REGION Network 62: ALL UNCLAMPED UNIT 02
   RUNG wire#powerrail
      Contact( "DB3510_U2_F1_GRIPPER".CYL.FULL_OPEN )
      wire#w1
      Contact( "DB3810_U2_F4_GRIPPER".CYL.FULL_OPEN )
      wire#w2
      Contact( "DB3610_U2_F2_GRIPPER".CYL.FULL_OPEN )
      wire#w3
      Contact( "DB3710_U2_F3_GRIPPER".CYL.FULL_OPEN )
      wire#w4
      Contact( "DB7215_PART_TYPE".PART_TYPE_U02_FIXTURES )
      Coil( "DB2440_GLOBAL_DATA".GLOBAL_DATA.ALL_UNCLAMPED_UNIT_02 )
   END_RUNG
   RUNG wire#powerrail
      Contact( "DB3500_UNIT_02_FIXTURE_1".CLAMPED_WITHOUT_PART_ANALOG )
   END_RUNG wire#w1
   RUNG wire#w1
      Contact( "DB3800_UNIT_02_FIXTURE_4".CLAMPED_WITHOUT_PART_ANALOG )
   END_RUNG wire#w2
   RUNG wire#powerrail
      I_Contact( "DB7240_HARDWARE_SOFTWARE_ENABLE_DISABLE".DISABLE_FIXTURE.SW_UNIT_2_FIX_1_4_ENABLED )
   END_RUNG wire#w2
   RUNG wire#w2
      Contact( "DB3600_UNIT_02_FIXTURE_2".CLAMPED_WITHOUT_PART_ANALOG )
   END_RUNG wire#w3
   RUNG wire#w3
      Contact( "DB3700_UNIT_02_FIXTURE_3".CLAMPED_WITHOUT_PART_ANALOG )
   END_RUNG wire#w4
   RUNG wire#w2
      I_Contact( "DB7240_HARDWARE_SOFTWARE_ENABLE_DISABLE".DISABLE_FIXTURE.SW_UNIT_2_FIX_2_3_ENABLED )
   END_RUNG wire#w4
   // the same network as SCL:
   "DB2440_GLOBAL_DATA".GLOBAL_DATA.ALL_UNCLAMPED_UNIT_02 := ((("DB3510_U2_F1_GRIPPER".CYL.FULL_OPEN OR "DB3500_UNIT_02_FIXTURE_1".CLAMPED_WITHOUT_PART_ANALOG) AND ("DB3810_U2_F4_GRIPPER".CYL.FULL_OPEN OR "DB3800_UNIT_02_FIXTURE_4".CLAMPED_WITHOUT_PART_ANALOG)) OR NOT "DB7240_HARDWARE_SOFTWARE_ENABLE_DISABLE".DISABLE_FIXTURE.SW_UNIT_2_FIX_1_4_ENABLED) AND ((("DB3610_U2_F2_GRIPPER".CYL.FULL_OPEN OR "DB3600_UNIT_02_FIXTURE_2".CLAMPED_WITHOUT_PART_ANALOG) AND ("DB3710_U2_F3_GRIPPER".CYL.FULL_OPEN OR "DB3700_UNIT_02_FIXTURE_3".CLAMPED_WITHOUT_PART_ANALOG)) OR NOT "DB7240_HARDWARE_SOFTWARE_ENABLE_DISABLE".DISABLE_FIXTURE.SW_UNIT_2_FIX_2_3_ENABLED) AND "DB7215_PART_TYPE".PART_TYPE_U02_FIXTURES;
END_REGION

REGION Network 63: CLAMPED OR UNCLAMPED UNIT 02
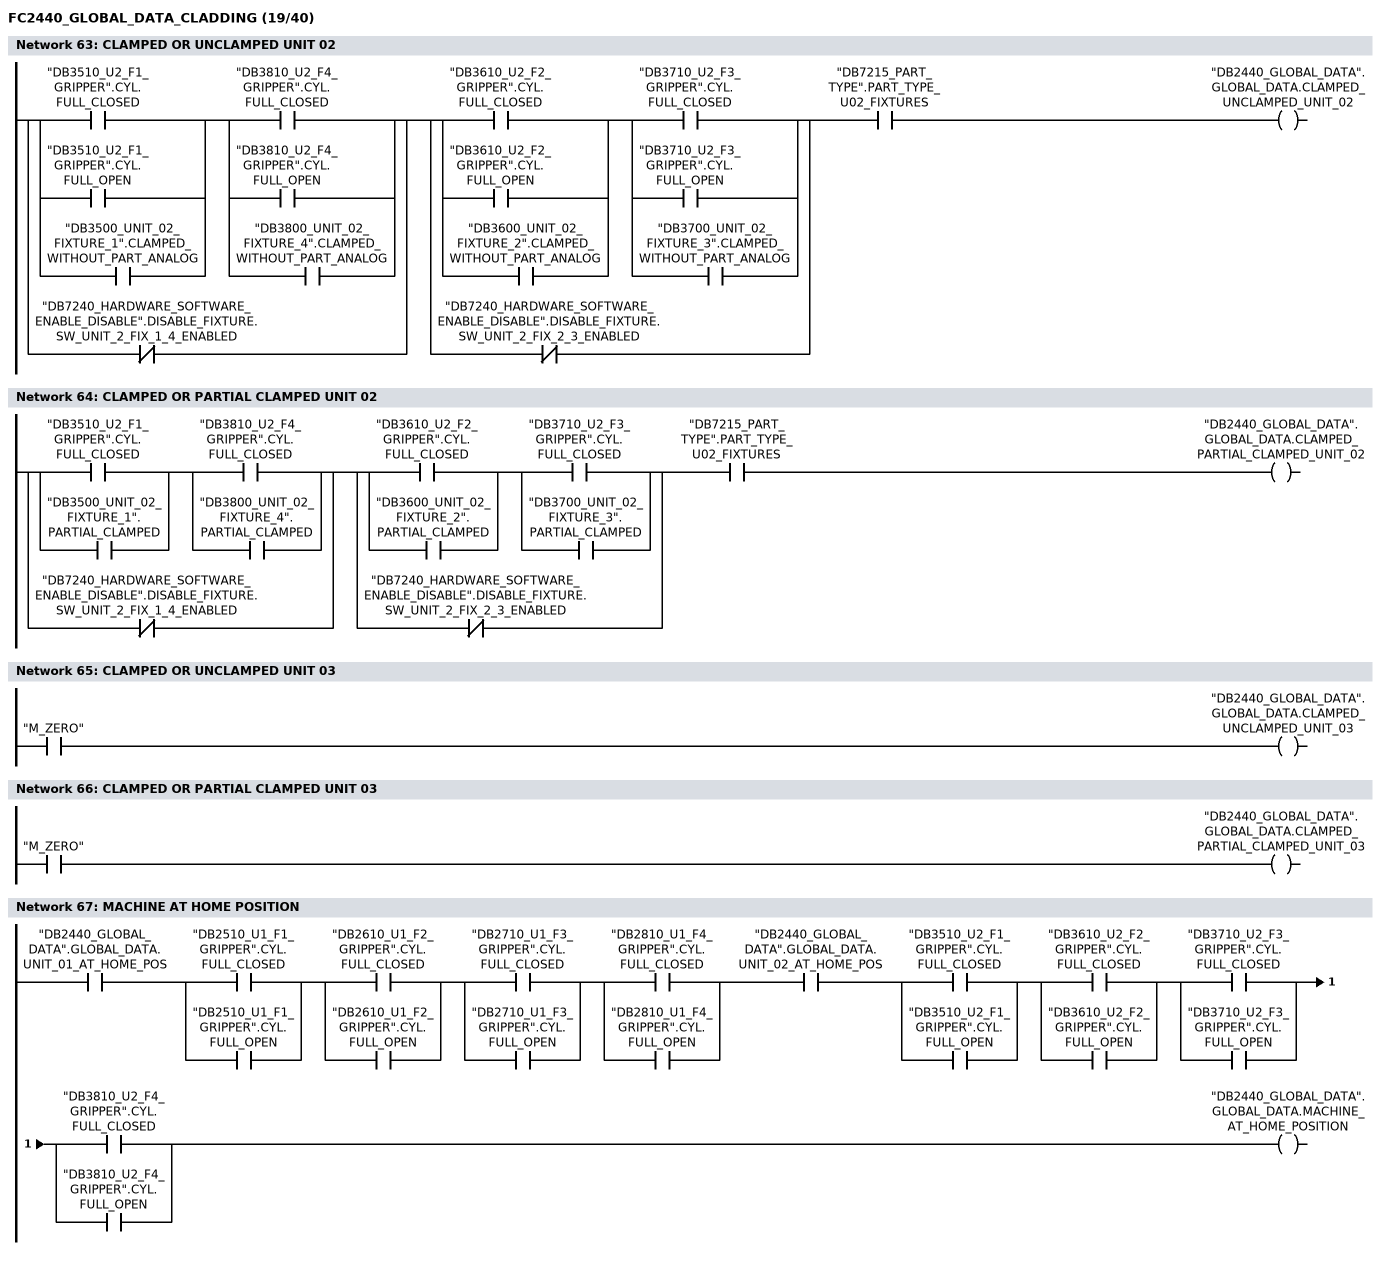
   RUNG wire#powerrail
      Contact( "DB3510_U2_F1_GRIPPER".CYL.FULL_CLOSED )
      wire#w1
      Contact( "DB3810_U2_F4_GRIPPER".CYL.FULL_CLOSED )
      wire#w2
      Contact( "DB3610_U2_F2_GRIPPER".CYL.FULL_CLOSED )
      wire#w3
      Contact( "DB3710_U2_F3_GRIPPER".CYL.FULL_CLOSED )
      wire#w4
      Contact( "DB7215_PART_TYPE".PART_TYPE_U02_FIXTURES )
      Coil( "DB2440_GLOBAL_DATA".GLOBAL_DATA.CLAMPED_UNCLAMPED_UNIT_02 )
   END_RUNG
   RUNG wire#powerrail
      Contact( "DB3510_U2_F1_GRIPPER".CYL.FULL_OPEN )
   END_RUNG wire#w1
   RUNG wire#powerrail
      Contact( "DB3500_UNIT_02_FIXTURE_1".CLAMPED_WITHOUT_PART_ANALOG )
   END_RUNG wire#w1
   RUNG wire#w1
      Contact( "DB3810_U2_F4_GRIPPER".CYL.FULL_OPEN )
   END_RUNG wire#w2
   RUNG wire#w1
      Contact( "DB3800_UNIT_02_FIXTURE_4".CLAMPED_WITHOUT_PART_ANALOG )
   END_RUNG wire#w2
   RUNG wire#powerrail
      I_Contact( "DB7240_HARDWARE_SOFTWARE_ENABLE_DISABLE".DISABLE_FIXTURE.SW_UNIT_2_FIX_1_4_ENABLED )
   END_RUNG wire#w2
   RUNG wire#w2
      Contact( "DB3610_U2_F2_GRIPPER".CYL.FULL_OPEN )
   END_RUNG wire#w3
   RUNG wire#w2
      Contact( "DB3600_UNIT_02_FIXTURE_2".CLAMPED_WITHOUT_PART_ANALOG )
   END_RUNG wire#w3
   RUNG wire#w3
      Contact( "DB3710_U2_F3_GRIPPER".CYL.FULL_OPEN )
   END_RUNG wire#w4
   RUNG wire#w3
      Contact( "DB3700_UNIT_02_FIXTURE_3".CLAMPED_WITHOUT_PART_ANALOG )
   END_RUNG wire#w4
   RUNG wire#w2
      I_Contact( "DB7240_HARDWARE_SOFTWARE_ENABLE_DISABLE".DISABLE_FIXTURE.SW_UNIT_2_FIX_2_3_ENABLED )
   END_RUNG wire#w4
   // the same network as SCL:
   "DB2440_GLOBAL_DATA".GLOBAL_DATA.CLAMPED_UNCLAMPED_UNIT_02 := ((("DB3510_U2_F1_GRIPPER".CYL.FULL_CLOSED OR "DB3510_U2_F1_GRIPPER".CYL.FULL_OPEN OR "DB3500_UNIT_02_FIXTURE_1".CLAMPED_WITHOUT_PART_ANALOG) AND ("DB3810_U2_F4_GRIPPER".CYL.FULL_CLOSED OR "DB3810_U2_F4_GRIPPER".CYL.FULL_OPEN OR "DB3800_UNIT_02_FIXTURE_4".CLAMPED_WITHOUT_PART_ANALOG)) OR NOT "DB7240_HARDWARE_SOFTWARE_ENABLE_DISABLE".DISABLE_FIXTURE.SW_UNIT_2_FIX_1_4_ENABLED) AND ((("DB3610_U2_F2_GRIPPER".CYL.FULL_CLOSED OR "DB3610_U2_F2_GRIPPER".CYL.FULL_OPEN OR "DB3600_UNIT_02_FIXTURE_2".CLAMPED_WITHOUT_PART_ANALOG) AND ("DB3710_U2_F3_GRIPPER".CYL.FULL_CLOSED OR "DB3710_U2_F3_GRIPPER".CYL.FULL_OPEN OR "DB3700_UNIT_02_FIXTURE_3".CLAMPED_WITHOUT_PART_ANALOG)) OR NOT "DB7240_HARDWARE_SOFTWARE_ENABLE_DISABLE".DISABLE_FIXTURE.SW_UNIT_2_FIX_2_3_ENABLED) AND "DB7215_PART_TYPE".PART_TYPE_U02_FIXTURES;
END_REGION

REGION Network 64: CLAMPED OR PARTIAL CLAMPED UNIT 02
   RUNG wire#powerrail
      Contact( "DB3510_U2_F1_GRIPPER".CYL.FULL_CLOSED )
      wire#w1
      Contact( "DB3810_U2_F4_GRIPPER".CYL.FULL_CLOSED )
      wire#w2
      Contact( "DB3610_U2_F2_GRIPPER".CYL.FULL_CLOSED )
      wire#w3
      Contact( "DB3710_U2_F3_GRIPPER".CYL.FULL_CLOSED )
      wire#w4
      Contact( "DB7215_PART_TYPE".PART_TYPE_U02_FIXTURES )
      Coil( "DB2440_GLOBAL_DATA".GLOBAL_DATA.CLAMPED_PARTIAL_CLAMPED_UNIT_02 )
   END_RUNG
   RUNG wire#powerrail
      Contact( "DB3500_UNIT_02_FIXTURE_1".PARTIAL_CLAMPED )
   END_RUNG wire#w1
   RUNG wire#w1
      Contact( "DB3800_UNIT_02_FIXTURE_4".PARTIAL_CLAMPED )
   END_RUNG wire#w2
   RUNG wire#powerrail
      I_Contact( "DB7240_HARDWARE_SOFTWARE_ENABLE_DISABLE".DISABLE_FIXTURE.SW_UNIT_2_FIX_1_4_ENABLED )
   END_RUNG wire#w2
   RUNG wire#w2
      Contact( "DB3600_UNIT_02_FIXTURE_2".PARTIAL_CLAMPED )
   END_RUNG wire#w3
   RUNG wire#w3
      Contact( "DB3700_UNIT_02_FIXTURE_3".PARTIAL_CLAMPED )
   END_RUNG wire#w4
   RUNG wire#w2
      I_Contact( "DB7240_HARDWARE_SOFTWARE_ENABLE_DISABLE".DISABLE_FIXTURE.SW_UNIT_2_FIX_2_3_ENABLED )
   END_RUNG wire#w4
   // the same network as SCL:
   "DB2440_GLOBAL_DATA".GLOBAL_DATA.CLAMPED_PARTIAL_CLAMPED_UNIT_02 := ((("DB3510_U2_F1_GRIPPER".CYL.FULL_CLOSED OR "DB3500_UNIT_02_FIXTURE_1".PARTIAL_CLAMPED) AND ("DB3810_U2_F4_GRIPPER".CYL.FULL_CLOSED OR "DB3800_UNIT_02_FIXTURE_4".PARTIAL_CLAMPED)) OR NOT "DB7240_HARDWARE_SOFTWARE_ENABLE_DISABLE".DISABLE_FIXTURE.SW_UNIT_2_FIX_1_4_ENABLED) AND ((("DB3610_U2_F2_GRIPPER".CYL.FULL_CLOSED OR "DB3600_UNIT_02_FIXTURE_2".PARTIAL_CLAMPED) AND ("DB3710_U2_F3_GRIPPER".CYL.FULL_CLOSED OR "DB3700_UNIT_02_FIXTURE_3".PARTIAL_CLAMPED)) OR NOT "DB7240_HARDWARE_SOFTWARE_ENABLE_DISABLE".DISABLE_FIXTURE.SW_UNIT_2_FIX_2_3_ENABLED) AND "DB7215_PART_TYPE".PART_TYPE_U02_FIXTURES;
END_REGION

REGION Network 65: CLAMPED OR UNCLAMPED UNIT 03
   RUNG wire#powerrail
      Contact( "M_ZERO" )
      Coil( "DB2440_GLOBAL_DATA".GLOBAL_DATA.CLAMPED_UNCLAMPED_UNIT_03 )
   END_RUNG
   // the same network as SCL:
   "DB2440_GLOBAL_DATA".GLOBAL_DATA.CLAMPED_UNCLAMPED_UNIT_03 := "M_ZERO";
END_REGION

REGION Network 66: CLAMPED OR PARTIAL CLAMPED UNIT 03
   RUNG wire#powerrail
      Contact( "M_ZERO" )
      Coil( "DB2440_GLOBAL_DATA".GLOBAL_DATA.CLAMPED_PARTIAL_CLAMPED_UNIT_03 )
   END_RUNG
   // the same network as SCL:
   "DB2440_GLOBAL_DATA".GLOBAL_DATA.CLAMPED_PARTIAL_CLAMPED_UNIT_03 := "M_ZERO";
END_REGION

REGION Network 67: MACHINE AT HOME POSITION
   RUNG wire#powerrail
      Contact( "DB2440_GLOBAL_DATA".GLOBAL_DATA.UNIT_01_AT_HOME_POS )
      wire#w1
      Contact( "DB2510_U1_F1_GRIPPER".CYL.FULL_CLOSED )
      wire#w2
      Contact( "DB2610_U1_F2_GRIPPER".CYL.FULL_CLOSED )
      wire#w3
      Contact( "DB2710_U1_F3_GRIPPER".CYL.FULL_CLOSED )
      wire#w4
      Contact( "DB2810_U1_F4_GRIPPER".CYL.FULL_CLOSED )
      wire#w5
      Contact( "DB2440_GLOBAL_DATA".GLOBAL_DATA.UNIT_02_AT_HOME_POS )
      wire#w6
      Contact( "DB3510_U2_F1_GRIPPER".CYL.FULL_CLOSED )
      wire#w7
      Contact( "DB3610_U2_F2_GRIPPER".CYL.FULL_CLOSED )
      wire#w8
      Contact( "DB3710_U2_F3_GRIPPER".CYL.FULL_CLOSED )
      wire#w9
      Contact( "DB3810_U2_F4_GRIPPER".CYL.FULL_CLOSED )
      wire#w10
      Coil( "DB2440_GLOBAL_DATA".GLOBAL_DATA.MACHINE_AT_HOME_POSITION )
   END_RUNG
   RUNG wire#w1
      Contact( "DB2510_U1_F1_GRIPPER".CYL.FULL_OPEN )
   END_RUNG wire#w2
   RUNG wire#w2
      Contact( "DB2610_U1_F2_GRIPPER".CYL.FULL_OPEN )
   END_RUNG wire#w3
   RUNG wire#w3
      Contact( "DB2710_U1_F3_GRIPPER".CYL.FULL_OPEN )
   END_RUNG wire#w4
   RUNG wire#w4
      Contact( "DB2810_U1_F4_GRIPPER".CYL.FULL_OPEN )
   END_RUNG wire#w5
   RUNG wire#w6
      Contact( "DB3510_U2_F1_GRIPPER".CYL.FULL_OPEN )
   END_RUNG wire#w7
   RUNG wire#w7
      Contact( "DB3610_U2_F2_GRIPPER".CYL.FULL_OPEN )
   END_RUNG wire#w8
   RUNG wire#w8
      Contact( "DB3710_U2_F3_GRIPPER".CYL.FULL_OPEN )
   END_RUNG wire#w9
   RUNG wire#w9
      Contact( "DB3810_U2_F4_GRIPPER".CYL.FULL_OPEN )
   END_RUNG wire#w10
   // the same network as SCL:
   "DB2440_GLOBAL_DATA".GLOBAL_DATA.MACHINE_AT_HOME_POSITION := "DB2440_GLOBAL_DATA".GLOBAL_DATA.UNIT_01_AT_HOME_POS AND ("DB2510_U1_F1_GRIPPER".CYL.FULL_CLOSED OR "DB2510_U1_F1_GRIPPER".CYL.FULL_OPEN) AND ("DB2610_U1_F2_GRIPPER".CYL.FULL_CLOSED OR "DB2610_U1_F2_GRIPPER".CYL.FULL_OPEN) AND ("DB2710_U1_F3_GRIPPER".CYL.FULL_CLOSED OR "DB2710_U1_F3_GRIPPER".CYL.FULL_OPEN) AND ("DB2810_U1_F4_GRIPPER".CYL.FULL_CLOSED OR "DB2810_U1_F4_GRIPPER".CYL.FULL_OPEN) AND "DB2440_GLOBAL_DATA".GLOBAL_DATA.UNIT_02_AT_HOME_POS AND ("DB3510_U2_F1_GRIPPER".CYL.FULL_CLOSED OR "DB3510_U2_F1_GRIPPER".CYL.FULL_OPEN) AND ("DB3610_U2_F2_GRIPPER".CYL.FULL_CLOSED OR "DB3610_U2_F2_GRIPPER".CYL.FULL_OPEN) AND ("DB3710_U2_F3_GRIPPER".CYL.FULL_CLOSED OR "DB3710_U2_F3_GRIPPER".CYL.FULL_OPEN) AND ("DB3810_U2_F4_GRIPPER".CYL.FULL_CLOSED OR "DB3810_U2_F4_GRIPPER".CYL.FULL_OPEN);
END_REGION

REGION Network 68: UNIT 01 STATION 0 ANY CYCLE ACTIVE
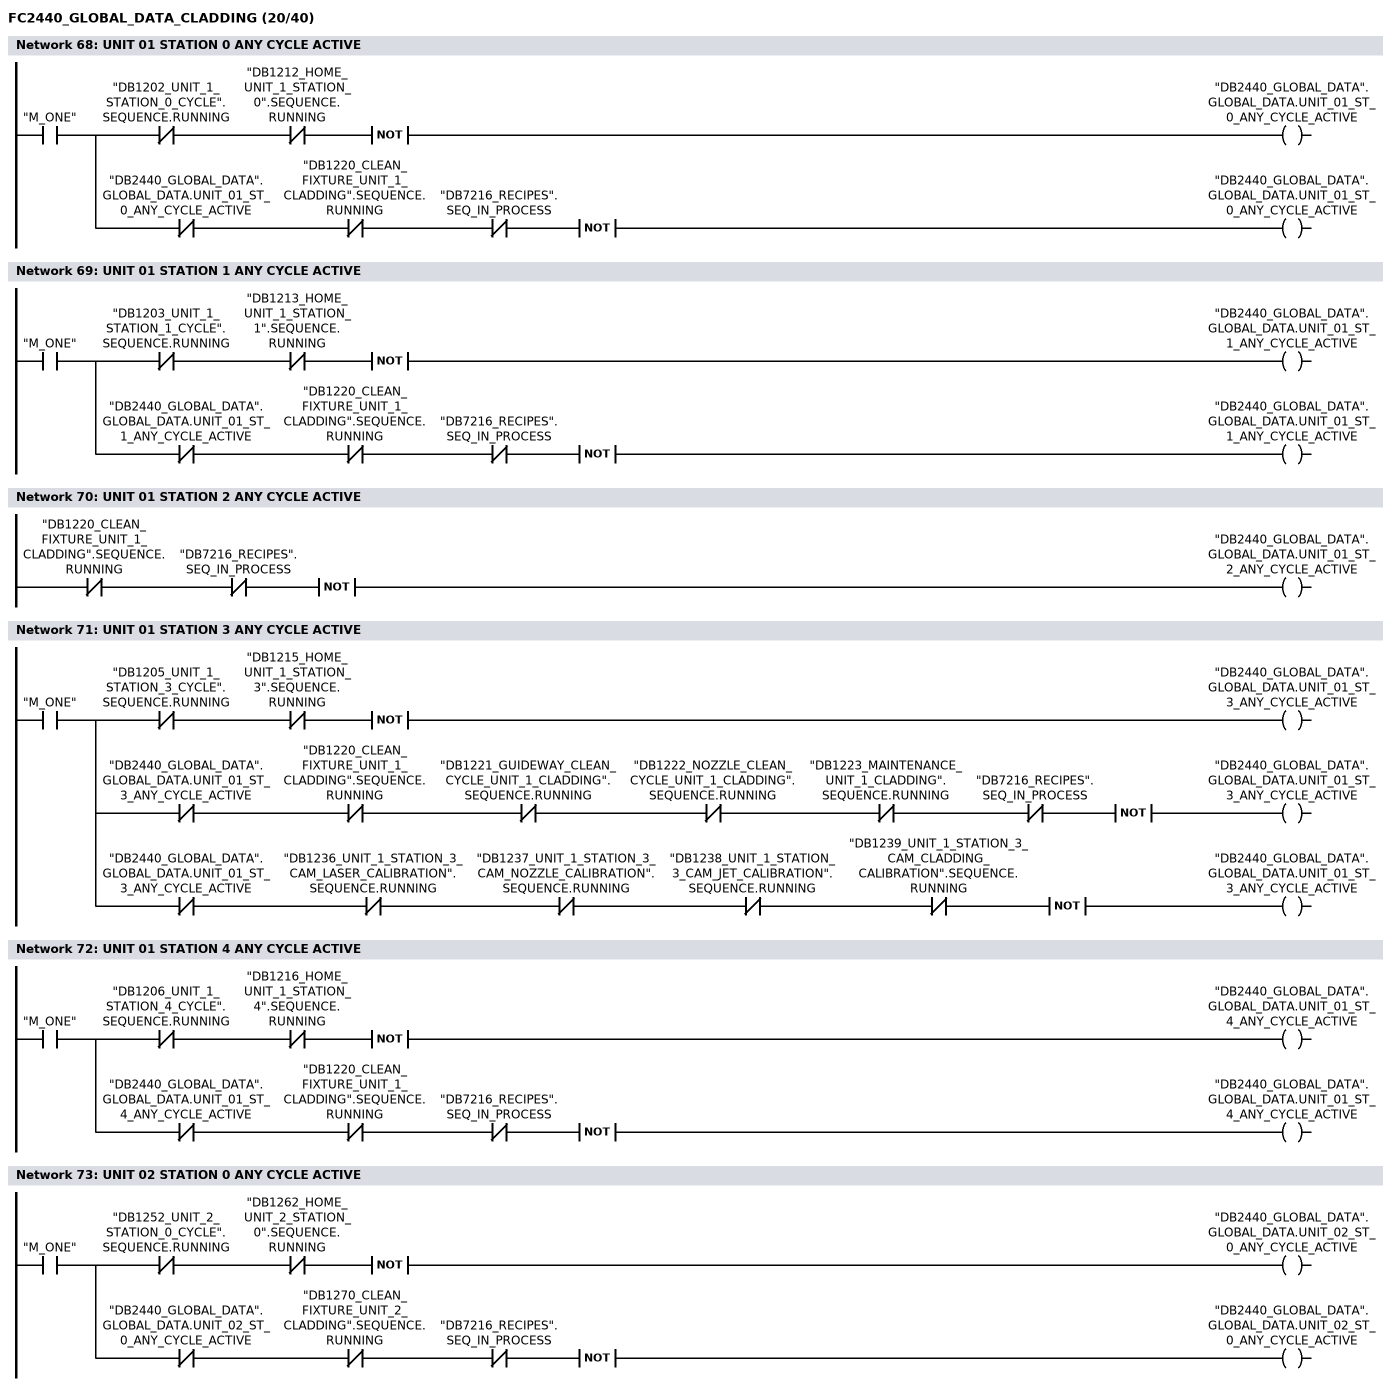
   RUNG wire#powerrail
      Contact( "M_ONE" )
      wire#w1
      I_Contact( "DB1202_UNIT_1_STATION_0_CYCLE".SEQUENCE.RUNNING )
      I_Contact( "DB1212_HOME_UNIT_1_STATION_0".SEQUENCE.RUNNING )
      Not()
      Coil( "DB2440_GLOBAL_DATA".GLOBAL_DATA.UNIT_01_ST_0_ANY_CYCLE_ACTIVE )
   END_RUNG
   RUNG wire#w1
      I_Contact( "DB2440_GLOBAL_DATA".GLOBAL_DATA.UNIT_01_ST_0_ANY_CYCLE_ACTIVE )
      I_Contact( "DB1220_CLEAN_FIXTURE_UNIT_1_CLADDING".SEQUENCE.RUNNING )
      I_Contact( "DB7216_RECIPES".SEQ_IN_PROCESS )
      Not()
      Coil( "DB2440_GLOBAL_DATA".GLOBAL_DATA.UNIT_01_ST_0_ANY_CYCLE_ACTIVE )
   END_RUNG
   // the same network as SCL:
   "DB2440_GLOBAL_DATA".GLOBAL_DATA.UNIT_01_ST_0_ANY_CYCLE_ACTIVE := NOT ("M_ONE" AND NOT "DB1202_UNIT_1_STATION_0_CYCLE".SEQUENCE.RUNNING AND NOT "DB1212_HOME_UNIT_1_STATION_0".SEQUENCE.RUNNING);
   "DB2440_GLOBAL_DATA".GLOBAL_DATA.UNIT_01_ST_0_ANY_CYCLE_ACTIVE := NOT ("M_ONE" AND NOT "DB2440_GLOBAL_DATA".GLOBAL_DATA.UNIT_01_ST_0_ANY_CYCLE_ACTIVE AND NOT "DB1220_CLEAN_FIXTURE_UNIT_1_CLADDING".SEQUENCE.RUNNING AND NOT "DB7216_RECIPES".SEQ_IN_PROCESS);
END_REGION

REGION Network 69: UNIT 01 STATION 1 ANY CYCLE ACTIVE
   RUNG wire#powerrail
      Contact( "M_ONE" )
      wire#w1
      I_Contact( "DB1203_UNIT_1_STATION_1_CYCLE".SEQUENCE.RUNNING )
      I_Contact( "DB1213_HOME_UNIT_1_STATION_1".SEQUENCE.RUNNING )
      Not()
      Coil( "DB2440_GLOBAL_DATA".GLOBAL_DATA.UNIT_01_ST_1_ANY_CYCLE_ACTIVE )
   END_RUNG
   RUNG wire#w1
      I_Contact( "DB2440_GLOBAL_DATA".GLOBAL_DATA.UNIT_01_ST_1_ANY_CYCLE_ACTIVE )
      I_Contact( "DB1220_CLEAN_FIXTURE_UNIT_1_CLADDING".SEQUENCE.RUNNING )
      I_Contact( "DB7216_RECIPES".SEQ_IN_PROCESS )
      Not()
      Coil( "DB2440_GLOBAL_DATA".GLOBAL_DATA.UNIT_01_ST_1_ANY_CYCLE_ACTIVE )
   END_RUNG
   // the same network as SCL:
   "DB2440_GLOBAL_DATA".GLOBAL_DATA.UNIT_01_ST_1_ANY_CYCLE_ACTIVE := NOT ("M_ONE" AND NOT "DB1203_UNIT_1_STATION_1_CYCLE".SEQUENCE.RUNNING AND NOT "DB1213_HOME_UNIT_1_STATION_1".SEQUENCE.RUNNING);
   "DB2440_GLOBAL_DATA".GLOBAL_DATA.UNIT_01_ST_1_ANY_CYCLE_ACTIVE := NOT ("M_ONE" AND NOT "DB2440_GLOBAL_DATA".GLOBAL_DATA.UNIT_01_ST_1_ANY_CYCLE_ACTIVE AND NOT "DB1220_CLEAN_FIXTURE_UNIT_1_CLADDING".SEQUENCE.RUNNING AND NOT "DB7216_RECIPES".SEQ_IN_PROCESS);
END_REGION

REGION Network 70: UNIT 01 STATION 2 ANY CYCLE ACTIVE
   RUNG wire#powerrail
      I_Contact( "DB1220_CLEAN_FIXTURE_UNIT_1_CLADDING".SEQUENCE.RUNNING )
      I_Contact( "DB7216_RECIPES".SEQ_IN_PROCESS )
      Not()
      Coil( "DB2440_GLOBAL_DATA".GLOBAL_DATA.UNIT_01_ST_2_ANY_CYCLE_ACTIVE )
   END_RUNG
   // the same network as SCL:
   "DB2440_GLOBAL_DATA".GLOBAL_DATA.UNIT_01_ST_2_ANY_CYCLE_ACTIVE := NOT (NOT "DB1220_CLEAN_FIXTURE_UNIT_1_CLADDING".SEQUENCE.RUNNING AND NOT "DB7216_RECIPES".SEQ_IN_PROCESS);
END_REGION

REGION Network 71: UNIT 01 STATION 3 ANY CYCLE ACTIVE
   RUNG wire#powerrail
      Contact( "M_ONE" )
      wire#w1
      I_Contact( "DB1205_UNIT_1_STATION_3_CYCLE".SEQUENCE.RUNNING )
      I_Contact( "DB1215_HOME_UNIT_1_STATION_3".SEQUENCE.RUNNING )
      Not()
      Coil( "DB2440_GLOBAL_DATA".GLOBAL_DATA.UNIT_01_ST_3_ANY_CYCLE_ACTIVE )
   END_RUNG
   RUNG wire#w1
      I_Contact( "DB2440_GLOBAL_DATA".GLOBAL_DATA.UNIT_01_ST_3_ANY_CYCLE_ACTIVE )
      I_Contact( "DB1220_CLEAN_FIXTURE_UNIT_1_CLADDING".SEQUENCE.RUNNING )
      I_Contact( "DB1221_GUIDEWAY_CLEAN_CYCLE_UNIT_1_CLADDING".SEQUENCE.RUNNING )
      I_Contact( "DB1222_NOZZLE_CLEAN_CYCLE_UNIT_1_CLADDING".SEQUENCE.RUNNING )
      I_Contact( "DB1223_MAINTENANCE_UNIT_1_CLADDING".SEQUENCE.RUNNING )
      I_Contact( "DB7216_RECIPES".SEQ_IN_PROCESS )
      Not()
      Coil( "DB2440_GLOBAL_DATA".GLOBAL_DATA.UNIT_01_ST_3_ANY_CYCLE_ACTIVE )
   END_RUNG
   RUNG wire#w1
      I_Contact( "DB2440_GLOBAL_DATA".GLOBAL_DATA.UNIT_01_ST_3_ANY_CYCLE_ACTIVE )
      I_Contact( "DB1236_UNIT_1_STATION_3_CAM_LASER_CALIBRATION".SEQUENCE.RUNNING )
      I_Contact( "DB1237_UNIT_1_STATION_3_CAM_NOZZLE_CALIBRATION".SEQUENCE.RUNNING )
      I_Contact( "DB1238_UNIT_1_STATION_3_CAM_JET_CALIBRATION".SEQUENCE.RUNNING )
      I_Contact( "DB1239_UNIT_1_STATION_3_CAM_CLADDING_CALIBRATION".SEQUENCE.RUNNING )
      Not()
      Coil( "DB2440_GLOBAL_DATA".GLOBAL_DATA.UNIT_01_ST_3_ANY_CYCLE_ACTIVE )
   END_RUNG
   // the same network as SCL:
   "DB2440_GLOBAL_DATA".GLOBAL_DATA.UNIT_01_ST_3_ANY_CYCLE_ACTIVE := NOT ("M_ONE" AND NOT "DB1205_UNIT_1_STATION_3_CYCLE".SEQUENCE.RUNNING AND NOT "DB1215_HOME_UNIT_1_STATION_3".SEQUENCE.RUNNING);
   "DB2440_GLOBAL_DATA".GLOBAL_DATA.UNIT_01_ST_3_ANY_CYCLE_ACTIVE := NOT ("M_ONE" AND NOT "DB2440_GLOBAL_DATA".GLOBAL_DATA.UNIT_01_ST_3_ANY_CYCLE_ACTIVE AND NOT "DB1220_CLEAN_FIXTURE_UNIT_1_CLADDING".SEQUENCE.RUNNING AND NOT "DB1221_GUIDEWAY_CLEAN_CYCLE_UNIT_1_CLADDING".SEQUENCE.RUNNING AND NOT "DB1222_NOZZLE_CLEAN_CYCLE_UNIT_1_CLADDING".SEQUENCE.RUNNING AND NOT "DB1223_MAINTENANCE_UNIT_1_CLADDING".SEQUENCE.RUNNING AND NOT "DB7216_RECIPES".SEQ_IN_PROCESS);
   "DB2440_GLOBAL_DATA".GLOBAL_DATA.UNIT_01_ST_3_ANY_CYCLE_ACTIVE := NOT ("M_ONE" AND NOT "DB2440_GLOBAL_DATA".GLOBAL_DATA.UNIT_01_ST_3_ANY_CYCLE_ACTIVE AND NOT "DB1236_UNIT_1_STATION_3_CAM_LASER_CALIBRATION".SEQUENCE.RUNNING AND NOT "DB1237_UNIT_1_STATION_3_CAM_NOZZLE_CALIBRATION".SEQUENCE.RUNNING AND NOT "DB1238_UNIT_1_STATION_3_CAM_JET_CALIBRATION".SEQUENCE.RUNNING AND NOT "DB1239_UNIT_1_STATION_3_CAM_CLADDING_CALIBRATION".SEQUENCE.RUNNING);
END_REGION

REGION Network 72: UNIT 01 STATION 4 ANY CYCLE ACTIVE
   RUNG wire#powerrail
      Contact( "M_ONE" )
      wire#w1
      I_Contact( "DB1206_UNIT_1_STATION_4_CYCLE".SEQUENCE.RUNNING )
      I_Contact( "DB1216_HOME_UNIT_1_STATION_4".SEQUENCE.RUNNING )
      Not()
      Coil( "DB2440_GLOBAL_DATA".GLOBAL_DATA.UNIT_01_ST_4_ANY_CYCLE_ACTIVE )
   END_RUNG
   RUNG wire#w1
      I_Contact( "DB2440_GLOBAL_DATA".GLOBAL_DATA.UNIT_01_ST_4_ANY_CYCLE_ACTIVE )
      I_Contact( "DB1220_CLEAN_FIXTURE_UNIT_1_CLADDING".SEQUENCE.RUNNING )
      I_Contact( "DB7216_RECIPES".SEQ_IN_PROCESS )
      Not()
      Coil( "DB2440_GLOBAL_DATA".GLOBAL_DATA.UNIT_01_ST_4_ANY_CYCLE_ACTIVE )
   END_RUNG
   // the same network as SCL:
   "DB2440_GLOBAL_DATA".GLOBAL_DATA.UNIT_01_ST_4_ANY_CYCLE_ACTIVE := NOT ("M_ONE" AND NOT "DB1206_UNIT_1_STATION_4_CYCLE".SEQUENCE.RUNNING AND NOT "DB1216_HOME_UNIT_1_STATION_4".SEQUENCE.RUNNING);
   "DB2440_GLOBAL_DATA".GLOBAL_DATA.UNIT_01_ST_4_ANY_CYCLE_ACTIVE := NOT ("M_ONE" AND NOT "DB2440_GLOBAL_DATA".GLOBAL_DATA.UNIT_01_ST_4_ANY_CYCLE_ACTIVE AND NOT "DB1220_CLEAN_FIXTURE_UNIT_1_CLADDING".SEQUENCE.RUNNING AND NOT "DB7216_RECIPES".SEQ_IN_PROCESS);
END_REGION

REGION Network 73: UNIT 02 STATION 0 ANY CYCLE ACTIVE
   RUNG wire#powerrail
      Contact( "M_ONE" )
      wire#w1
      I_Contact( "DB1252_UNIT_2_STATION_0_CYCLE".SEQUENCE.RUNNING )
      I_Contact( "DB1262_HOME_UNIT_2_STATION_0".SEQUENCE.RUNNING )
      Not()
      Coil( "DB2440_GLOBAL_DATA".GLOBAL_DATA.UNIT_02_ST_0_ANY_CYCLE_ACTIVE )
   END_RUNG
   RUNG wire#w1
      I_Contact( "DB2440_GLOBAL_DATA".GLOBAL_DATA.UNIT_02_ST_0_ANY_CYCLE_ACTIVE )
      I_Contact( "DB1270_CLEAN_FIXTURE_UNIT_2_CLADDING".SEQUENCE.RUNNING )
      I_Contact( "DB7216_RECIPES".SEQ_IN_PROCESS )
      Not()
      Coil( "DB2440_GLOBAL_DATA".GLOBAL_DATA.UNIT_02_ST_0_ANY_CYCLE_ACTIVE )
   END_RUNG
   // the same network as SCL:
   "DB2440_GLOBAL_DATA".GLOBAL_DATA.UNIT_02_ST_0_ANY_CYCLE_ACTIVE := NOT ("M_ONE" AND NOT "DB1252_UNIT_2_STATION_0_CYCLE".SEQUENCE.RUNNING AND NOT "DB1262_HOME_UNIT_2_STATION_0".SEQUENCE.RUNNING);
   "DB2440_GLOBAL_DATA".GLOBAL_DATA.UNIT_02_ST_0_ANY_CYCLE_ACTIVE := NOT ("M_ONE" AND NOT "DB2440_GLOBAL_DATA".GLOBAL_DATA.UNIT_02_ST_0_ANY_CYCLE_ACTIVE AND NOT "DB1270_CLEAN_FIXTURE_UNIT_2_CLADDING".SEQUENCE.RUNNING AND NOT "DB7216_RECIPES".SEQ_IN_PROCESS);
END_REGION

REGION Network 74: UNIT 02 STATION 1 ANY CYCLE ACTIVE
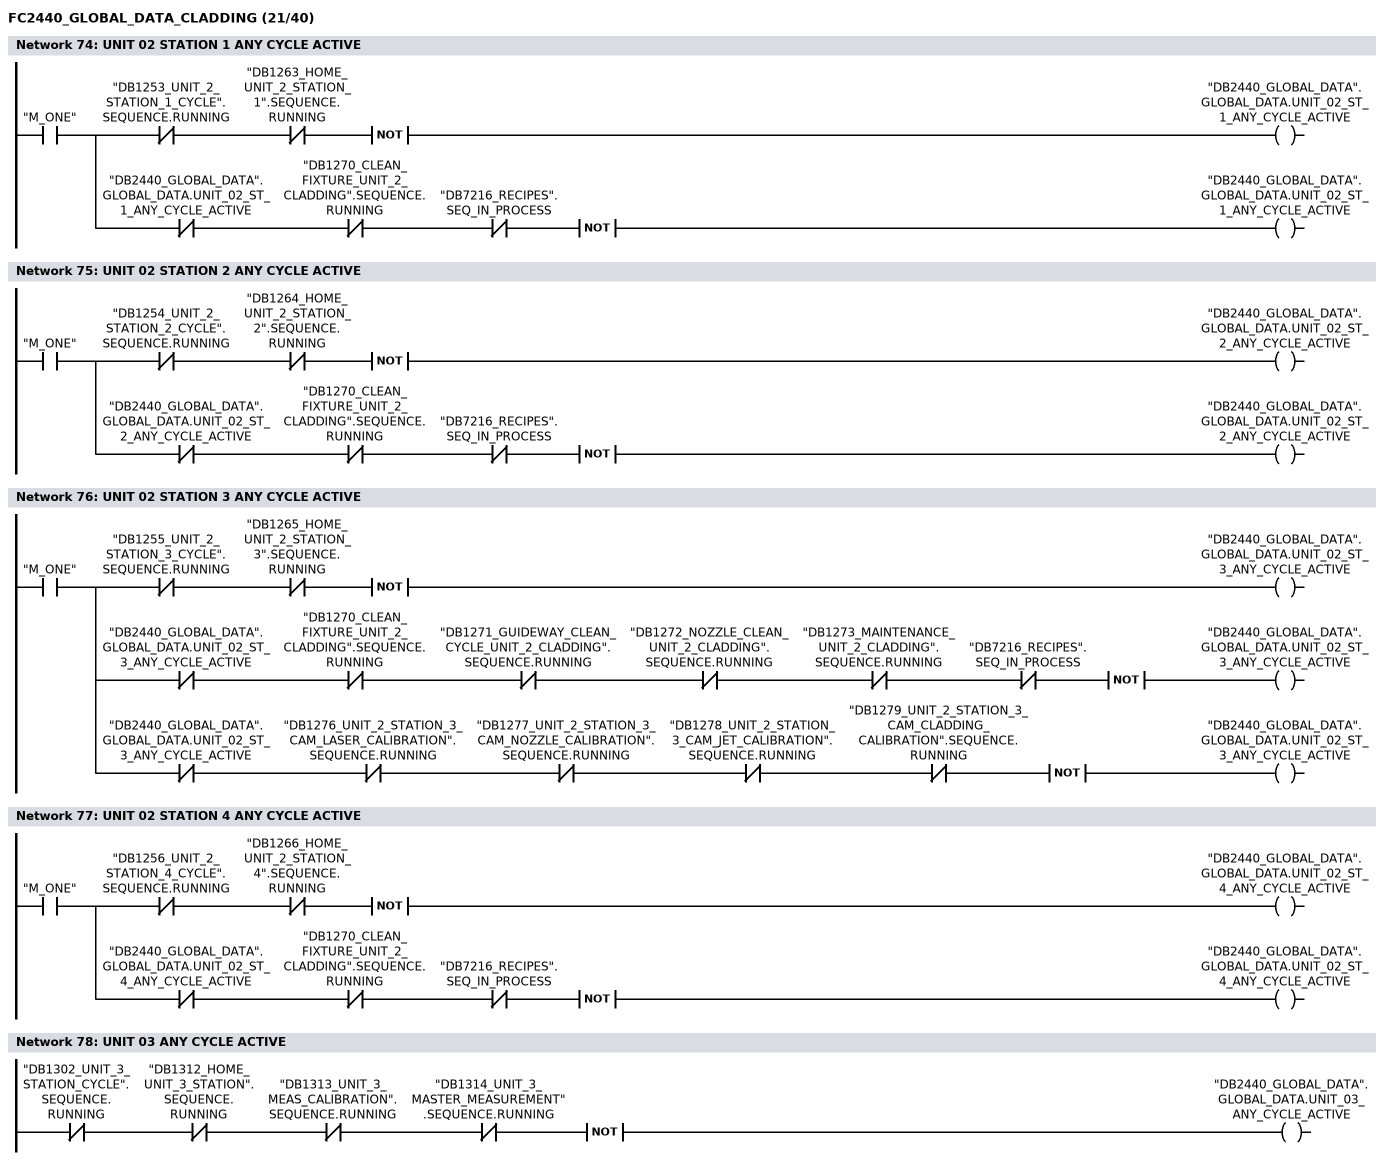
   RUNG wire#powerrail
      Contact( "M_ONE" )
      wire#w1
      I_Contact( "DB1253_UNIT_2_STATION_1_CYCLE".SEQUENCE.RUNNING )
      I_Contact( "DB1263_HOME_UNIT_2_STATION_1".SEQUENCE.RUNNING )
      Not()
      Coil( "DB2440_GLOBAL_DATA".GLOBAL_DATA.UNIT_02_ST_1_ANY_CYCLE_ACTIVE )
   END_RUNG
   RUNG wire#w1
      I_Contact( "DB2440_GLOBAL_DATA".GLOBAL_DATA.UNIT_02_ST_1_ANY_CYCLE_ACTIVE )
      I_Contact( "DB1270_CLEAN_FIXTURE_UNIT_2_CLADDING".SEQUENCE.RUNNING )
      I_Contact( "DB7216_RECIPES".SEQ_IN_PROCESS )
      Not()
      Coil( "DB2440_GLOBAL_DATA".GLOBAL_DATA.UNIT_02_ST_1_ANY_CYCLE_ACTIVE )
   END_RUNG
   // the same network as SCL:
   "DB2440_GLOBAL_DATA".GLOBAL_DATA.UNIT_02_ST_1_ANY_CYCLE_ACTIVE := NOT ("M_ONE" AND NOT "DB1253_UNIT_2_STATION_1_CYCLE".SEQUENCE.RUNNING AND NOT "DB1263_HOME_UNIT_2_STATION_1".SEQUENCE.RUNNING);
   "DB2440_GLOBAL_DATA".GLOBAL_DATA.UNIT_02_ST_1_ANY_CYCLE_ACTIVE := NOT ("M_ONE" AND NOT "DB2440_GLOBAL_DATA".GLOBAL_DATA.UNIT_02_ST_1_ANY_CYCLE_ACTIVE AND NOT "DB1270_CLEAN_FIXTURE_UNIT_2_CLADDING".SEQUENCE.RUNNING AND NOT "DB7216_RECIPES".SEQ_IN_PROCESS);
END_REGION

REGION Network 75: UNIT 02 STATION 2 ANY CYCLE ACTIVE
   RUNG wire#powerrail
      Contact( "M_ONE" )
      wire#w1
      I_Contact( "DB1254_UNIT_2_STATION_2_CYCLE".SEQUENCE.RUNNING )
      I_Contact( "DB1264_HOME_UNIT_2_STATION_2".SEQUENCE.RUNNING )
      Not()
      Coil( "DB2440_GLOBAL_DATA".GLOBAL_DATA.UNIT_02_ST_2_ANY_CYCLE_ACTIVE )
   END_RUNG
   RUNG wire#w1
      I_Contact( "DB2440_GLOBAL_DATA".GLOBAL_DATA.UNIT_02_ST_2_ANY_CYCLE_ACTIVE )
      I_Contact( "DB1270_CLEAN_FIXTURE_UNIT_2_CLADDING".SEQUENCE.RUNNING )
      I_Contact( "DB7216_RECIPES".SEQ_IN_PROCESS )
      Not()
      Coil( "DB2440_GLOBAL_DATA".GLOBAL_DATA.UNIT_02_ST_2_ANY_CYCLE_ACTIVE )
   END_RUNG
   // the same network as SCL:
   "DB2440_GLOBAL_DATA".GLOBAL_DATA.UNIT_02_ST_2_ANY_CYCLE_ACTIVE := NOT ("M_ONE" AND NOT "DB1254_UNIT_2_STATION_2_CYCLE".SEQUENCE.RUNNING AND NOT "DB1264_HOME_UNIT_2_STATION_2".SEQUENCE.RUNNING);
   "DB2440_GLOBAL_DATA".GLOBAL_DATA.UNIT_02_ST_2_ANY_CYCLE_ACTIVE := NOT ("M_ONE" AND NOT "DB2440_GLOBAL_DATA".GLOBAL_DATA.UNIT_02_ST_2_ANY_CYCLE_ACTIVE AND NOT "DB1270_CLEAN_FIXTURE_UNIT_2_CLADDING".SEQUENCE.RUNNING AND NOT "DB7216_RECIPES".SEQ_IN_PROCESS);
END_REGION

REGION Network 76: UNIT 02 STATION 3 ANY CYCLE ACTIVE
   RUNG wire#powerrail
      Contact( "M_ONE" )
      wire#w1
      I_Contact( "DB1255_UNIT_2_STATION_3_CYCLE".SEQUENCE.RUNNING )
      I_Contact( "DB1265_HOME_UNIT_2_STATION_3".SEQUENCE.RUNNING )
      Not()
      Coil( "DB2440_GLOBAL_DATA".GLOBAL_DATA.UNIT_02_ST_3_ANY_CYCLE_ACTIVE )
   END_RUNG
   RUNG wire#w1
      I_Contact( "DB2440_GLOBAL_DATA".GLOBAL_DATA.UNIT_02_ST_3_ANY_CYCLE_ACTIVE )
      I_Contact( "DB1270_CLEAN_FIXTURE_UNIT_2_CLADDING".SEQUENCE.RUNNING )
      I_Contact( "DB1271_GUIDEWAY_CLEAN_CYCLE_UNIT_2_CLADDING".SEQUENCE.RUNNING )
      I_Contact( "DB1272_NOZZLE_CLEAN_UNIT_2_CLADDING".SEQUENCE.RUNNING )
      I_Contact( "DB1273_MAINTENANCE_UNIT_2_CLADDING".SEQUENCE.RUNNING )
      I_Contact( "DB7216_RECIPES".SEQ_IN_PROCESS )
      Not()
      Coil( "DB2440_GLOBAL_DATA".GLOBAL_DATA.UNIT_02_ST_3_ANY_CYCLE_ACTIVE )
   END_RUNG
   RUNG wire#w1
      I_Contact( "DB2440_GLOBAL_DATA".GLOBAL_DATA.UNIT_02_ST_3_ANY_CYCLE_ACTIVE )
      I_Contact( "DB1276_UNIT_2_STATION_3_CAM_LASER_CALIBRATION".SEQUENCE.RUNNING )
      I_Contact( "DB1277_UNIT_2_STATION_3_CAM_NOZZLE_CALIBRATION".SEQUENCE.RUNNING )
      I_Contact( "DB1278_UNIT_2_STATION_3_CAM_JET_CALIBRATION".SEQUENCE.RUNNING )
      I_Contact( "DB1279_UNIT_2_STATION_3_CAM_CLADDING_CALIBRATION".SEQUENCE.RUNNING )
      Not()
      Coil( "DB2440_GLOBAL_DATA".GLOBAL_DATA.UNIT_02_ST_3_ANY_CYCLE_ACTIVE )
   END_RUNG
   // the same network as SCL:
   "DB2440_GLOBAL_DATA".GLOBAL_DATA.UNIT_02_ST_3_ANY_CYCLE_ACTIVE := NOT ("M_ONE" AND NOT "DB1255_UNIT_2_STATION_3_CYCLE".SEQUENCE.RUNNING AND NOT "DB1265_HOME_UNIT_2_STATION_3".SEQUENCE.RUNNING);
   "DB2440_GLOBAL_DATA".GLOBAL_DATA.UNIT_02_ST_3_ANY_CYCLE_ACTIVE := NOT ("M_ONE" AND NOT "DB2440_GLOBAL_DATA".GLOBAL_DATA.UNIT_02_ST_3_ANY_CYCLE_ACTIVE AND NOT "DB1270_CLEAN_FIXTURE_UNIT_2_CLADDING".SEQUENCE.RUNNING AND NOT "DB1271_GUIDEWAY_CLEAN_CYCLE_UNIT_2_CLADDING".SEQUENCE.RUNNING AND NOT "DB1272_NOZZLE_CLEAN_UNIT_2_CLADDING".SEQUENCE.RUNNING AND NOT "DB1273_MAINTENANCE_UNIT_2_CLADDING".SEQUENCE.RUNNING AND NOT "DB7216_RECIPES".SEQ_IN_PROCESS);
   "DB2440_GLOBAL_DATA".GLOBAL_DATA.UNIT_02_ST_3_ANY_CYCLE_ACTIVE := NOT ("M_ONE" AND NOT "DB2440_GLOBAL_DATA".GLOBAL_DATA.UNIT_02_ST_3_ANY_CYCLE_ACTIVE AND NOT "DB1276_UNIT_2_STATION_3_CAM_LASER_CALIBRATION".SEQUENCE.RUNNING AND NOT "DB1277_UNIT_2_STATION_3_CAM_NOZZLE_CALIBRATION".SEQUENCE.RUNNING AND NOT "DB1278_UNIT_2_STATION_3_CAM_JET_CALIBRATION".SEQUENCE.RUNNING AND NOT "DB1279_UNIT_2_STATION_3_CAM_CLADDING_CALIBRATION".SEQUENCE.RUNNING);
END_REGION

REGION Network 77: UNIT 02 STATION 4 ANY CYCLE ACTIVE
   RUNG wire#powerrail
      Contact( "M_ONE" )
      wire#w1
      I_Contact( "DB1256_UNIT_2_STATION_4_CYCLE".SEQUENCE.RUNNING )
      I_Contact( "DB1266_HOME_UNIT_2_STATION_4".SEQUENCE.RUNNING )
      Not()
      Coil( "DB2440_GLOBAL_DATA".GLOBAL_DATA.UNIT_02_ST_4_ANY_CYCLE_ACTIVE )
   END_RUNG
   RUNG wire#w1
      I_Contact( "DB2440_GLOBAL_DATA".GLOBAL_DATA.UNIT_02_ST_4_ANY_CYCLE_ACTIVE )
      I_Contact( "DB1270_CLEAN_FIXTURE_UNIT_2_CLADDING".SEQUENCE.RUNNING )
      I_Contact( "DB7216_RECIPES".SEQ_IN_PROCESS )
      Not()
      Coil( "DB2440_GLOBAL_DATA".GLOBAL_DATA.UNIT_02_ST_4_ANY_CYCLE_ACTIVE )
   END_RUNG
   // the same network as SCL:
   "DB2440_GLOBAL_DATA".GLOBAL_DATA.UNIT_02_ST_4_ANY_CYCLE_ACTIVE := NOT ("M_ONE" AND NOT "DB1256_UNIT_2_STATION_4_CYCLE".SEQUENCE.RUNNING AND NOT "DB1266_HOME_UNIT_2_STATION_4".SEQUENCE.RUNNING);
   "DB2440_GLOBAL_DATA".GLOBAL_DATA.UNIT_02_ST_4_ANY_CYCLE_ACTIVE := NOT ("M_ONE" AND NOT "DB2440_GLOBAL_DATA".GLOBAL_DATA.UNIT_02_ST_4_ANY_CYCLE_ACTIVE AND NOT "DB1270_CLEAN_FIXTURE_UNIT_2_CLADDING".SEQUENCE.RUNNING AND NOT "DB7216_RECIPES".SEQ_IN_PROCESS);
END_REGION

REGION Network 78: UNIT 03 ANY CYCLE ACTIVE
   RUNG wire#powerrail
      I_Contact( "DB1302_UNIT_3_STATION_CYCLE".SEQUENCE.RUNNING )
      I_Contact( "DB1312_HOME_UNIT_3_STATION".SEQUENCE.RUNNING )
      I_Contact( "DB1313_UNIT_3_MEAS_CALIBRATION".SEQUENCE.RUNNING )
      I_Contact( "DB1314_UNIT_3_MASTER_MEASUREMENT".SEQUENCE.RUNNING )
      Not()
      Coil( "DB2440_GLOBAL_DATA".GLOBAL_DATA.UNIT_03_ANY_CYCLE_ACTIVE )
   END_RUNG
   // the same network as SCL:
   "DB2440_GLOBAL_DATA".GLOBAL_DATA.UNIT_03_ANY_CYCLE_ACTIVE := NOT (NOT "DB1302_UNIT_3_STATION_CYCLE".SEQUENCE.RUNNING AND NOT "DB1312_HOME_UNIT_3_STATION".SEQUENCE.RUNNING AND NOT "DB1313_UNIT_3_MEAS_CALIBRATION".SEQUENCE.RUNNING AND NOT "DB1314_UNIT_3_MASTER_MEASUREMENT".SEQUENCE.RUNNING);
END_REGION

REGION Network 79: ANY UNIT 01 CYCLE RUNNING
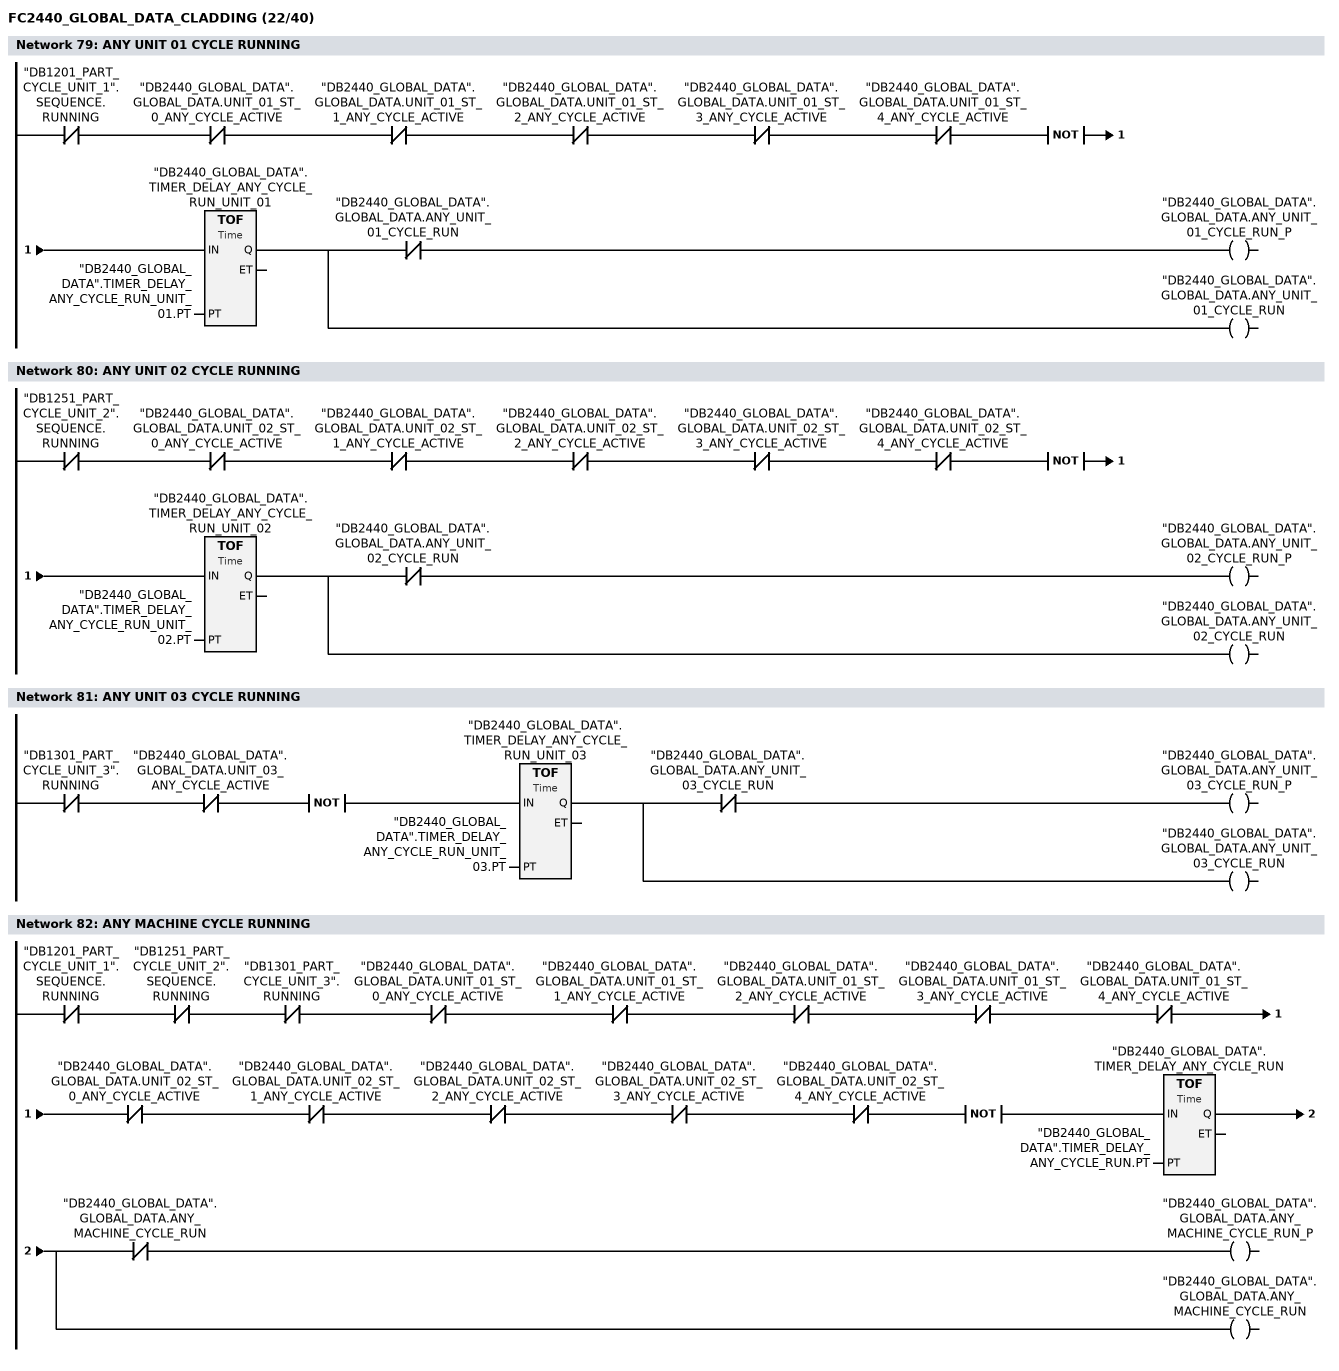
   RUNG wire#powerrail
      I_Contact( "DB1201_PART_CYCLE_UNIT_1".SEQUENCE.RUNNING )
      I_Contact( "DB2440_GLOBAL_DATA".GLOBAL_DATA.UNIT_01_ST_0_ANY_CYCLE_ACTIVE )
      I_Contact( "DB2440_GLOBAL_DATA".GLOBAL_DATA.UNIT_01_ST_1_ANY_CYCLE_ACTIVE )
      I_Contact( "DB2440_GLOBAL_DATA".GLOBAL_DATA.UNIT_01_ST_2_ANY_CYCLE_ACTIVE )
      I_Contact( "DB2440_GLOBAL_DATA".GLOBAL_DATA.UNIT_01_ST_3_ANY_CYCLE_ACTIVE )
      I_Contact( "DB2440_GLOBAL_DATA".GLOBAL_DATA.UNIT_01_ST_4_ANY_CYCLE_ACTIVE )
      Not()
      { S7_Templates := "time_type := Time" } "DB2440_GLOBAL_DATA".TIMER_DELAY_ANY_CYCLE_RUN_UNIT_01.TOF(pt := "DB2440_GLOBAL_DATA".TIMER_DELAY_ANY_CYCLE_RUN_UNIT_01.PT, et =>)
      wire#w1
      I_Contact( "DB2440_GLOBAL_DATA".GLOBAL_DATA.ANY_UNIT_01_CYCLE_RUN )
      Coil( "DB2440_GLOBAL_DATA".GLOBAL_DATA.ANY_UNIT_01_CYCLE_RUN_P )
   END_RUNG
   RUNG wire#w1
      Coil( "DB2440_GLOBAL_DATA".GLOBAL_DATA.ANY_UNIT_01_CYCLE_RUN )
   END_RUNG
   // the same network as SCL:
   "DB2440_GLOBAL_DATA".TIMER_DELAY_ANY_CYCLE_RUN_UNIT_01.TOF(IN := NOT (NOT "DB1201_PART_CYCLE_UNIT_1".SEQUENCE.RUNNING AND NOT "DB2440_GLOBAL_DATA".GLOBAL_DATA.UNIT_01_ST_0_ANY_CYCLE_ACTIVE AND NOT "DB2440_GLOBAL_DATA".GLOBAL_DATA.UNIT_01_ST_1_ANY_CYCLE_ACTIVE AND NOT "DB2440_GLOBAL_DATA".GLOBAL_DATA.UNIT_01_ST_2_ANY_CYCLE_ACTIVE AND NOT "DB2440_GLOBAL_DATA".GLOBAL_DATA.UNIT_01_ST_3_ANY_CYCLE_ACTIVE AND NOT "DB2440_GLOBAL_DATA".GLOBAL_DATA.UNIT_01_ST_4_ANY_CYCLE_ACTIVE),
                           PT := "DB2440_GLOBAL_DATA".TIMER_DELAY_ANY_CYCLE_RUN_UNIT_01.PT);
   "DB2440_GLOBAL_DATA".GLOBAL_DATA.ANY_UNIT_01_CYCLE_RUN_P := "DB2440_GLOBAL_DATA".TIMER_DELAY_ANY_CYCLE_RUN_UNIT_01.Q AND NOT "DB2440_GLOBAL_DATA".GLOBAL_DATA.ANY_UNIT_01_CYCLE_RUN;
   "DB2440_GLOBAL_DATA".GLOBAL_DATA.ANY_UNIT_01_CYCLE_RUN := "DB2440_GLOBAL_DATA".TIMER_DELAY_ANY_CYCLE_RUN_UNIT_01.Q;
END_REGION

REGION Network 80: ANY UNIT 02 CYCLE RUNNING
   RUNG wire#powerrail
      I_Contact( "DB1251_PART_CYCLE_UNIT_2".SEQUENCE.RUNNING )
      I_Contact( "DB2440_GLOBAL_DATA".GLOBAL_DATA.UNIT_02_ST_0_ANY_CYCLE_ACTIVE )
      I_Contact( "DB2440_GLOBAL_DATA".GLOBAL_DATA.UNIT_02_ST_1_ANY_CYCLE_ACTIVE )
      I_Contact( "DB2440_GLOBAL_DATA".GLOBAL_DATA.UNIT_02_ST_2_ANY_CYCLE_ACTIVE )
      I_Contact( "DB2440_GLOBAL_DATA".GLOBAL_DATA.UNIT_02_ST_3_ANY_CYCLE_ACTIVE )
      I_Contact( "DB2440_GLOBAL_DATA".GLOBAL_DATA.UNIT_02_ST_4_ANY_CYCLE_ACTIVE )
      Not()
      { S7_Templates := "time_type := Time" } "DB2440_GLOBAL_DATA".TIMER_DELAY_ANY_CYCLE_RUN_UNIT_02.TOF(pt := "DB2440_GLOBAL_DATA".TIMER_DELAY_ANY_CYCLE_RUN_UNIT_02.PT, et =>)
      wire#w1
      I_Contact( "DB2440_GLOBAL_DATA".GLOBAL_DATA.ANY_UNIT_02_CYCLE_RUN )
      Coil( "DB2440_GLOBAL_DATA".GLOBAL_DATA.ANY_UNIT_02_CYCLE_RUN_P )
   END_RUNG
   RUNG wire#w1
      Coil( "DB2440_GLOBAL_DATA".GLOBAL_DATA.ANY_UNIT_02_CYCLE_RUN )
   END_RUNG
   // the same network as SCL:
   "DB2440_GLOBAL_DATA".TIMER_DELAY_ANY_CYCLE_RUN_UNIT_02.TOF(IN := NOT (NOT "DB1251_PART_CYCLE_UNIT_2".SEQUENCE.RUNNING AND NOT "DB2440_GLOBAL_DATA".GLOBAL_DATA.UNIT_02_ST_0_ANY_CYCLE_ACTIVE AND NOT "DB2440_GLOBAL_DATA".GLOBAL_DATA.UNIT_02_ST_1_ANY_CYCLE_ACTIVE AND NOT "DB2440_GLOBAL_DATA".GLOBAL_DATA.UNIT_02_ST_2_ANY_CYCLE_ACTIVE AND NOT "DB2440_GLOBAL_DATA".GLOBAL_DATA.UNIT_02_ST_3_ANY_CYCLE_ACTIVE AND NOT "DB2440_GLOBAL_DATA".GLOBAL_DATA.UNIT_02_ST_4_ANY_CYCLE_ACTIVE),
                           PT := "DB2440_GLOBAL_DATA".TIMER_DELAY_ANY_CYCLE_RUN_UNIT_02.PT);
   "DB2440_GLOBAL_DATA".GLOBAL_DATA.ANY_UNIT_02_CYCLE_RUN_P := "DB2440_GLOBAL_DATA".TIMER_DELAY_ANY_CYCLE_RUN_UNIT_02.Q AND NOT "DB2440_GLOBAL_DATA".GLOBAL_DATA.ANY_UNIT_02_CYCLE_RUN;
   "DB2440_GLOBAL_DATA".GLOBAL_DATA.ANY_UNIT_02_CYCLE_RUN := "DB2440_GLOBAL_DATA".TIMER_DELAY_ANY_CYCLE_RUN_UNIT_02.Q;
END_REGION

REGION Network 81: ANY UNIT 03 CYCLE RUNNING
   RUNG wire#powerrail
      I_Contact( "DB1301_PART_CYCLE_UNIT_3".RUNNING )
      I_Contact( "DB2440_GLOBAL_DATA".GLOBAL_DATA.UNIT_03_ANY_CYCLE_ACTIVE )
      Not()
      { S7_Templates := "time_type := Time" } "DB2440_GLOBAL_DATA".TIMER_DELAY_ANY_CYCLE_RUN_UNIT_03.TOF(pt := "DB2440_GLOBAL_DATA".TIMER_DELAY_ANY_CYCLE_RUN_UNIT_03.PT, et =>)
      wire#w1
      I_Contact( "DB2440_GLOBAL_DATA".GLOBAL_DATA.ANY_UNIT_03_CYCLE_RUN )
      Coil( "DB2440_GLOBAL_DATA".GLOBAL_DATA.ANY_UNIT_03_CYCLE_RUN_P )
   END_RUNG
   RUNG wire#w1
      Coil( "DB2440_GLOBAL_DATA".GLOBAL_DATA.ANY_UNIT_03_CYCLE_RUN )
   END_RUNG
   // the same network as SCL:
   "DB2440_GLOBAL_DATA".TIMER_DELAY_ANY_CYCLE_RUN_UNIT_03.TOF(IN := NOT (NOT "DB1301_PART_CYCLE_UNIT_3".RUNNING AND NOT "DB2440_GLOBAL_DATA".GLOBAL_DATA.UNIT_03_ANY_CYCLE_ACTIVE),
                           PT := "DB2440_GLOBAL_DATA".TIMER_DELAY_ANY_CYCLE_RUN_UNIT_03.PT);
   "DB2440_GLOBAL_DATA".GLOBAL_DATA.ANY_UNIT_03_CYCLE_RUN_P := "DB2440_GLOBAL_DATA".TIMER_DELAY_ANY_CYCLE_RUN_UNIT_03.Q AND NOT "DB2440_GLOBAL_DATA".GLOBAL_DATA.ANY_UNIT_03_CYCLE_RUN;
   "DB2440_GLOBAL_DATA".GLOBAL_DATA.ANY_UNIT_03_CYCLE_RUN := "DB2440_GLOBAL_DATA".TIMER_DELAY_ANY_CYCLE_RUN_UNIT_03.Q;
END_REGION

REGION Network 82: ANY MACHINE CYCLE RUNNING
   RUNG wire#powerrail
      I_Contact( "DB1201_PART_CYCLE_UNIT_1".SEQUENCE.RUNNING )
      I_Contact( "DB1251_PART_CYCLE_UNIT_2".SEQUENCE.RUNNING )
      I_Contact( "DB1301_PART_CYCLE_UNIT_3".RUNNING )
      I_Contact( "DB2440_GLOBAL_DATA".GLOBAL_DATA.UNIT_01_ST_0_ANY_CYCLE_ACTIVE )
      I_Contact( "DB2440_GLOBAL_DATA".GLOBAL_DATA.UNIT_01_ST_1_ANY_CYCLE_ACTIVE )
      I_Contact( "DB2440_GLOBAL_DATA".GLOBAL_DATA.UNIT_01_ST_2_ANY_CYCLE_ACTIVE )
      I_Contact( "DB2440_GLOBAL_DATA".GLOBAL_DATA.UNIT_01_ST_3_ANY_CYCLE_ACTIVE )
      I_Contact( "DB2440_GLOBAL_DATA".GLOBAL_DATA.UNIT_01_ST_4_ANY_CYCLE_ACTIVE )
      I_Contact( "DB2440_GLOBAL_DATA".GLOBAL_DATA.UNIT_02_ST_0_ANY_CYCLE_ACTIVE )
      I_Contact( "DB2440_GLOBAL_DATA".GLOBAL_DATA.UNIT_02_ST_1_ANY_CYCLE_ACTIVE )
      I_Contact( "DB2440_GLOBAL_DATA".GLOBAL_DATA.UNIT_02_ST_2_ANY_CYCLE_ACTIVE )
      I_Contact( "DB2440_GLOBAL_DATA".GLOBAL_DATA.UNIT_02_ST_3_ANY_CYCLE_ACTIVE )
      I_Contact( "DB2440_GLOBAL_DATA".GLOBAL_DATA.UNIT_02_ST_4_ANY_CYCLE_ACTIVE )
      Not()
      { S7_Templates := "time_type := Time" } "DB2440_GLOBAL_DATA".TIMER_DELAY_ANY_CYCLE_RUN.TOF(pt := "DB2440_GLOBAL_DATA".TIMER_DELAY_ANY_CYCLE_RUN.PT, et =>)
      wire#w1
      I_Contact( "DB2440_GLOBAL_DATA".GLOBAL_DATA.ANY_MACHINE_CYCLE_RUN )
      Coil( "DB2440_GLOBAL_DATA".GLOBAL_DATA.ANY_MACHINE_CYCLE_RUN_P )
   END_RUNG
   RUNG wire#w1
      Coil( "DB2440_GLOBAL_DATA".GLOBAL_DATA.ANY_MACHINE_CYCLE_RUN )
   END_RUNG
   // the same network as SCL:
   "DB2440_GLOBAL_DATA".TIMER_DELAY_ANY_CYCLE_RUN.TOF(IN := NOT (NOT "DB1201_PART_CYCLE_UNIT_1".SEQUENCE.RUNNING AND NOT "DB1251_PART_CYCLE_UNIT_2".SEQUENCE.RUNNING AND NOT "DB1301_PART_CYCLE_UNIT_3".RUNNING AND NOT "DB2440_GLOBAL_DATA".GLOBAL_DATA.UNIT_01_ST_0_ANY_CYCLE_ACTIVE AND NOT "DB2440_GLOBAL_DATA".GLOBAL_DATA.UNIT_01_ST_1_ANY_CYCLE_ACTIVE AND NOT "DB2440_GLOBAL_DATA".GLOBAL_DATA.UNIT_01_ST_2_ANY_CYCLE_ACTIVE AND NOT "DB2440_GLOBAL_DATA".GLOBAL_DATA.UNIT_01_ST_3_ANY_CYCLE_ACTIVE AND NOT "DB2440_GLOBAL_DATA".GLOBAL_DATA.UNIT_01_ST_4_ANY_CYCLE_ACTIVE AND NOT "DB2440_GLOBAL_DATA".GLOBAL_DATA.UNIT_02_ST_0_ANY_CYCLE_ACTIVE AND NOT "DB2440_GLOBAL_DATA".GLOBAL_DATA.UNIT_02_ST_1_ANY_CYCLE_ACTIVE AND NOT "DB2440_GLOBAL_DATA".GLOBAL_DATA.UNIT_02_ST_2_ANY_CYCLE_ACTIVE AND NOT "DB2440_GLOBAL_DATA".GLOBAL_DATA.UNIT_02_ST_3_ANY_CYCLE_ACTIVE AND NOT "DB2440_GLOBAL_DATA".GLOBAL_DATA.UNIT_02_ST_4_ANY_CYCLE_ACTIVE),
                           PT := "DB2440_GLOBAL_DATA".TIMER_DELAY_ANY_CYCLE_RUN.PT);
   "DB2440_GLOBAL_DATA".GLOBAL_DATA.ANY_MACHINE_CYCLE_RUN_P := "DB2440_GLOBAL_DATA".TIMER_DELAY_ANY_CYCLE_RUN.Q AND NOT "DB2440_GLOBAL_DATA".GLOBAL_DATA.ANY_MACHINE_CYCLE_RUN;
   "DB2440_GLOBAL_DATA".GLOBAL_DATA.ANY_MACHINE_CYCLE_RUN := "DB2440_GLOBAL_DATA".TIMER_DELAY_ANY_CYCLE_RUN.Q;
END_REGION

REGION Network 83: NO MACHINE CYCLE RUNNING ALL
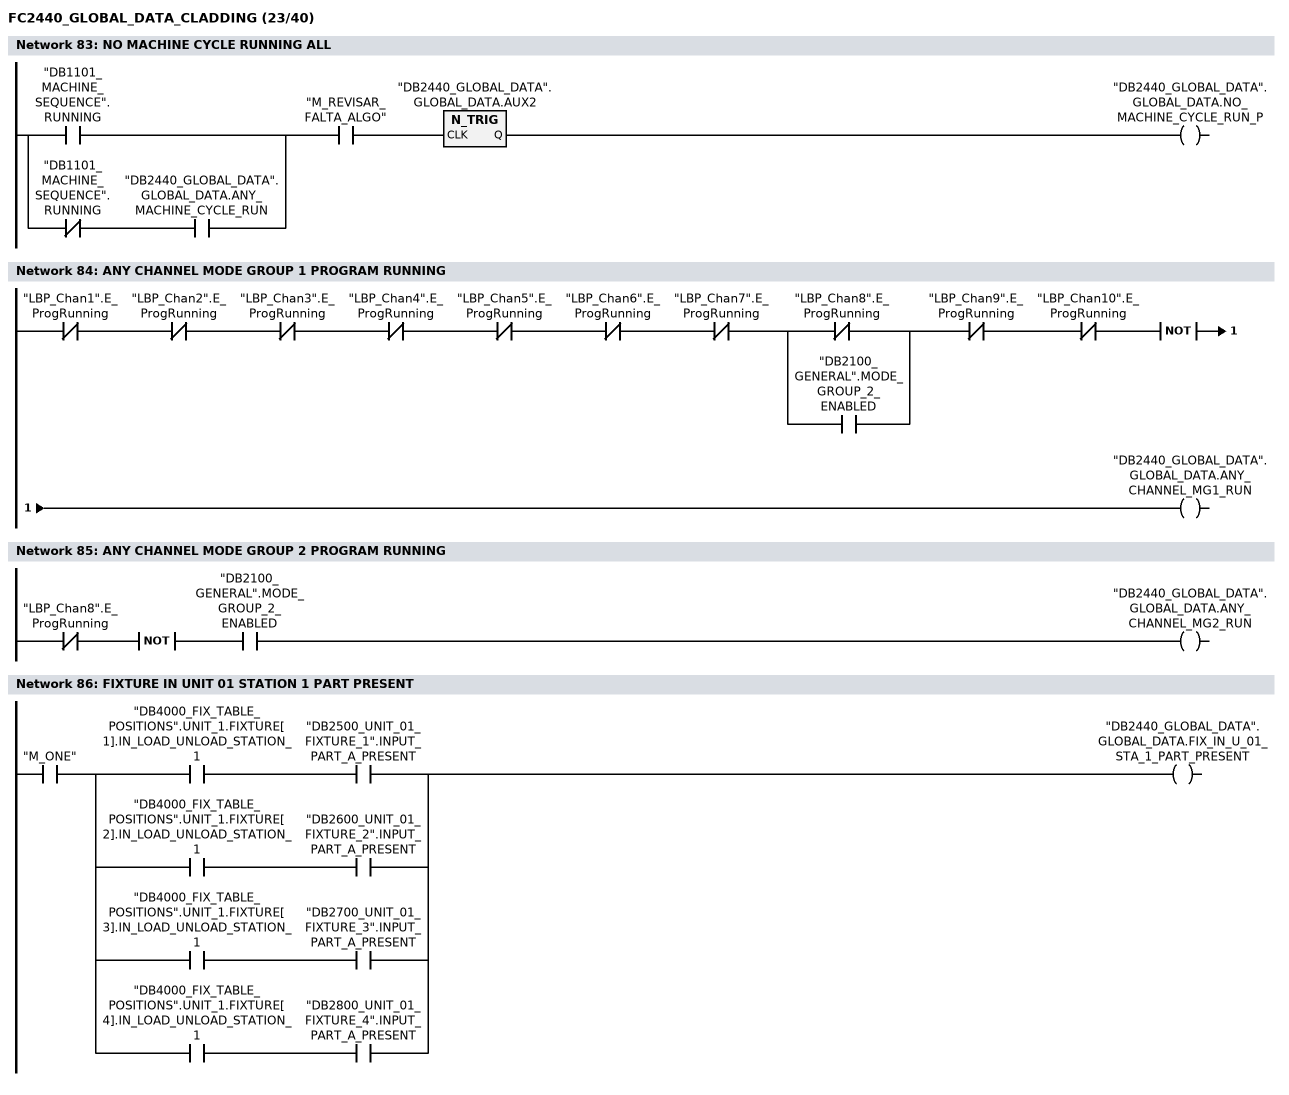
   RUNG wire#powerrail
      Contact( "DB1101_MACHINE_SEQUENCE".RUNNING )
      wire#w1
      Contact( "M_REVISAR_FALTA_ALGO" )
      N_Trig( "DB2440_GLOBAL_DATA".GLOBAL_DATA.AUX2 )
      Coil( "DB2440_GLOBAL_DATA".GLOBAL_DATA.NO_MACHINE_CYCLE_RUN_P )
   END_RUNG
   RUNG wire#powerrail
      I_Contact( "DB1101_MACHINE_SEQUENCE".RUNNING )
      Contact( "DB2440_GLOBAL_DATA".GLOBAL_DATA.ANY_MACHINE_CYCLE_RUN )
   END_RUNG wire#w1
   // the same network as SCL:
   #_w1 := ("DB1101_MACHINE_SEQUENCE".RUNNING OR (NOT "DB1101_MACHINE_SEQUENCE".RUNNING AND "DB2440_GLOBAL_DATA".GLOBAL_DATA.ANY_MACHINE_CYCLE_RUN)) AND "M_REVISAR_FALTA_ALGO";
   #_w2 := NOT #_w1 AND "DB2440_GLOBAL_DATA".GLOBAL_DATA.AUX2;   // falling edge
   "DB2440_GLOBAL_DATA".GLOBAL_DATA.AUX2 := #_w1;
   "DB2440_GLOBAL_DATA".GLOBAL_DATA.NO_MACHINE_CYCLE_RUN_P := #_w2;
END_REGION

REGION Network 84: ANY CHANNEL MODE GROUP 1 PROGRAM RUNNING
   RUNG wire#powerrail
      I_Contact( "LBP_Chan1".E_ProgRunning )
      I_Contact( "LBP_Chan2".E_ProgRunning )
      I_Contact( "LBP_Chan3".E_ProgRunning )
      I_Contact( "LBP_Chan4".E_ProgRunning )
      I_Contact( "LBP_Chan5".E_ProgRunning )
      I_Contact( "LBP_Chan6".E_ProgRunning )
      I_Contact( "LBP_Chan7".E_ProgRunning )
      wire#w1
      I_Contact( "LBP_Chan8".E_ProgRunning )
      wire#w2
      I_Contact( "LBP_Chan9".E_ProgRunning )
      I_Contact( "LBP_Chan10".E_ProgRunning )
      Not()
      Coil( "DB2440_GLOBAL_DATA".GLOBAL_DATA.ANY_CHANNEL_MG1_RUN )
   END_RUNG
   RUNG wire#w1
      Contact( "DB2100_GENERAL".MODE_GROUP_2_ENABLED )
   END_RUNG wire#w2
   // the same network as SCL:
   "DB2440_GLOBAL_DATA".GLOBAL_DATA.ANY_CHANNEL_MG1_RUN := NOT (NOT "LBP_Chan1".E_ProgRunning AND NOT "LBP_Chan2".E_ProgRunning AND NOT "LBP_Chan3".E_ProgRunning AND NOT "LBP_Chan4".E_ProgRunning AND NOT "LBP_Chan5".E_ProgRunning AND NOT "LBP_Chan6".E_ProgRunning AND NOT "LBP_Chan7".E_ProgRunning AND (NOT "LBP_Chan8".E_ProgRunning OR "DB2100_GENERAL".MODE_GROUP_2_ENABLED) AND NOT "LBP_Chan9".E_ProgRunning AND NOT "LBP_Chan10".E_ProgRunning);
END_REGION

REGION Network 85: ANY CHANNEL MODE GROUP 2 PROGRAM RUNNING
   RUNG wire#powerrail
      I_Contact( "LBP_Chan8".E_ProgRunning )
      Not()
      Contact( "DB2100_GENERAL".MODE_GROUP_2_ENABLED )
      Coil( "DB2440_GLOBAL_DATA".GLOBAL_DATA.ANY_CHANNEL_MG2_RUN )
   END_RUNG
   // the same network as SCL:
   "DB2440_GLOBAL_DATA".GLOBAL_DATA.ANY_CHANNEL_MG2_RUN := NOT (NOT "LBP_Chan8".E_ProgRunning) AND "DB2100_GENERAL".MODE_GROUP_2_ENABLED;
END_REGION

REGION Network 86: FIXTURE IN UNIT 01 STATION 1 PART PRESENT
   RUNG wire#powerrail
      Contact( "M_ONE" )
      wire#w1
      Contact( "DB4000_FIX_TABLE_POSITIONS".UNIT_1.FIXTURE[1].IN_LOAD_UNLOAD_STATION_1 )
      Contact( "DB2500_UNIT_01_FIXTURE_1".INPUT_PART_A_PRESENT )
      wire#w2
      Coil( "DB2440_GLOBAL_DATA".GLOBAL_DATA.FIX_IN_U_01_STA_1_PART_PRESENT )
   END_RUNG
   RUNG wire#w1
      Contact( "DB4000_FIX_TABLE_POSITIONS".UNIT_1.FIXTURE[2].IN_LOAD_UNLOAD_STATION_1 )
      Contact( "DB2600_UNIT_01_FIXTURE_2".INPUT_PART_A_PRESENT )
   END_RUNG wire#w2
   RUNG wire#w1
      Contact( "DB4000_FIX_TABLE_POSITIONS".UNIT_1.FIXTURE[3].IN_LOAD_UNLOAD_STATION_1 )
      Contact( "DB2700_UNIT_01_FIXTURE_3".INPUT_PART_A_PRESENT )
   END_RUNG wire#w2
   RUNG wire#w1
      Contact( "DB4000_FIX_TABLE_POSITIONS".UNIT_1.FIXTURE[4].IN_LOAD_UNLOAD_STATION_1 )
      Contact( "DB2800_UNIT_01_FIXTURE_4".INPUT_PART_A_PRESENT )
   END_RUNG wire#w2
   // the same network as SCL:
   "DB2440_GLOBAL_DATA".GLOBAL_DATA.FIX_IN_U_01_STA_1_PART_PRESENT := "M_ONE" AND (("DB4000_FIX_TABLE_POSITIONS".UNIT_1.FIXTURE[1].IN_LOAD_UNLOAD_STATION_1 AND "DB2500_UNIT_01_FIXTURE_1".INPUT_PART_A_PRESENT) OR ("DB4000_FIX_TABLE_POSITIONS".UNIT_1.FIXTURE[2].IN_LOAD_UNLOAD_STATION_1 AND "DB2600_UNIT_01_FIXTURE_2".INPUT_PART_A_PRESENT) OR ("DB4000_FIX_TABLE_POSITIONS".UNIT_1.FIXTURE[3].IN_LOAD_UNLOAD_STATION_1 AND "DB2700_UNIT_01_FIXTURE_3".INPUT_PART_A_PRESENT) OR ("DB4000_FIX_TABLE_POSITIONS".UNIT_1.FIXTURE[4].IN_LOAD_UNLOAD_STATION_1 AND "DB2800_UNIT_01_FIXTURE_4".INPUT_PART_A_PRESENT));
END_REGION

REGION Network 87: FIXTURE IN UNIT 01 STATION 2 PART PRESENT
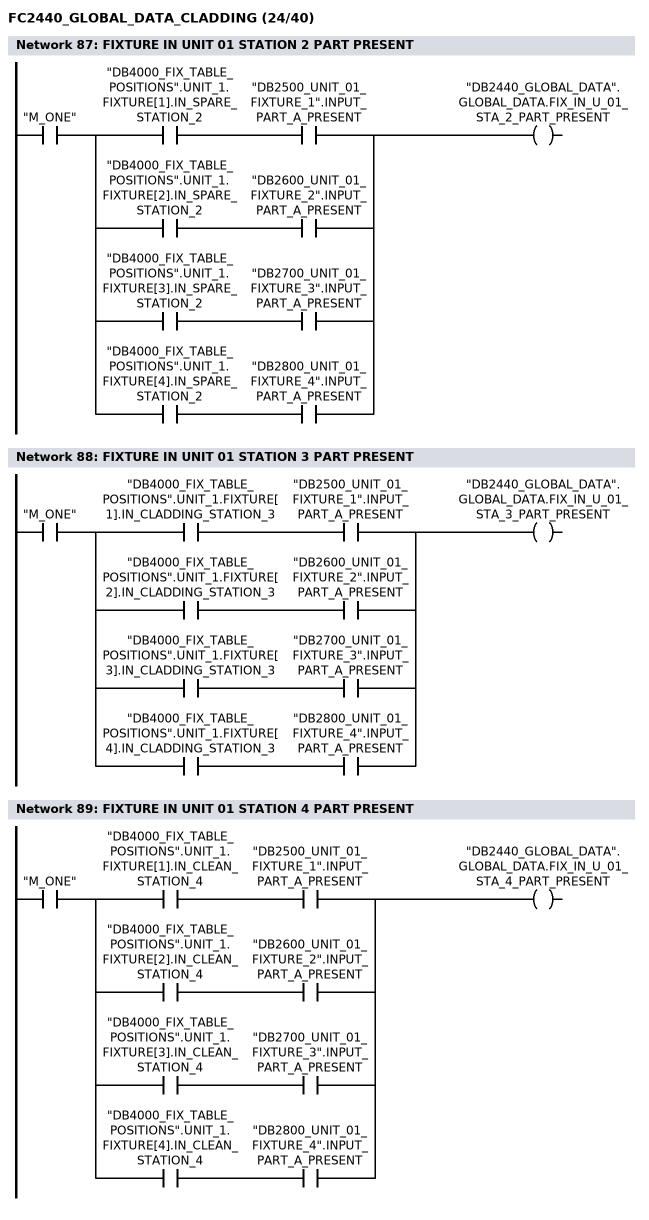
   RUNG wire#powerrail
      Contact( "M_ONE" )
      wire#w1
      Contact( "DB4000_FIX_TABLE_POSITIONS".UNIT_1.FIXTURE[1].IN_SPARE_STATION_2 )
      Contact( "DB2500_UNIT_01_FIXTURE_1".INPUT_PART_A_PRESENT )
      wire#w2
      Coil( "DB2440_GLOBAL_DATA".GLOBAL_DATA.FIX_IN_U_01_STA_2_PART_PRESENT )
   END_RUNG
   RUNG wire#w1
      Contact( "DB4000_FIX_TABLE_POSITIONS".UNIT_1.FIXTURE[2].IN_SPARE_STATION_2 )
      Contact( "DB2600_UNIT_01_FIXTURE_2".INPUT_PART_A_PRESENT )
   END_RUNG wire#w2
   RUNG wire#w1
      Contact( "DB4000_FIX_TABLE_POSITIONS".UNIT_1.FIXTURE[3].IN_SPARE_STATION_2 )
      Contact( "DB2700_UNIT_01_FIXTURE_3".INPUT_PART_A_PRESENT )
   END_RUNG wire#w2
   RUNG wire#w1
      Contact( "DB4000_FIX_TABLE_POSITIONS".UNIT_1.FIXTURE[4].IN_SPARE_STATION_2 )
      Contact( "DB2800_UNIT_01_FIXTURE_4".INPUT_PART_A_PRESENT )
   END_RUNG wire#w2
   // the same network as SCL:
   "DB2440_GLOBAL_DATA".GLOBAL_DATA.FIX_IN_U_01_STA_2_PART_PRESENT := "M_ONE" AND (("DB4000_FIX_TABLE_POSITIONS".UNIT_1.FIXTURE[1].IN_SPARE_STATION_2 AND "DB2500_UNIT_01_FIXTURE_1".INPUT_PART_A_PRESENT) OR ("DB4000_FIX_TABLE_POSITIONS".UNIT_1.FIXTURE[2].IN_SPARE_STATION_2 AND "DB2600_UNIT_01_FIXTURE_2".INPUT_PART_A_PRESENT) OR ("DB4000_FIX_TABLE_POSITIONS".UNIT_1.FIXTURE[3].IN_SPARE_STATION_2 AND "DB2700_UNIT_01_FIXTURE_3".INPUT_PART_A_PRESENT) OR ("DB4000_FIX_TABLE_POSITIONS".UNIT_1.FIXTURE[4].IN_SPARE_STATION_2 AND "DB2800_UNIT_01_FIXTURE_4".INPUT_PART_A_PRESENT));
END_REGION

REGION Network 88: FIXTURE IN UNIT 01 STATION 3 PART PRESENT
   RUNG wire#powerrail
      Contact( "M_ONE" )
      wire#w1
      Contact( "DB4000_FIX_TABLE_POSITIONS".UNIT_1.FIXTURE[1].IN_CLADDING_STATION_3 )
      Contact( "DB2500_UNIT_01_FIXTURE_1".INPUT_PART_A_PRESENT )
      wire#w2
      Coil( "DB2440_GLOBAL_DATA".GLOBAL_DATA.FIX_IN_U_01_STA_3_PART_PRESENT )
   END_RUNG
   RUNG wire#w1
      Contact( "DB4000_FIX_TABLE_POSITIONS".UNIT_1.FIXTURE[2].IN_CLADDING_STATION_3 )
      Contact( "DB2600_UNIT_01_FIXTURE_2".INPUT_PART_A_PRESENT )
   END_RUNG wire#w2
   RUNG wire#w1
      Contact( "DB4000_FIX_TABLE_POSITIONS".UNIT_1.FIXTURE[3].IN_CLADDING_STATION_3 )
      Contact( "DB2700_UNIT_01_FIXTURE_3".INPUT_PART_A_PRESENT )
   END_RUNG wire#w2
   RUNG wire#w1
      Contact( "DB4000_FIX_TABLE_POSITIONS".UNIT_1.FIXTURE[4].IN_CLADDING_STATION_3 )
      Contact( "DB2800_UNIT_01_FIXTURE_4".INPUT_PART_A_PRESENT )
   END_RUNG wire#w2
   // the same network as SCL:
   "DB2440_GLOBAL_DATA".GLOBAL_DATA.FIX_IN_U_01_STA_3_PART_PRESENT := "M_ONE" AND (("DB4000_FIX_TABLE_POSITIONS".UNIT_1.FIXTURE[1].IN_CLADDING_STATION_3 AND "DB2500_UNIT_01_FIXTURE_1".INPUT_PART_A_PRESENT) OR ("DB4000_FIX_TABLE_POSITIONS".UNIT_1.FIXTURE[2].IN_CLADDING_STATION_3 AND "DB2600_UNIT_01_FIXTURE_2".INPUT_PART_A_PRESENT) OR ("DB4000_FIX_TABLE_POSITIONS".UNIT_1.FIXTURE[3].IN_CLADDING_STATION_3 AND "DB2700_UNIT_01_FIXTURE_3".INPUT_PART_A_PRESENT) OR ("DB4000_FIX_TABLE_POSITIONS".UNIT_1.FIXTURE[4].IN_CLADDING_STATION_3 AND "DB2800_UNIT_01_FIXTURE_4".INPUT_PART_A_PRESENT));
END_REGION

REGION Network 89: FIXTURE IN UNIT 01 STATION 4 PART PRESENT
   RUNG wire#powerrail
      Contact( "M_ONE" )
      wire#w1
      Contact( "DB4000_FIX_TABLE_POSITIONS".UNIT_1.FIXTURE[1].IN_CLEAN_STATION_4 )
      Contact( "DB2500_UNIT_01_FIXTURE_1".INPUT_PART_A_PRESENT )
      wire#w2
      Coil( "DB2440_GLOBAL_DATA".GLOBAL_DATA.FIX_IN_U_01_STA_4_PART_PRESENT )
   END_RUNG
   RUNG wire#w1
      Contact( "DB4000_FIX_TABLE_POSITIONS".UNIT_1.FIXTURE[2].IN_CLEAN_STATION_4 )
      Contact( "DB2600_UNIT_01_FIXTURE_2".INPUT_PART_A_PRESENT )
   END_RUNG wire#w2
   RUNG wire#w1
      Contact( "DB4000_FIX_TABLE_POSITIONS".UNIT_1.FIXTURE[3].IN_CLEAN_STATION_4 )
      Contact( "DB2700_UNIT_01_FIXTURE_3".INPUT_PART_A_PRESENT )
   END_RUNG wire#w2
   RUNG wire#w1
      Contact( "DB4000_FIX_TABLE_POSITIONS".UNIT_1.FIXTURE[4].IN_CLEAN_STATION_4 )
      Contact( "DB2800_UNIT_01_FIXTURE_4".INPUT_PART_A_PRESENT )
   END_RUNG wire#w2
   // the same network as SCL:
   "DB2440_GLOBAL_DATA".GLOBAL_DATA.FIX_IN_U_01_STA_4_PART_PRESENT := "M_ONE" AND (("DB4000_FIX_TABLE_POSITIONS".UNIT_1.FIXTURE[1].IN_CLEAN_STATION_4 AND "DB2500_UNIT_01_FIXTURE_1".INPUT_PART_A_PRESENT) OR ("DB4000_FIX_TABLE_POSITIONS".UNIT_1.FIXTURE[2].IN_CLEAN_STATION_4 AND "DB2600_UNIT_01_FIXTURE_2".INPUT_PART_A_PRESENT) OR ("DB4000_FIX_TABLE_POSITIONS".UNIT_1.FIXTURE[3].IN_CLEAN_STATION_4 AND "DB2700_UNIT_01_FIXTURE_3".INPUT_PART_A_PRESENT) OR ("DB4000_FIX_TABLE_POSITIONS".UNIT_1.FIXTURE[4].IN_CLEAN_STATION_4 AND "DB2800_UNIT_01_FIXTURE_4".INPUT_PART_A_PRESENT));
END_REGION

REGION Network 90: FIXTURE IN UNIT 02 STATION 1 PART PRESENT
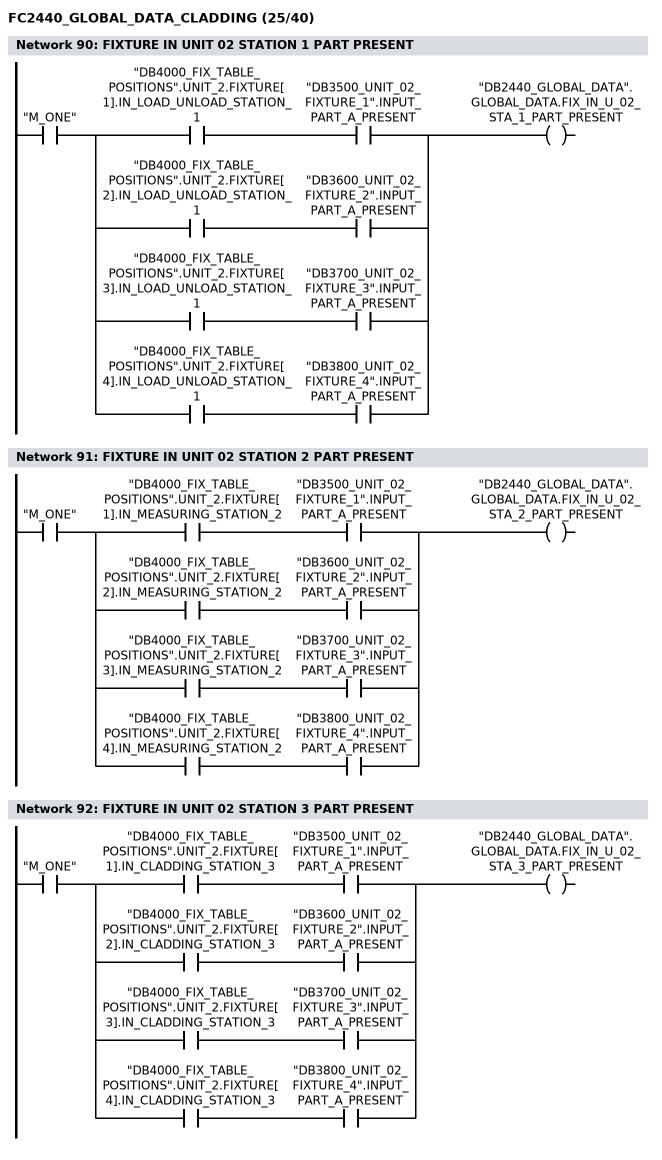
   RUNG wire#powerrail
      Contact( "M_ONE" )
      wire#w1
      Contact( "DB4000_FIX_TABLE_POSITIONS".UNIT_2.FIXTURE[1].IN_LOAD_UNLOAD_STATION_1 )
      Contact( "DB3500_UNIT_02_FIXTURE_1".INPUT_PART_A_PRESENT )
      wire#w2
      Coil( "DB2440_GLOBAL_DATA".GLOBAL_DATA.FIX_IN_U_02_STA_1_PART_PRESENT )
   END_RUNG
   RUNG wire#w1
      Contact( "DB4000_FIX_TABLE_POSITIONS".UNIT_2.FIXTURE[2].IN_LOAD_UNLOAD_STATION_1 )
      Contact( "DB3600_UNIT_02_FIXTURE_2".INPUT_PART_A_PRESENT )
   END_RUNG wire#w2
   RUNG wire#w1
      Contact( "DB4000_FIX_TABLE_POSITIONS".UNIT_2.FIXTURE[3].IN_LOAD_UNLOAD_STATION_1 )
      Contact( "DB3700_UNIT_02_FIXTURE_3".INPUT_PART_A_PRESENT )
   END_RUNG wire#w2
   RUNG wire#w1
      Contact( "DB4000_FIX_TABLE_POSITIONS".UNIT_2.FIXTURE[4].IN_LOAD_UNLOAD_STATION_1 )
      Contact( "DB3800_UNIT_02_FIXTURE_4".INPUT_PART_A_PRESENT )
   END_RUNG wire#w2
   // the same network as SCL:
   "DB2440_GLOBAL_DATA".GLOBAL_DATA.FIX_IN_U_02_STA_1_PART_PRESENT := "M_ONE" AND (("DB4000_FIX_TABLE_POSITIONS".UNIT_2.FIXTURE[1].IN_LOAD_UNLOAD_STATION_1 AND "DB3500_UNIT_02_FIXTURE_1".INPUT_PART_A_PRESENT) OR ("DB4000_FIX_TABLE_POSITIONS".UNIT_2.FIXTURE[2].IN_LOAD_UNLOAD_STATION_1 AND "DB3600_UNIT_02_FIXTURE_2".INPUT_PART_A_PRESENT) OR ("DB4000_FIX_TABLE_POSITIONS".UNIT_2.FIXTURE[3].IN_LOAD_UNLOAD_STATION_1 AND "DB3700_UNIT_02_FIXTURE_3".INPUT_PART_A_PRESENT) OR ("DB4000_FIX_TABLE_POSITIONS".UNIT_2.FIXTURE[4].IN_LOAD_UNLOAD_STATION_1 AND "DB3800_UNIT_02_FIXTURE_4".INPUT_PART_A_PRESENT));
END_REGION

REGION Network 91: FIXTURE IN UNIT 02 STATION 2 PART PRESENT
   RUNG wire#powerrail
      Contact( "M_ONE" )
      wire#w1
      Contact( "DB4000_FIX_TABLE_POSITIONS".UNIT_2.FIXTURE[1].IN_MEASURING_STATION_2 )
      Contact( "DB3500_UNIT_02_FIXTURE_1".INPUT_PART_A_PRESENT )
      wire#w2
      Coil( "DB2440_GLOBAL_DATA".GLOBAL_DATA.FIX_IN_U_02_STA_2_PART_PRESENT )
   END_RUNG
   RUNG wire#w1
      Contact( "DB4000_FIX_TABLE_POSITIONS".UNIT_2.FIXTURE[2].IN_MEASURING_STATION_2 )
      Contact( "DB3600_UNIT_02_FIXTURE_2".INPUT_PART_A_PRESENT )
   END_RUNG wire#w2
   RUNG wire#w1
      Contact( "DB4000_FIX_TABLE_POSITIONS".UNIT_2.FIXTURE[3].IN_MEASURING_STATION_2 )
      Contact( "DB3700_UNIT_02_FIXTURE_3".INPUT_PART_A_PRESENT )
   END_RUNG wire#w2
   RUNG wire#w1
      Contact( "DB4000_FIX_TABLE_POSITIONS".UNIT_2.FIXTURE[4].IN_MEASURING_STATION_2 )
      Contact( "DB3800_UNIT_02_FIXTURE_4".INPUT_PART_A_PRESENT )
   END_RUNG wire#w2
   // the same network as SCL:
   "DB2440_GLOBAL_DATA".GLOBAL_DATA.FIX_IN_U_02_STA_2_PART_PRESENT := "M_ONE" AND (("DB4000_FIX_TABLE_POSITIONS".UNIT_2.FIXTURE[1].IN_MEASURING_STATION_2 AND "DB3500_UNIT_02_FIXTURE_1".INPUT_PART_A_PRESENT) OR ("DB4000_FIX_TABLE_POSITIONS".UNIT_2.FIXTURE[2].IN_MEASURING_STATION_2 AND "DB3600_UNIT_02_FIXTURE_2".INPUT_PART_A_PRESENT) OR ("DB4000_FIX_TABLE_POSITIONS".UNIT_2.FIXTURE[3].IN_MEASURING_STATION_2 AND "DB3700_UNIT_02_FIXTURE_3".INPUT_PART_A_PRESENT) OR ("DB4000_FIX_TABLE_POSITIONS".UNIT_2.FIXTURE[4].IN_MEASURING_STATION_2 AND "DB3800_UNIT_02_FIXTURE_4".INPUT_PART_A_PRESENT));
END_REGION

REGION Network 92: FIXTURE IN UNIT 02 STATION 3 PART PRESENT
   RUNG wire#powerrail
      Contact( "M_ONE" )
      wire#w1
      Contact( "DB4000_FIX_TABLE_POSITIONS".UNIT_2.FIXTURE[1].IN_CLADDING_STATION_3 )
      Contact( "DB3500_UNIT_02_FIXTURE_1".INPUT_PART_A_PRESENT )
      wire#w2
      Coil( "DB2440_GLOBAL_DATA".GLOBAL_DATA.FIX_IN_U_02_STA_3_PART_PRESENT )
   END_RUNG
   RUNG wire#w1
      Contact( "DB4000_FIX_TABLE_POSITIONS".UNIT_2.FIXTURE[2].IN_CLADDING_STATION_3 )
      Contact( "DB3600_UNIT_02_FIXTURE_2".INPUT_PART_A_PRESENT )
   END_RUNG wire#w2
   RUNG wire#w1
      Contact( "DB4000_FIX_TABLE_POSITIONS".UNIT_2.FIXTURE[3].IN_CLADDING_STATION_3 )
      Contact( "DB3700_UNIT_02_FIXTURE_3".INPUT_PART_A_PRESENT )
   END_RUNG wire#w2
   RUNG wire#w1
      Contact( "DB4000_FIX_TABLE_POSITIONS".UNIT_2.FIXTURE[4].IN_CLADDING_STATION_3 )
      Contact( "DB3800_UNIT_02_FIXTURE_4".INPUT_PART_A_PRESENT )
   END_RUNG wire#w2
   // the same network as SCL:
   "DB2440_GLOBAL_DATA".GLOBAL_DATA.FIX_IN_U_02_STA_3_PART_PRESENT := "M_ONE" AND (("DB4000_FIX_TABLE_POSITIONS".UNIT_2.FIXTURE[1].IN_CLADDING_STATION_3 AND "DB3500_UNIT_02_FIXTURE_1".INPUT_PART_A_PRESENT) OR ("DB4000_FIX_TABLE_POSITIONS".UNIT_2.FIXTURE[2].IN_CLADDING_STATION_3 AND "DB3600_UNIT_02_FIXTURE_2".INPUT_PART_A_PRESENT) OR ("DB4000_FIX_TABLE_POSITIONS".UNIT_2.FIXTURE[3].IN_CLADDING_STATION_3 AND "DB3700_UNIT_02_FIXTURE_3".INPUT_PART_A_PRESENT) OR ("DB4000_FIX_TABLE_POSITIONS".UNIT_2.FIXTURE[4].IN_CLADDING_STATION_3 AND "DB3800_UNIT_02_FIXTURE_4".INPUT_PART_A_PRESENT));
END_REGION

REGION Network 93: FIXTURE IN UNIT 02 STATION 4 PART PRESENT
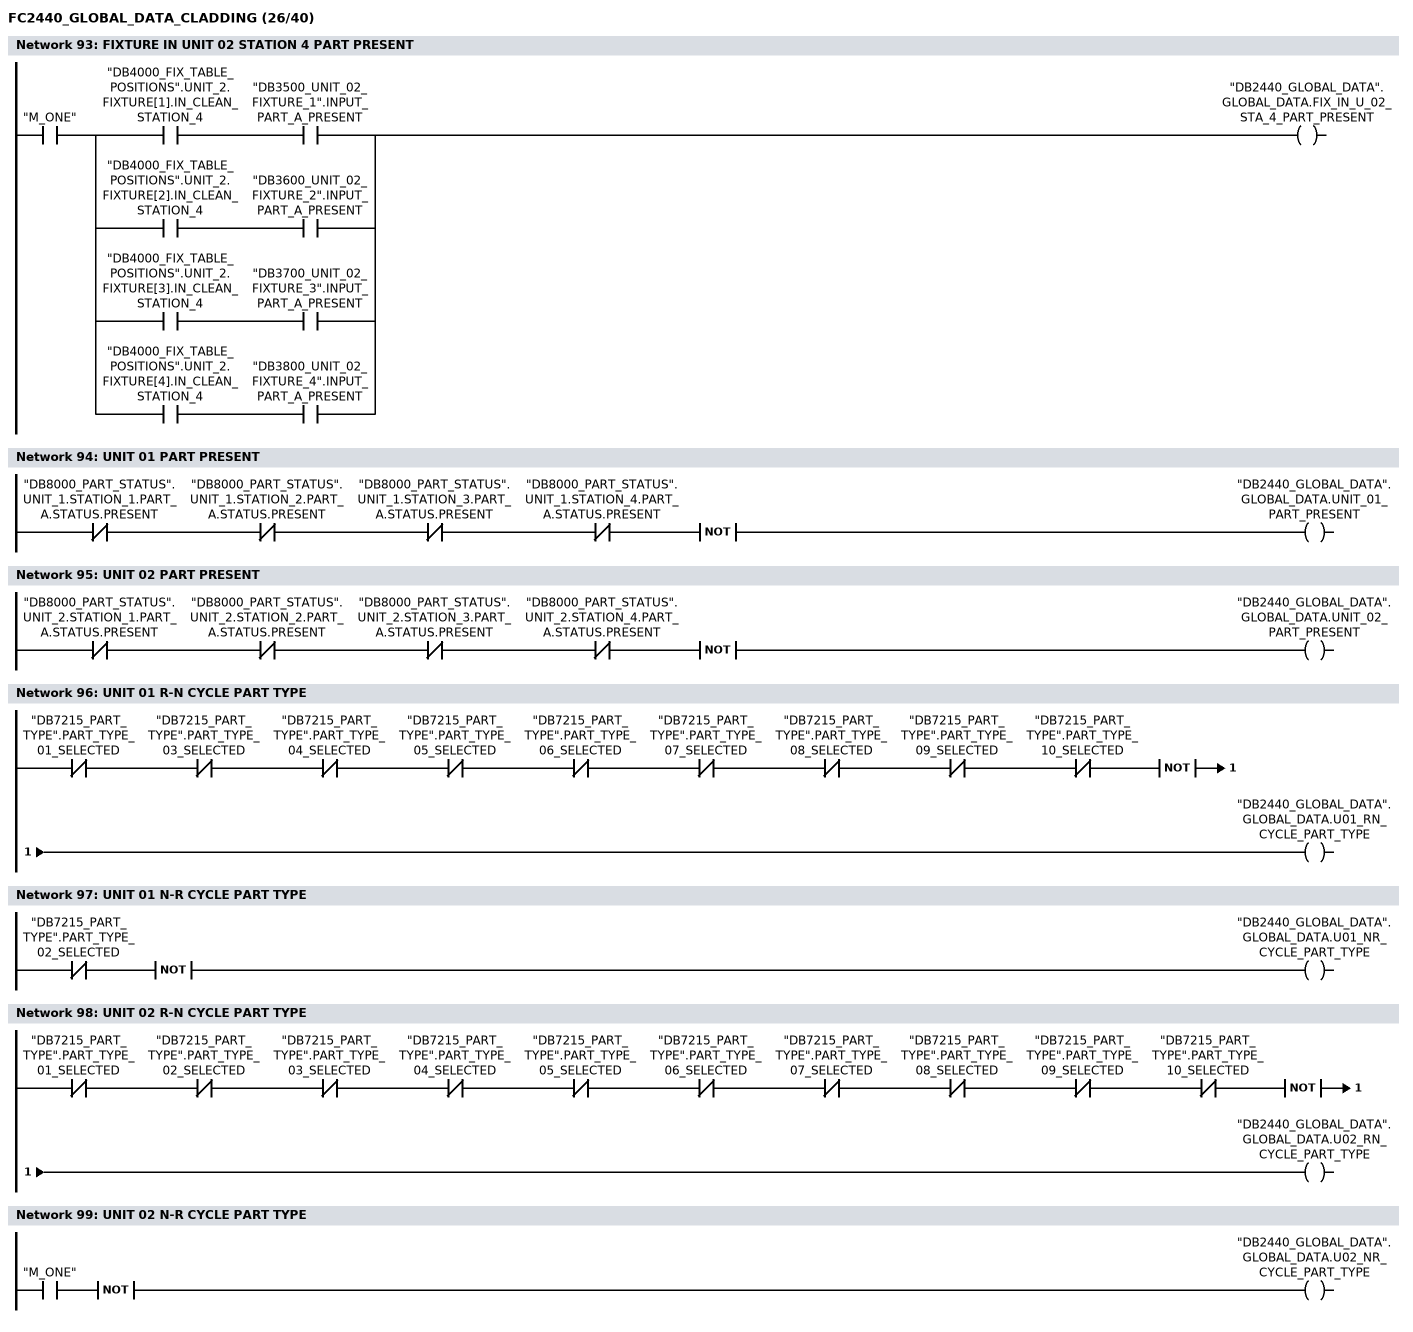
   RUNG wire#powerrail
      Contact( "M_ONE" )
      wire#w1
      Contact( "DB4000_FIX_TABLE_POSITIONS".UNIT_2.FIXTURE[1].IN_CLEAN_STATION_4 )
      Contact( "DB3500_UNIT_02_FIXTURE_1".INPUT_PART_A_PRESENT )
      wire#w2
      Coil( "DB2440_GLOBAL_DATA".GLOBAL_DATA.FIX_IN_U_02_STA_4_PART_PRESENT )
   END_RUNG
   RUNG wire#w1
      Contact( "DB4000_FIX_TABLE_POSITIONS".UNIT_2.FIXTURE[2].IN_CLEAN_STATION_4 )
      Contact( "DB3600_UNIT_02_FIXTURE_2".INPUT_PART_A_PRESENT )
   END_RUNG wire#w2
   RUNG wire#w1
      Contact( "DB4000_FIX_TABLE_POSITIONS".UNIT_2.FIXTURE[3].IN_CLEAN_STATION_4 )
      Contact( "DB3700_UNIT_02_FIXTURE_3".INPUT_PART_A_PRESENT )
   END_RUNG wire#w2
   RUNG wire#w1
      Contact( "DB4000_FIX_TABLE_POSITIONS".UNIT_2.FIXTURE[4].IN_CLEAN_STATION_4 )
      Contact( "DB3800_UNIT_02_FIXTURE_4".INPUT_PART_A_PRESENT )
   END_RUNG wire#w2
   // the same network as SCL:
   "DB2440_GLOBAL_DATA".GLOBAL_DATA.FIX_IN_U_02_STA_4_PART_PRESENT := "M_ONE" AND (("DB4000_FIX_TABLE_POSITIONS".UNIT_2.FIXTURE[1].IN_CLEAN_STATION_4 AND "DB3500_UNIT_02_FIXTURE_1".INPUT_PART_A_PRESENT) OR ("DB4000_FIX_TABLE_POSITIONS".UNIT_2.FIXTURE[2].IN_CLEAN_STATION_4 AND "DB3600_UNIT_02_FIXTURE_2".INPUT_PART_A_PRESENT) OR ("DB4000_FIX_TABLE_POSITIONS".UNIT_2.FIXTURE[3].IN_CLEAN_STATION_4 AND "DB3700_UNIT_02_FIXTURE_3".INPUT_PART_A_PRESENT) OR ("DB4000_FIX_TABLE_POSITIONS".UNIT_2.FIXTURE[4].IN_CLEAN_STATION_4 AND "DB3800_UNIT_02_FIXTURE_4".INPUT_PART_A_PRESENT));
END_REGION

REGION Network 94: UNIT 01 PART PRESENT
   RUNG wire#powerrail
      I_Contact( "DB8000_PART_STATUS".UNIT_1.STATION_1.PART_A.STATUS.PRESENT )
      I_Contact( "DB8000_PART_STATUS".UNIT_1.STATION_2.PART_A.STATUS.PRESENT )
      I_Contact( "DB8000_PART_STATUS".UNIT_1.STATION_3.PART_A.STATUS.PRESENT )
      I_Contact( "DB8000_PART_STATUS".UNIT_1.STATION_4.PART_A.STATUS.PRESENT )
      Not()
      Coil( "DB2440_GLOBAL_DATA".GLOBAL_DATA.UNIT_01_PART_PRESENT )
   END_RUNG
   // the same network as SCL:
   "DB2440_GLOBAL_DATA".GLOBAL_DATA.UNIT_01_PART_PRESENT := NOT (NOT "DB8000_PART_STATUS".UNIT_1.STATION_1.PART_A.STATUS.PRESENT AND NOT "DB8000_PART_STATUS".UNIT_1.STATION_2.PART_A.STATUS.PRESENT AND NOT "DB8000_PART_STATUS".UNIT_1.STATION_3.PART_A.STATUS.PRESENT AND NOT "DB8000_PART_STATUS".UNIT_1.STATION_4.PART_A.STATUS.PRESENT);
END_REGION

REGION Network 95: UNIT 02 PART PRESENT
   RUNG wire#powerrail
      I_Contact( "DB8000_PART_STATUS".UNIT_2.STATION_1.PART_A.STATUS.PRESENT )
      I_Contact( "DB8000_PART_STATUS".UNIT_2.STATION_2.PART_A.STATUS.PRESENT )
      I_Contact( "DB8000_PART_STATUS".UNIT_2.STATION_3.PART_A.STATUS.PRESENT )
      I_Contact( "DB8000_PART_STATUS".UNIT_2.STATION_4.PART_A.STATUS.PRESENT )
      Not()
      Coil( "DB2440_GLOBAL_DATA".GLOBAL_DATA.UNIT_02_PART_PRESENT )
   END_RUNG
   // the same network as SCL:
   "DB2440_GLOBAL_DATA".GLOBAL_DATA.UNIT_02_PART_PRESENT := NOT (NOT "DB8000_PART_STATUS".UNIT_2.STATION_1.PART_A.STATUS.PRESENT AND NOT "DB8000_PART_STATUS".UNIT_2.STATION_2.PART_A.STATUS.PRESENT AND NOT "DB8000_PART_STATUS".UNIT_2.STATION_3.PART_A.STATUS.PRESENT AND NOT "DB8000_PART_STATUS".UNIT_2.STATION_4.PART_A.STATUS.PRESENT);
END_REGION

REGION Network 96: UNIT 01 R-N CYCLE PART TYPE
   RUNG wire#powerrail
      I_Contact( "DB7215_PART_TYPE".PART_TYPE_01_SELECTED )
      I_Contact( "DB7215_PART_TYPE".PART_TYPE_03_SELECTED )
      I_Contact( "DB7215_PART_TYPE".PART_TYPE_04_SELECTED )
      I_Contact( "DB7215_PART_TYPE".PART_TYPE_05_SELECTED )
      I_Contact( "DB7215_PART_TYPE".PART_TYPE_06_SELECTED )
      I_Contact( "DB7215_PART_TYPE".PART_TYPE_07_SELECTED )
      I_Contact( "DB7215_PART_TYPE".PART_TYPE_08_SELECTED )
      I_Contact( "DB7215_PART_TYPE".PART_TYPE_09_SELECTED )
      I_Contact( "DB7215_PART_TYPE".PART_TYPE_10_SELECTED )
      Not()
      Coil( "DB2440_GLOBAL_DATA".GLOBAL_DATA.U01_RN_CYCLE_PART_TYPE )
   END_RUNG
   // the same network as SCL:
   "DB2440_GLOBAL_DATA".GLOBAL_DATA.U01_RN_CYCLE_PART_TYPE := NOT (NOT "DB7215_PART_TYPE".PART_TYPE_01_SELECTED AND NOT "DB7215_PART_TYPE".PART_TYPE_03_SELECTED AND NOT "DB7215_PART_TYPE".PART_TYPE_04_SELECTED AND NOT "DB7215_PART_TYPE".PART_TYPE_05_SELECTED AND NOT "DB7215_PART_TYPE".PART_TYPE_06_SELECTED AND NOT "DB7215_PART_TYPE".PART_TYPE_07_SELECTED AND NOT "DB7215_PART_TYPE".PART_TYPE_08_SELECTED AND NOT "DB7215_PART_TYPE".PART_TYPE_09_SELECTED AND NOT "DB7215_PART_TYPE".PART_TYPE_10_SELECTED);
END_REGION

REGION Network 97: UNIT 01 N-R CYCLE PART TYPE
   RUNG wire#powerrail
      I_Contact( "DB7215_PART_TYPE".PART_TYPE_02_SELECTED )
      Not()
      Coil( "DB2440_GLOBAL_DATA".GLOBAL_DATA.U01_NR_CYCLE_PART_TYPE )
   END_RUNG
   // the same network as SCL:
   "DB2440_GLOBAL_DATA".GLOBAL_DATA.U01_NR_CYCLE_PART_TYPE := NOT (NOT "DB7215_PART_TYPE".PART_TYPE_02_SELECTED);
END_REGION

REGION Network 98: UNIT 02 R-N CYCLE PART TYPE
   RUNG wire#powerrail
      I_Contact( "DB7215_PART_TYPE".PART_TYPE_01_SELECTED )
      I_Contact( "DB7215_PART_TYPE".PART_TYPE_02_SELECTED )
      I_Contact( "DB7215_PART_TYPE".PART_TYPE_03_SELECTED )
      I_Contact( "DB7215_PART_TYPE".PART_TYPE_04_SELECTED )
      I_Contact( "DB7215_PART_TYPE".PART_TYPE_05_SELECTED )
      I_Contact( "DB7215_PART_TYPE".PART_TYPE_06_SELECTED )
      I_Contact( "DB7215_PART_TYPE".PART_TYPE_07_SELECTED )
      I_Contact( "DB7215_PART_TYPE".PART_TYPE_08_SELECTED )
      I_Contact( "DB7215_PART_TYPE".PART_TYPE_09_SELECTED )
      I_Contact( "DB7215_PART_TYPE".PART_TYPE_10_SELECTED )
      Not()
      Coil( "DB2440_GLOBAL_DATA".GLOBAL_DATA.U02_RN_CYCLE_PART_TYPE )
   END_RUNG
   // the same network as SCL:
   "DB2440_GLOBAL_DATA".GLOBAL_DATA.U02_RN_CYCLE_PART_TYPE := NOT (NOT "DB7215_PART_TYPE".PART_TYPE_01_SELECTED AND NOT "DB7215_PART_TYPE".PART_TYPE_02_SELECTED AND NOT "DB7215_PART_TYPE".PART_TYPE_03_SELECTED AND NOT "DB7215_PART_TYPE".PART_TYPE_04_SELECTED AND NOT "DB7215_PART_TYPE".PART_TYPE_05_SELECTED AND NOT "DB7215_PART_TYPE".PART_TYPE_06_SELECTED AND NOT "DB7215_PART_TYPE".PART_TYPE_07_SELECTED AND NOT "DB7215_PART_TYPE".PART_TYPE_08_SELECTED AND NOT "DB7215_PART_TYPE".PART_TYPE_09_SELECTED AND NOT "DB7215_PART_TYPE".PART_TYPE_10_SELECTED);
END_REGION

REGION Network 99: UNIT 02 N-R CYCLE PART TYPE
   RUNG wire#powerrail
      Contact( "M_ONE" )
      Not()
      Coil( "DB2440_GLOBAL_DATA".GLOBAL_DATA.U02_NR_CYCLE_PART_TYPE )
   END_RUNG
   // the same network as SCL:
   "DB2440_GLOBAL_DATA".GLOBAL_DATA.U02_NR_CYCLE_PART_TYPE := NOT "M_ONE";
END_REGION

REGION Network 100: CHANNEL 1 PARAMETER SET SELECTION A
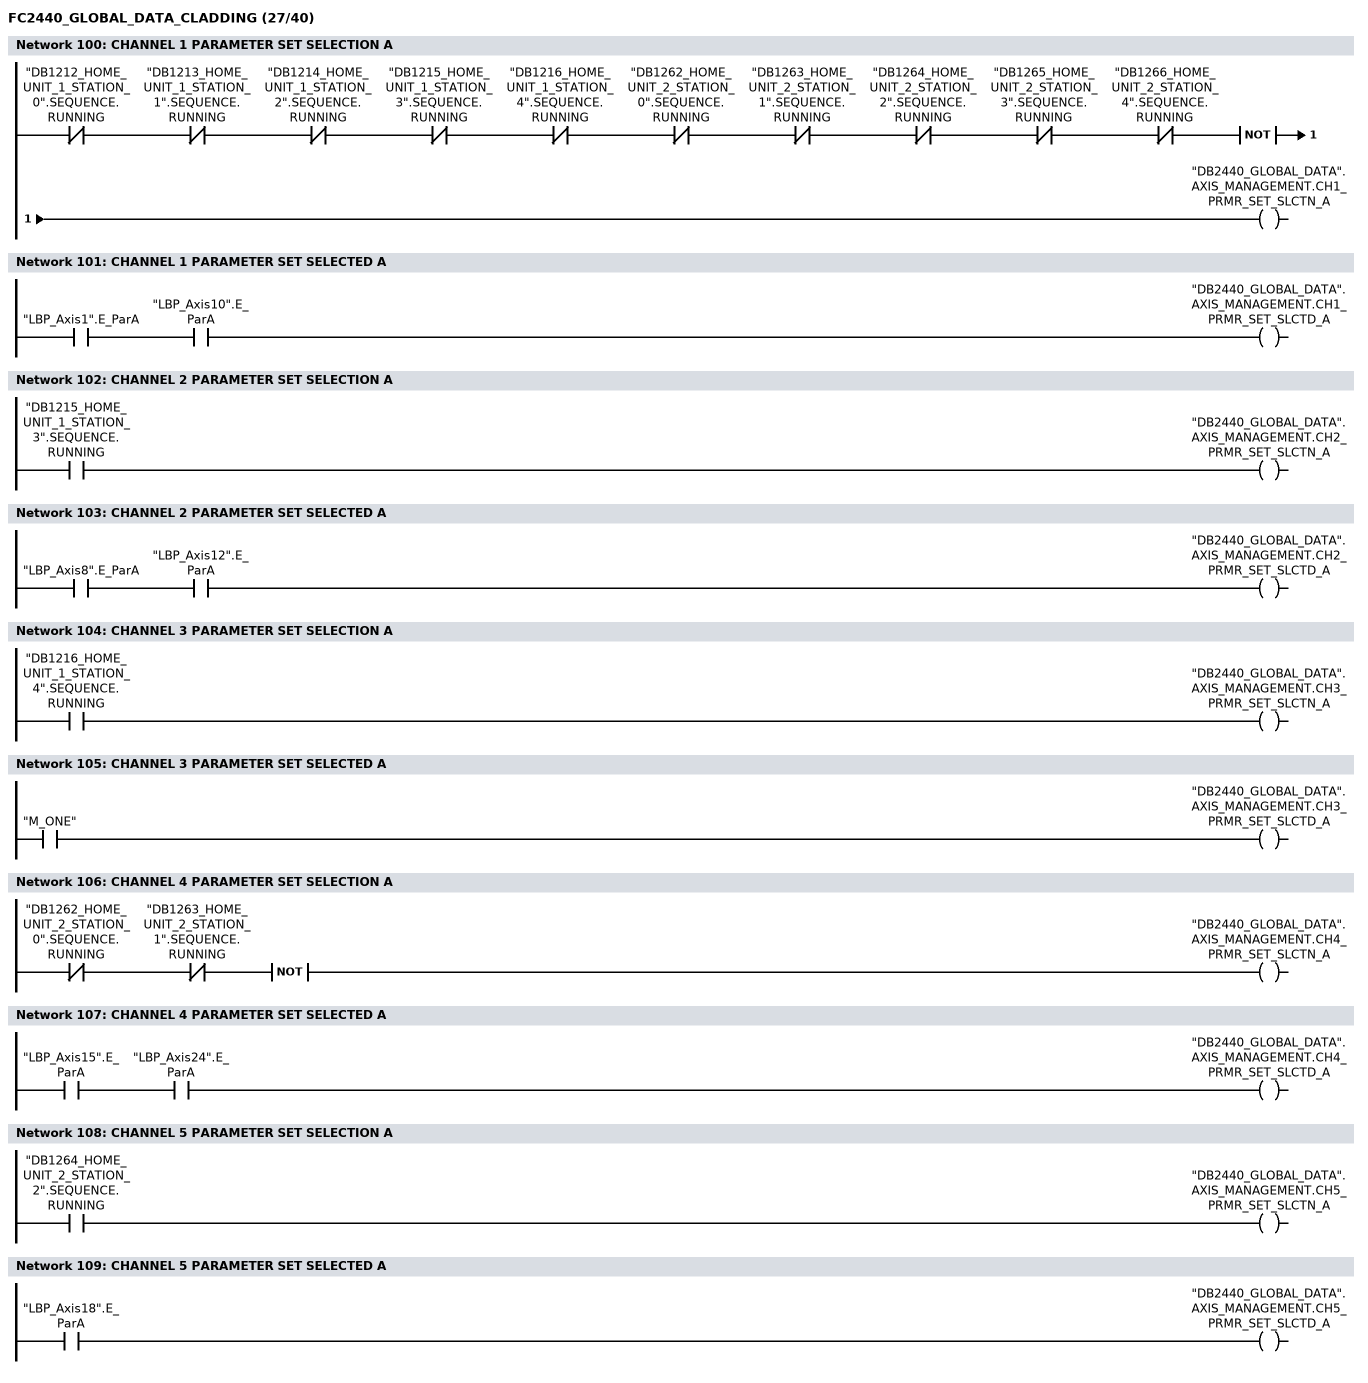
   RUNG wire#powerrail
      I_Contact( "DB1212_HOME_UNIT_1_STATION_0".SEQUENCE.RUNNING )
      I_Contact( "DB1213_HOME_UNIT_1_STATION_1".SEQUENCE.RUNNING )
      I_Contact( "DB1214_HOME_UNIT_1_STATION_2".SEQUENCE.RUNNING )
      I_Contact( "DB1215_HOME_UNIT_1_STATION_3".SEQUENCE.RUNNING )
      I_Contact( "DB1216_HOME_UNIT_1_STATION_4".SEQUENCE.RUNNING )
      I_Contact( "DB1262_HOME_UNIT_2_STATION_0".SEQUENCE.RUNNING )
      I_Contact( "DB1263_HOME_UNIT_2_STATION_1".SEQUENCE.RUNNING )
      I_Contact( "DB1264_HOME_UNIT_2_STATION_2".SEQUENCE.RUNNING )
      I_Contact( "DB1265_HOME_UNIT_2_STATION_3".SEQUENCE.RUNNING )
      I_Contact( "DB1266_HOME_UNIT_2_STATION_4".SEQUENCE.RUNNING )
      Not()
      Coil( "DB2440_GLOBAL_DATA".AXIS_MANAGEMENT.CH1_PRMR_SET_SLCTN_A )
   END_RUNG
   // the same network as SCL:
   "DB2440_GLOBAL_DATA".AXIS_MANAGEMENT.CH1_PRMR_SET_SLCTN_A := NOT (NOT "DB1212_HOME_UNIT_1_STATION_0".SEQUENCE.RUNNING AND NOT "DB1213_HOME_UNIT_1_STATION_1".SEQUENCE.RUNNING AND NOT "DB1214_HOME_UNIT_1_STATION_2".SEQUENCE.RUNNING AND NOT "DB1215_HOME_UNIT_1_STATION_3".SEQUENCE.RUNNING AND NOT "DB1216_HOME_UNIT_1_STATION_4".SEQUENCE.RUNNING AND NOT "DB1262_HOME_UNIT_2_STATION_0".SEQUENCE.RUNNING AND NOT "DB1263_HOME_UNIT_2_STATION_1".SEQUENCE.RUNNING AND NOT "DB1264_HOME_UNIT_2_STATION_2".SEQUENCE.RUNNING AND NOT "DB1265_HOME_UNIT_2_STATION_3".SEQUENCE.RUNNING AND NOT "DB1266_HOME_UNIT_2_STATION_4".SEQUENCE.RUNNING);
END_REGION

REGION Network 101: CHANNEL 1 PARAMETER SET SELECTED A
   RUNG wire#powerrail
      Contact( "LBP_Axis1".E_ParA )
      Contact( "LBP_Axis10".E_ParA )
      Coil( "DB2440_GLOBAL_DATA".AXIS_MANAGEMENT.CH1_PRMR_SET_SLCTD_A )
   END_RUNG
   // the same network as SCL:
   "DB2440_GLOBAL_DATA".AXIS_MANAGEMENT.CH1_PRMR_SET_SLCTD_A := "LBP_Axis1".E_ParA AND "LBP_Axis10".E_ParA;
END_REGION

REGION Network 102: CHANNEL 2 PARAMETER SET SELECTION A
   RUNG wire#powerrail
      Contact( "DB1215_HOME_UNIT_1_STATION_3".SEQUENCE.RUNNING )
      Coil( "DB2440_GLOBAL_DATA".AXIS_MANAGEMENT.CH2_PRMR_SET_SLCTN_A )
   END_RUNG
   // the same network as SCL:
   "DB2440_GLOBAL_DATA".AXIS_MANAGEMENT.CH2_PRMR_SET_SLCTN_A := "DB1215_HOME_UNIT_1_STATION_3".SEQUENCE.RUNNING;
END_REGION

REGION Network 103: CHANNEL 2 PARAMETER SET SELECTED A
   RUNG wire#powerrail
      Contact( "LBP_Axis8".E_ParA )
      Contact( "LBP_Axis12".E_ParA )
      Coil( "DB2440_GLOBAL_DATA".AXIS_MANAGEMENT.CH2_PRMR_SET_SLCTD_A )
   END_RUNG
   // the same network as SCL:
   "DB2440_GLOBAL_DATA".AXIS_MANAGEMENT.CH2_PRMR_SET_SLCTD_A := "LBP_Axis8".E_ParA AND "LBP_Axis12".E_ParA;
END_REGION

REGION Network 104: CHANNEL 3 PARAMETER SET SELECTION A
   RUNG wire#powerrail
      Contact( "DB1216_HOME_UNIT_1_STATION_4".SEQUENCE.RUNNING )
      Coil( "DB2440_GLOBAL_DATA".AXIS_MANAGEMENT.CH3_PRMR_SET_SLCTN_A )
   END_RUNG
   // the same network as SCL:
   "DB2440_GLOBAL_DATA".AXIS_MANAGEMENT.CH3_PRMR_SET_SLCTN_A := "DB1216_HOME_UNIT_1_STATION_4".SEQUENCE.RUNNING;
END_REGION

REGION Network 105: CHANNEL 3 PARAMETER SET SELECTED A
   RUNG wire#powerrail
      Contact( "M_ONE" )
      Coil( "DB2440_GLOBAL_DATA".AXIS_MANAGEMENT.CH3_PRMR_SET_SLCTD_A )
   END_RUNG
   // the same network as SCL:
   "DB2440_GLOBAL_DATA".AXIS_MANAGEMENT.CH3_PRMR_SET_SLCTD_A := "M_ONE";
END_REGION

REGION Network 106: CHANNEL 4 PARAMETER SET SELECTION A
   RUNG wire#powerrail
      I_Contact( "DB1262_HOME_UNIT_2_STATION_0".SEQUENCE.RUNNING )
      I_Contact( "DB1263_HOME_UNIT_2_STATION_1".SEQUENCE.RUNNING )
      Not()
      Coil( "DB2440_GLOBAL_DATA".AXIS_MANAGEMENT.CH4_PRMR_SET_SLCTN_A )
   END_RUNG
   // the same network as SCL:
   "DB2440_GLOBAL_DATA".AXIS_MANAGEMENT.CH4_PRMR_SET_SLCTN_A := NOT (NOT "DB1262_HOME_UNIT_2_STATION_0".SEQUENCE.RUNNING AND NOT "DB1263_HOME_UNIT_2_STATION_1".SEQUENCE.RUNNING);
END_REGION

REGION Network 107: CHANNEL 4 PARAMETER SET SELECTED A
   RUNG wire#powerrail
      Contact( "LBP_Axis15".E_ParA )
      Contact( "LBP_Axis24".E_ParA )
      Coil( "DB2440_GLOBAL_DATA".AXIS_MANAGEMENT.CH4_PRMR_SET_SLCTD_A )
   END_RUNG
   // the same network as SCL:
   "DB2440_GLOBAL_DATA".AXIS_MANAGEMENT.CH4_PRMR_SET_SLCTD_A := "LBP_Axis15".E_ParA AND "LBP_Axis24".E_ParA;
END_REGION

REGION Network 108: CHANNEL 5 PARAMETER SET SELECTION A
   RUNG wire#powerrail
      Contact( "DB1264_HOME_UNIT_2_STATION_2".SEQUENCE.RUNNING )
      Coil( "DB2440_GLOBAL_DATA".AXIS_MANAGEMENT.CH5_PRMR_SET_SLCTN_A )
   END_RUNG
   // the same network as SCL:
   "DB2440_GLOBAL_DATA".AXIS_MANAGEMENT.CH5_PRMR_SET_SLCTN_A := "DB1264_HOME_UNIT_2_STATION_2".SEQUENCE.RUNNING;
END_REGION

REGION Network 109: CHANNEL 5 PARAMETER SET SELECTED A
   RUNG wire#powerrail
      Contact( "LBP_Axis18".E_ParA )
      Coil( "DB2440_GLOBAL_DATA".AXIS_MANAGEMENT.CH5_PRMR_SET_SLCTD_A )
   END_RUNG
   // the same network as SCL:
   "DB2440_GLOBAL_DATA".AXIS_MANAGEMENT.CH5_PRMR_SET_SLCTD_A := "LBP_Axis18".E_ParA;
END_REGION

REGION Network 110: CHANNEL 6 PARAMETER SET SELECTION A
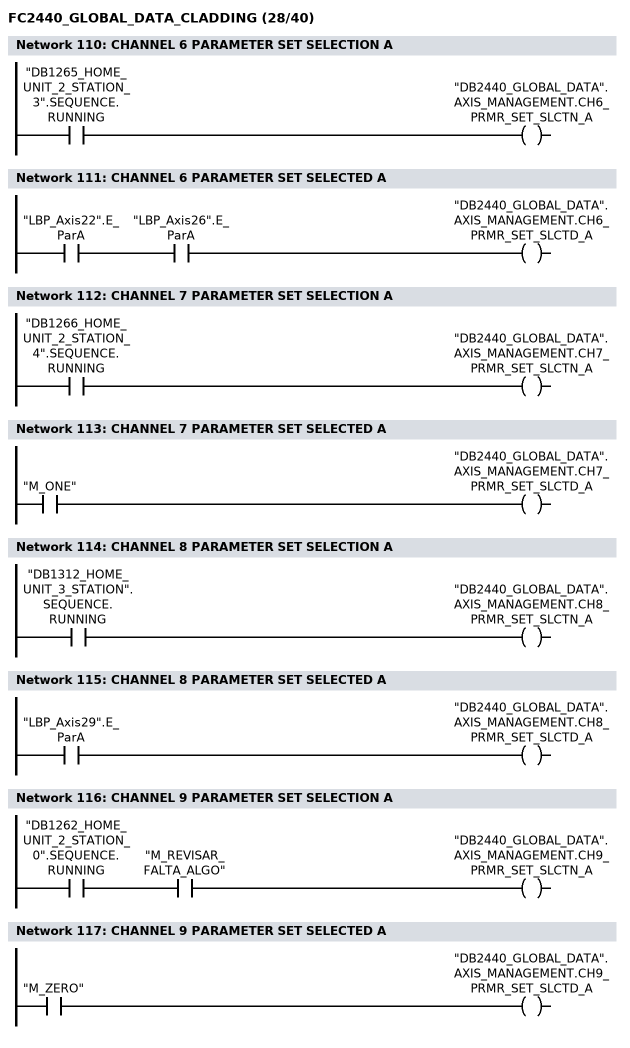
   RUNG wire#powerrail
      Contact( "DB1265_HOME_UNIT_2_STATION_3".SEQUENCE.RUNNING )
      Coil( "DB2440_GLOBAL_DATA".AXIS_MANAGEMENT.CH6_PRMR_SET_SLCTN_A )
   END_RUNG
   // the same network as SCL:
   "DB2440_GLOBAL_DATA".AXIS_MANAGEMENT.CH6_PRMR_SET_SLCTN_A := "DB1265_HOME_UNIT_2_STATION_3".SEQUENCE.RUNNING;
END_REGION

REGION Network 111: CHANNEL 6 PARAMETER SET SELECTED A
   RUNG wire#powerrail
      Contact( "LBP_Axis22".E_ParA )
      Contact( "LBP_Axis26".E_ParA )
      Coil( "DB2440_GLOBAL_DATA".AXIS_MANAGEMENT.CH6_PRMR_SET_SLCTD_A )
   END_RUNG
   // the same network as SCL:
   "DB2440_GLOBAL_DATA".AXIS_MANAGEMENT.CH6_PRMR_SET_SLCTD_A := "LBP_Axis22".E_ParA AND "LBP_Axis26".E_ParA;
END_REGION

REGION Network 112: CHANNEL 7 PARAMETER SET SELECTION A
   RUNG wire#powerrail
      Contact( "DB1266_HOME_UNIT_2_STATION_4".SEQUENCE.RUNNING )
      Coil( "DB2440_GLOBAL_DATA".AXIS_MANAGEMENT.CH7_PRMR_SET_SLCTN_A )
   END_RUNG
   // the same network as SCL:
   "DB2440_GLOBAL_DATA".AXIS_MANAGEMENT.CH7_PRMR_SET_SLCTN_A := "DB1266_HOME_UNIT_2_STATION_4".SEQUENCE.RUNNING;
END_REGION

REGION Network 113: CHANNEL 7 PARAMETER SET SELECTED A
   RUNG wire#powerrail
      Contact( "M_ONE" )
      Coil( "DB2440_GLOBAL_DATA".AXIS_MANAGEMENT.CH7_PRMR_SET_SLCTD_A )
   END_RUNG
   // the same network as SCL:
   "DB2440_GLOBAL_DATA".AXIS_MANAGEMENT.CH7_PRMR_SET_SLCTD_A := "M_ONE";
END_REGION

REGION Network 114: CHANNEL 8 PARAMETER SET SELECTION A
   RUNG wire#powerrail
      Contact( "DB1312_HOME_UNIT_3_STATION".SEQUENCE.RUNNING )
      Coil( "DB2440_GLOBAL_DATA".AXIS_MANAGEMENT.CH8_PRMR_SET_SLCTN_A )
   END_RUNG
   // the same network as SCL:
   "DB2440_GLOBAL_DATA".AXIS_MANAGEMENT.CH8_PRMR_SET_SLCTN_A := "DB1312_HOME_UNIT_3_STATION".SEQUENCE.RUNNING;
END_REGION

REGION Network 115: CHANNEL 8 PARAMETER SET SELECTED A
   RUNG wire#powerrail
      Contact( "LBP_Axis29".E_ParA )
      Coil( "DB2440_GLOBAL_DATA".AXIS_MANAGEMENT.CH8_PRMR_SET_SLCTD_A )
   END_RUNG
   // the same network as SCL:
   "DB2440_GLOBAL_DATA".AXIS_MANAGEMENT.CH8_PRMR_SET_SLCTD_A := "LBP_Axis29".E_ParA;
END_REGION

REGION Network 116: CHANNEL 9 PARAMETER SET SELECTION A
   RUNG wire#powerrail
      Contact( "DB1262_HOME_UNIT_2_STATION_0".SEQUENCE.RUNNING )
      Contact( "M_REVISAR_FALTA_ALGO" )
      Coil( "DB2440_GLOBAL_DATA".AXIS_MANAGEMENT.CH9_PRMR_SET_SLCTN_A )
   END_RUNG
   // the same network as SCL:
   "DB2440_GLOBAL_DATA".AXIS_MANAGEMENT.CH9_PRMR_SET_SLCTN_A := "DB1262_HOME_UNIT_2_STATION_0".SEQUENCE.RUNNING AND "M_REVISAR_FALTA_ALGO";
END_REGION

REGION Network 117: CHANNEL 9 PARAMETER SET SELECTED A
   RUNG wire#powerrail
      Contact( "M_ZERO" )
      Coil( "DB2440_GLOBAL_DATA".AXIS_MANAGEMENT.CH9_PRMR_SET_SLCTD_A )
   END_RUNG
   // the same network as SCL:
   "DB2440_GLOBAL_DATA".AXIS_MANAGEMENT.CH9_PRMR_SET_SLCTD_A := "M_ZERO";
END_REGION

REGION Network 118: ALL FULL DEPTH UNIT 01
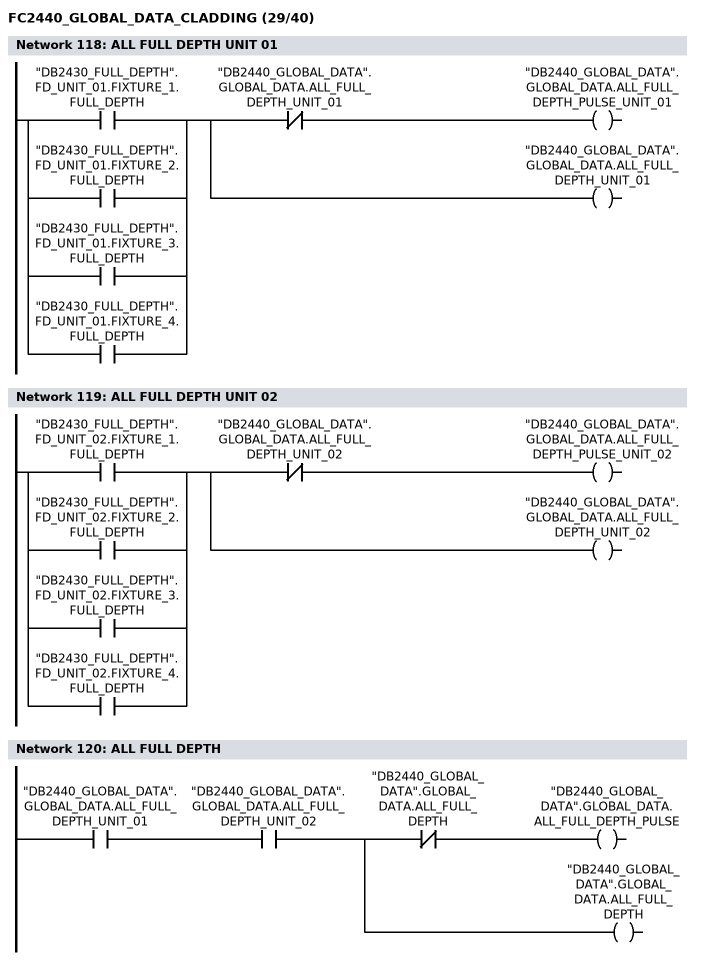
   RUNG wire#powerrail
      Contact( "DB2430_FULL_DEPTH".FD_UNIT_01.FIXTURE_1.FULL_DEPTH )
      wire#w1
      I_Contact( "DB2440_GLOBAL_DATA".GLOBAL_DATA.ALL_FULL_DEPTH_UNIT_01 )
      Coil( "DB2440_GLOBAL_DATA".GLOBAL_DATA.ALL_FULL_DEPTH_PULSE_UNIT_01 )
   END_RUNG
   RUNG wire#powerrail
      Contact( "DB2430_FULL_DEPTH".FD_UNIT_01.FIXTURE_2.FULL_DEPTH )
   END_RUNG wire#w1
   RUNG wire#powerrail
      Contact( "DB2430_FULL_DEPTH".FD_UNIT_01.FIXTURE_3.FULL_DEPTH )
   END_RUNG wire#w1
   RUNG wire#powerrail
      Contact( "DB2430_FULL_DEPTH".FD_UNIT_01.FIXTURE_4.FULL_DEPTH )
   END_RUNG wire#w1
   RUNG wire#w1
      Coil( "DB2440_GLOBAL_DATA".GLOBAL_DATA.ALL_FULL_DEPTH_UNIT_01 )
   END_RUNG
   // the same network as SCL:
   #_w1 := "DB2430_FULL_DEPTH".FD_UNIT_01.FIXTURE_1.FULL_DEPTH OR "DB2430_FULL_DEPTH".FD_UNIT_01.FIXTURE_2.FULL_DEPTH OR "DB2430_FULL_DEPTH".FD_UNIT_01.FIXTURE_3.FULL_DEPTH OR "DB2430_FULL_DEPTH".FD_UNIT_01.FIXTURE_4.FULL_DEPTH;
   "DB2440_GLOBAL_DATA".GLOBAL_DATA.ALL_FULL_DEPTH_PULSE_UNIT_01 := #_w1 AND NOT "DB2440_GLOBAL_DATA".GLOBAL_DATA.ALL_FULL_DEPTH_UNIT_01;
   "DB2440_GLOBAL_DATA".GLOBAL_DATA.ALL_FULL_DEPTH_UNIT_01 := #_w1;
END_REGION

REGION Network 119: ALL FULL DEPTH UNIT 02
   RUNG wire#powerrail
      Contact( "DB2430_FULL_DEPTH".FD_UNIT_02.FIXTURE_1.FULL_DEPTH )
      wire#w1
      I_Contact( "DB2440_GLOBAL_DATA".GLOBAL_DATA.ALL_FULL_DEPTH_UNIT_02 )
      Coil( "DB2440_GLOBAL_DATA".GLOBAL_DATA.ALL_FULL_DEPTH_PULSE_UNIT_02 )
   END_RUNG
   RUNG wire#powerrail
      Contact( "DB2430_FULL_DEPTH".FD_UNIT_02.FIXTURE_2.FULL_DEPTH )
   END_RUNG wire#w1
   RUNG wire#powerrail
      Contact( "DB2430_FULL_DEPTH".FD_UNIT_02.FIXTURE_3.FULL_DEPTH )
   END_RUNG wire#w1
   RUNG wire#powerrail
      Contact( "DB2430_FULL_DEPTH".FD_UNIT_02.FIXTURE_4.FULL_DEPTH )
   END_RUNG wire#w1
   RUNG wire#w1
      Coil( "DB2440_GLOBAL_DATA".GLOBAL_DATA.ALL_FULL_DEPTH_UNIT_02 )
   END_RUNG
   // the same network as SCL:
   #_w1 := "DB2430_FULL_DEPTH".FD_UNIT_02.FIXTURE_1.FULL_DEPTH OR "DB2430_FULL_DEPTH".FD_UNIT_02.FIXTURE_2.FULL_DEPTH OR "DB2430_FULL_DEPTH".FD_UNIT_02.FIXTURE_3.FULL_DEPTH OR "DB2430_FULL_DEPTH".FD_UNIT_02.FIXTURE_4.FULL_DEPTH;
   "DB2440_GLOBAL_DATA".GLOBAL_DATA.ALL_FULL_DEPTH_PULSE_UNIT_02 := #_w1 AND NOT "DB2440_GLOBAL_DATA".GLOBAL_DATA.ALL_FULL_DEPTH_UNIT_02;
   "DB2440_GLOBAL_DATA".GLOBAL_DATA.ALL_FULL_DEPTH_UNIT_02 := #_w1;
END_REGION

REGION Network 120: ALL FULL DEPTH
   RUNG wire#powerrail
      Contact( "DB2440_GLOBAL_DATA".GLOBAL_DATA.ALL_FULL_DEPTH_UNIT_01 )
      Contact( "DB2440_GLOBAL_DATA".GLOBAL_DATA.ALL_FULL_DEPTH_UNIT_02 )
      wire#w1
      I_Contact( "DB2440_GLOBAL_DATA".GLOBAL_DATA.ALL_FULL_DEPTH )
      Coil( "DB2440_GLOBAL_DATA".GLOBAL_DATA.ALL_FULL_DEPTH_PULSE )
   END_RUNG
   RUNG wire#w1
      Coil( "DB2440_GLOBAL_DATA".GLOBAL_DATA.ALL_FULL_DEPTH )
   END_RUNG
   // the same network as SCL:
   #_w1 := "DB2440_GLOBAL_DATA".GLOBAL_DATA.ALL_FULL_DEPTH_UNIT_01 AND "DB2440_GLOBAL_DATA".GLOBAL_DATA.ALL_FULL_DEPTH_UNIT_02;
   "DB2440_GLOBAL_DATA".GLOBAL_DATA.ALL_FULL_DEPTH_PULSE := #_w1 AND NOT "DB2440_GLOBAL_DATA".GLOBAL_DATA.ALL_FULL_DEPTH;
   "DB2440_GLOBAL_DATA".GLOBAL_DATA.ALL_FULL_DEPTH := #_w1;
END_REGION

REGION Network 121: RESET FULL DEPTH PULSE UNIT 01 FIXTURE 1
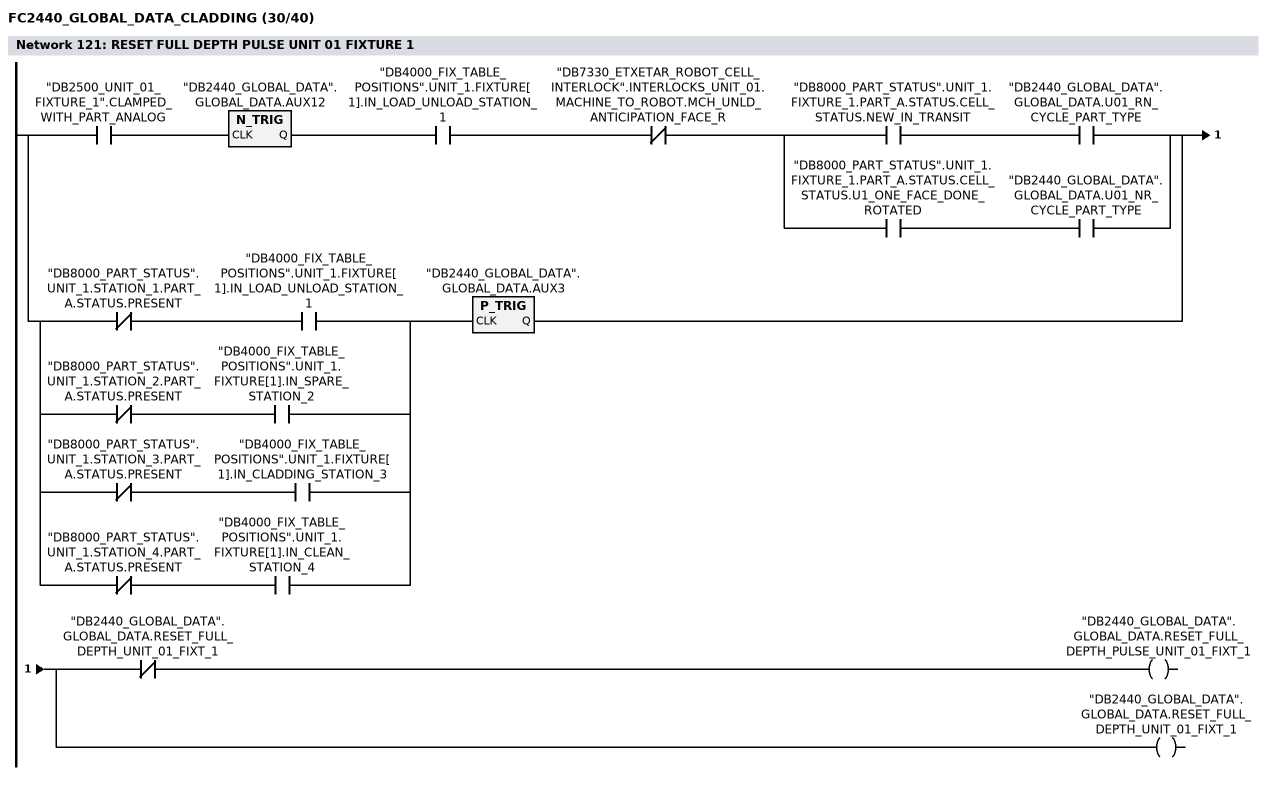
   RUNG wire#powerrail
      Contact( "DB2500_UNIT_01_FIXTURE_1".CLAMPED_WITH_PART_ANALOG )
      N_Trig( "DB2440_GLOBAL_DATA".GLOBAL_DATA.AUX12 )
      Contact( "DB4000_FIX_TABLE_POSITIONS".UNIT_1.FIXTURE[1].IN_LOAD_UNLOAD_STATION_1 )
      I_Contact( "DB7330_ETXETAR_ROBOT_CELL_INTERLOCK".INTERLOCKS_UNIT_01.MACHINE_TO_ROBOT.MCH_UNLD_ANTICIPATION_FACE_R )
      wire#w1
      Contact( "DB8000_PART_STATUS".UNIT_1.FIXTURE_1.PART_A.STATUS.CELL_STATUS.NEW_IN_TRANSIT )
      Contact( "DB2440_GLOBAL_DATA".GLOBAL_DATA.U01_RN_CYCLE_PART_TYPE )
      wire#w2
      I_Contact( "DB2440_GLOBAL_DATA".GLOBAL_DATA.RESET_FULL_DEPTH_UNIT_01_FIXT_1 )
      Coil( "DB2440_GLOBAL_DATA".GLOBAL_DATA.RESET_FULL_DEPTH_PULSE_UNIT_01_FIXT_1 )
   END_RUNG
   RUNG wire#w1
      Contact( "DB8000_PART_STATUS".UNIT_1.FIXTURE_1.PART_A.STATUS.CELL_STATUS.U1_ONE_FACE_DONE_ROTATED )
      Contact( "DB2440_GLOBAL_DATA".GLOBAL_DATA.U01_NR_CYCLE_PART_TYPE )
   END_RUNG wire#w2
   RUNG wire#powerrail
      I_Contact( "DB8000_PART_STATUS".UNIT_1.STATION_1.PART_A.STATUS.PRESENT )
      Contact( "DB4000_FIX_TABLE_POSITIONS".UNIT_1.FIXTURE[1].IN_LOAD_UNLOAD_STATION_1 )
      wire#w3
      P_Trig( "DB2440_GLOBAL_DATA".GLOBAL_DATA.AUX3 )
   END_RUNG wire#w2
   RUNG wire#powerrail
      I_Contact( "DB8000_PART_STATUS".UNIT_1.STATION_2.PART_A.STATUS.PRESENT )
      Contact( "DB4000_FIX_TABLE_POSITIONS".UNIT_1.FIXTURE[1].IN_SPARE_STATION_2 )
   END_RUNG wire#w3
   RUNG wire#powerrail
      I_Contact( "DB8000_PART_STATUS".UNIT_1.STATION_3.PART_A.STATUS.PRESENT )
      Contact( "DB4000_FIX_TABLE_POSITIONS".UNIT_1.FIXTURE[1].IN_CLADDING_STATION_3 )
   END_RUNG wire#w3
   RUNG wire#powerrail
      I_Contact( "DB8000_PART_STATUS".UNIT_1.STATION_4.PART_A.STATUS.PRESENT )
      Contact( "DB4000_FIX_TABLE_POSITIONS".UNIT_1.FIXTURE[1].IN_CLEAN_STATION_4 )
   END_RUNG wire#w3
   RUNG wire#w2
      Coil( "DB2440_GLOBAL_DATA".GLOBAL_DATA.RESET_FULL_DEPTH_UNIT_01_FIXT_1 )
   END_RUNG
   // the same network as SCL:
   #_w1 := NOT "DB2500_UNIT_01_FIXTURE_1".CLAMPED_WITH_PART_ANALOG AND "DB2440_GLOBAL_DATA".GLOBAL_DATA.AUX12;   // falling edge
   "DB2440_GLOBAL_DATA".GLOBAL_DATA.AUX12 := "DB2500_UNIT_01_FIXTURE_1".CLAMPED_WITH_PART_ANALOG;
   #_w2 := (NOT "DB8000_PART_STATUS".UNIT_1.STATION_1.PART_A.STATUS.PRESENT AND "DB4000_FIX_TABLE_POSITIONS".UNIT_1.FIXTURE[1].IN_LOAD_UNLOAD_STATION_1) OR (NOT "DB8000_PART_STATUS".UNIT_1.STATION_2.PART_A.STATUS.PRESENT AND "DB4000_FIX_TABLE_POSITIONS".UNIT_1.FIXTURE[1].IN_SPARE_STATION_2) OR (NOT "DB8000_PART_STATUS".UNIT_1.STATION_3.PART_A.STATUS.PRESENT AND "DB4000_FIX_TABLE_POSITIONS".UNIT_1.FIXTURE[1].IN_CLADDING_STATION_3) OR (NOT "DB8000_PART_STATUS".UNIT_1.STATION_4.PART_A.STATUS.PRESENT AND "DB4000_FIX_TABLE_POSITIONS".UNIT_1.FIXTURE[1].IN_CLEAN_STATION_4);
   #_w3 := #_w2 AND NOT "DB2440_GLOBAL_DATA".GLOBAL_DATA.AUX3;   // rising edge
   "DB2440_GLOBAL_DATA".GLOBAL_DATA.AUX3 := #_w2;
   #_w4 := (#_w1 AND "DB4000_FIX_TABLE_POSITIONS".UNIT_1.FIXTURE[1].IN_LOAD_UNLOAD_STATION_1 AND NOT "DB7330_ETXETAR_ROBOT_CELL_INTERLOCK".INTERLOCKS_UNIT_01.MACHINE_TO_ROBOT.MCH_UNLD_ANTICIPATION_FACE_R AND (("DB8000_PART_STATUS".UNIT_1.FIXTURE_1.PART_A.STATUS.CELL_STATUS.NEW_IN_TRANSIT AND "DB2440_GLOBAL_DATA".GLOBAL_DATA.U01_RN_CYCLE_PART_TYPE) OR ("DB8000_PART_STATUS".UNIT_1.FIXTURE_1.PART_A.STATUS.CELL_STATUS.U1_ONE_FACE_DONE_ROTATED AND "DB2440_GLOBAL_DATA".GLOBAL_DATA.U01_NR_CYCLE_PART_TYPE))) OR #_w3;
   "DB2440_GLOBAL_DATA".GLOBAL_DATA.RESET_FULL_DEPTH_PULSE_UNIT_01_FIXT_1 := #_w4 AND NOT "DB2440_GLOBAL_DATA".GLOBAL_DATA.RESET_FULL_DEPTH_UNIT_01_FIXT_1;
   "DB2440_GLOBAL_DATA".GLOBAL_DATA.RESET_FULL_DEPTH_UNIT_01_FIXT_1 := #_w4;
END_REGION

REGION Network 122: RESET FULL DEPTH PULSE UNIT 01 FIXTURE 2
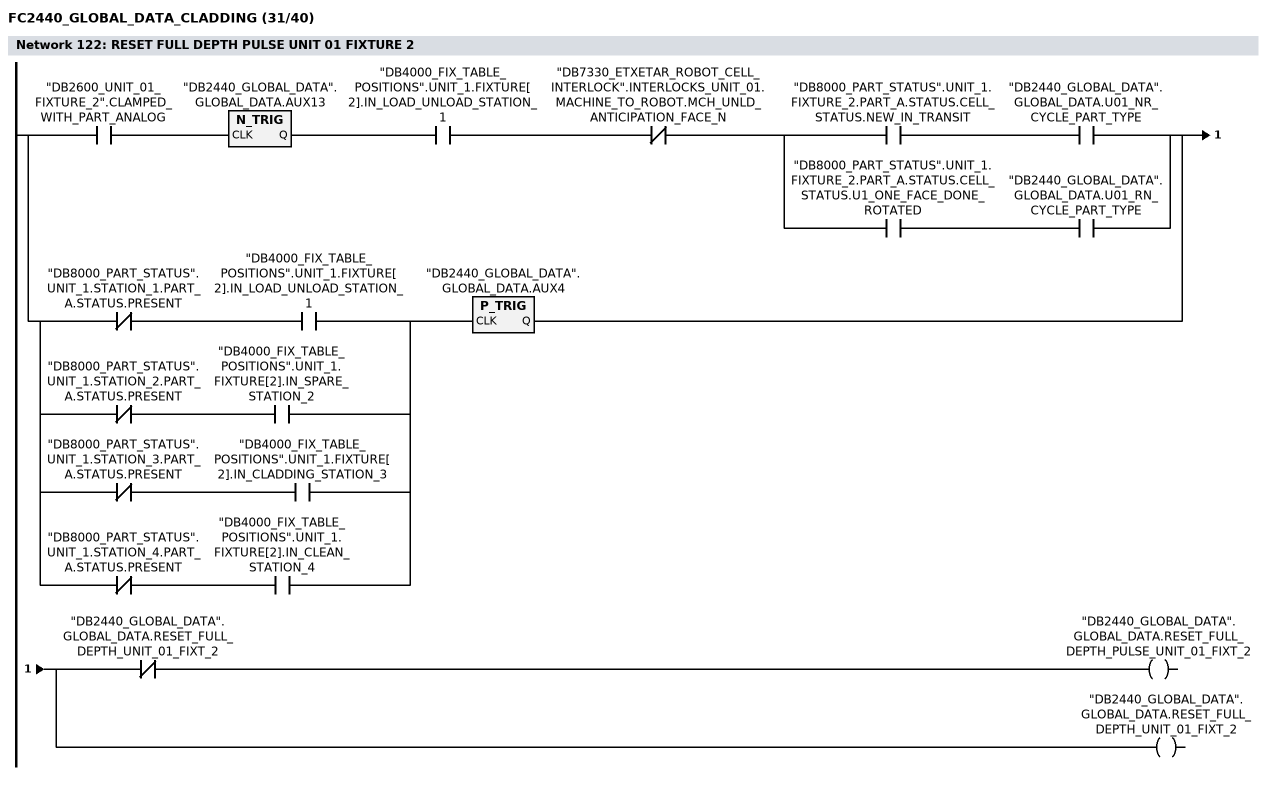
   RUNG wire#powerrail
      Contact( "DB2600_UNIT_01_FIXTURE_2".CLAMPED_WITH_PART_ANALOG )
      N_Trig( "DB2440_GLOBAL_DATA".GLOBAL_DATA.AUX13 )
      Contact( "DB4000_FIX_TABLE_POSITIONS".UNIT_1.FIXTURE[2].IN_LOAD_UNLOAD_STATION_1 )
      I_Contact( "DB7330_ETXETAR_ROBOT_CELL_INTERLOCK".INTERLOCKS_UNIT_01.MACHINE_TO_ROBOT.MCH_UNLD_ANTICIPATION_FACE_N )
      wire#w1
      Contact( "DB8000_PART_STATUS".UNIT_1.FIXTURE_2.PART_A.STATUS.CELL_STATUS.NEW_IN_TRANSIT )
      Contact( "DB2440_GLOBAL_DATA".GLOBAL_DATA.U01_NR_CYCLE_PART_TYPE )
      wire#w2
      I_Contact( "DB2440_GLOBAL_DATA".GLOBAL_DATA.RESET_FULL_DEPTH_UNIT_01_FIXT_2 )
      Coil( "DB2440_GLOBAL_DATA".GLOBAL_DATA.RESET_FULL_DEPTH_PULSE_UNIT_01_FIXT_2 )
   END_RUNG
   RUNG wire#w1
      Contact( "DB8000_PART_STATUS".UNIT_1.FIXTURE_2.PART_A.STATUS.CELL_STATUS.U1_ONE_FACE_DONE_ROTATED )
      Contact( "DB2440_GLOBAL_DATA".GLOBAL_DATA.U01_RN_CYCLE_PART_TYPE )
   END_RUNG wire#w2
   RUNG wire#powerrail
      I_Contact( "DB8000_PART_STATUS".UNIT_1.STATION_1.PART_A.STATUS.PRESENT )
      Contact( "DB4000_FIX_TABLE_POSITIONS".UNIT_1.FIXTURE[2].IN_LOAD_UNLOAD_STATION_1 )
      wire#w3
      P_Trig( "DB2440_GLOBAL_DATA".GLOBAL_DATA.AUX4 )
   END_RUNG wire#w2
   RUNG wire#powerrail
      I_Contact( "DB8000_PART_STATUS".UNIT_1.STATION_2.PART_A.STATUS.PRESENT )
      Contact( "DB4000_FIX_TABLE_POSITIONS".UNIT_1.FIXTURE[2].IN_SPARE_STATION_2 )
   END_RUNG wire#w3
   RUNG wire#powerrail
      I_Contact( "DB8000_PART_STATUS".UNIT_1.STATION_3.PART_A.STATUS.PRESENT )
      Contact( "DB4000_FIX_TABLE_POSITIONS".UNIT_1.FIXTURE[2].IN_CLADDING_STATION_3 )
   END_RUNG wire#w3
   RUNG wire#powerrail
      I_Contact( "DB8000_PART_STATUS".UNIT_1.STATION_4.PART_A.STATUS.PRESENT )
      Contact( "DB4000_FIX_TABLE_POSITIONS".UNIT_1.FIXTURE[2].IN_CLEAN_STATION_4 )
   END_RUNG wire#w3
   RUNG wire#w2
      Coil( "DB2440_GLOBAL_DATA".GLOBAL_DATA.RESET_FULL_DEPTH_UNIT_01_FIXT_2 )
   END_RUNG
   // the same network as SCL:
   #_w1 := NOT "DB2600_UNIT_01_FIXTURE_2".CLAMPED_WITH_PART_ANALOG AND "DB2440_GLOBAL_DATA".GLOBAL_DATA.AUX13;   // falling edge
   "DB2440_GLOBAL_DATA".GLOBAL_DATA.AUX13 := "DB2600_UNIT_01_FIXTURE_2".CLAMPED_WITH_PART_ANALOG;
   #_w2 := (NOT "DB8000_PART_STATUS".UNIT_1.STATION_1.PART_A.STATUS.PRESENT AND "DB4000_FIX_TABLE_POSITIONS".UNIT_1.FIXTURE[2].IN_LOAD_UNLOAD_STATION_1) OR (NOT "DB8000_PART_STATUS".UNIT_1.STATION_2.PART_A.STATUS.PRESENT AND "DB4000_FIX_TABLE_POSITIONS".UNIT_1.FIXTURE[2].IN_SPARE_STATION_2) OR (NOT "DB8000_PART_STATUS".UNIT_1.STATION_3.PART_A.STATUS.PRESENT AND "DB4000_FIX_TABLE_POSITIONS".UNIT_1.FIXTURE[2].IN_CLADDING_STATION_3) OR (NOT "DB8000_PART_STATUS".UNIT_1.STATION_4.PART_A.STATUS.PRESENT AND "DB4000_FIX_TABLE_POSITIONS".UNIT_1.FIXTURE[2].IN_CLEAN_STATION_4);
   #_w3 := #_w2 AND NOT "DB2440_GLOBAL_DATA".GLOBAL_DATA.AUX4;   // rising edge
   "DB2440_GLOBAL_DATA".GLOBAL_DATA.AUX4 := #_w2;
   #_w4 := (#_w1 AND "DB4000_FIX_TABLE_POSITIONS".UNIT_1.FIXTURE[2].IN_LOAD_UNLOAD_STATION_1 AND NOT "DB7330_ETXETAR_ROBOT_CELL_INTERLOCK".INTERLOCKS_UNIT_01.MACHINE_TO_ROBOT.MCH_UNLD_ANTICIPATION_FACE_N AND (("DB8000_PART_STATUS".UNIT_1.FIXTURE_2.PART_A.STATUS.CELL_STATUS.NEW_IN_TRANSIT AND "DB2440_GLOBAL_DATA".GLOBAL_DATA.U01_NR_CYCLE_PART_TYPE) OR ("DB8000_PART_STATUS".UNIT_1.FIXTURE_2.PART_A.STATUS.CELL_STATUS.U1_ONE_FACE_DONE_ROTATED AND "DB2440_GLOBAL_DATA".GLOBAL_DATA.U01_RN_CYCLE_PART_TYPE))) OR #_w3;
   "DB2440_GLOBAL_DATA".GLOBAL_DATA.RESET_FULL_DEPTH_PULSE_UNIT_01_FIXT_2 := #_w4 AND NOT "DB2440_GLOBAL_DATA".GLOBAL_DATA.RESET_FULL_DEPTH_UNIT_01_FIXT_2;
   "DB2440_GLOBAL_DATA".GLOBAL_DATA.RESET_FULL_DEPTH_UNIT_01_FIXT_2 := #_w4;
END_REGION

REGION Network 123: RESET FULL DEPTH PULSE UNIT 01 FIXTURE 3
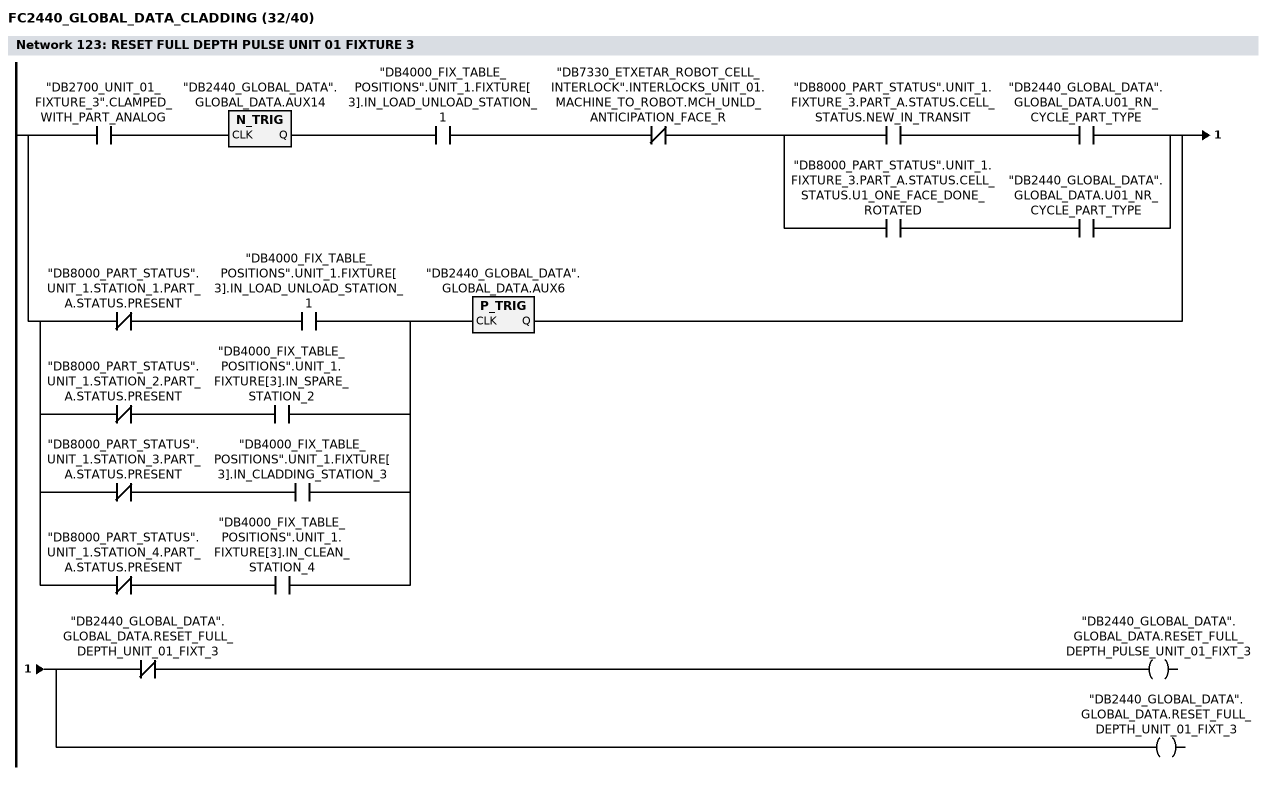
   RUNG wire#powerrail
      Contact( "DB2700_UNIT_01_FIXTURE_3".CLAMPED_WITH_PART_ANALOG )
      N_Trig( "DB2440_GLOBAL_DATA".GLOBAL_DATA.AUX14 )
      Contact( "DB4000_FIX_TABLE_POSITIONS".UNIT_1.FIXTURE[3].IN_LOAD_UNLOAD_STATION_1 )
      I_Contact( "DB7330_ETXETAR_ROBOT_CELL_INTERLOCK".INTERLOCKS_UNIT_01.MACHINE_TO_ROBOT.MCH_UNLD_ANTICIPATION_FACE_R )
      wire#w1
      Contact( "DB8000_PART_STATUS".UNIT_1.FIXTURE_3.PART_A.STATUS.CELL_STATUS.NEW_IN_TRANSIT )
      Contact( "DB2440_GLOBAL_DATA".GLOBAL_DATA.U01_RN_CYCLE_PART_TYPE )
      wire#w2
      I_Contact( "DB2440_GLOBAL_DATA".GLOBAL_DATA.RESET_FULL_DEPTH_UNIT_01_FIXT_3 )
      Coil( "DB2440_GLOBAL_DATA".GLOBAL_DATA.RESET_FULL_DEPTH_PULSE_UNIT_01_FIXT_3 )
   END_RUNG
   RUNG wire#w1
      Contact( "DB8000_PART_STATUS".UNIT_1.FIXTURE_3.PART_A.STATUS.CELL_STATUS.U1_ONE_FACE_DONE_ROTATED )
      Contact( "DB2440_GLOBAL_DATA".GLOBAL_DATA.U01_NR_CYCLE_PART_TYPE )
   END_RUNG wire#w2
   RUNG wire#powerrail
      I_Contact( "DB8000_PART_STATUS".UNIT_1.STATION_1.PART_A.STATUS.PRESENT )
      Contact( "DB4000_FIX_TABLE_POSITIONS".UNIT_1.FIXTURE[3].IN_LOAD_UNLOAD_STATION_1 )
      wire#w3
      P_Trig( "DB2440_GLOBAL_DATA".GLOBAL_DATA.AUX6 )
   END_RUNG wire#w2
   RUNG wire#powerrail
      I_Contact( "DB8000_PART_STATUS".UNIT_1.STATION_2.PART_A.STATUS.PRESENT )
      Contact( "DB4000_FIX_TABLE_POSITIONS".UNIT_1.FIXTURE[3].IN_SPARE_STATION_2 )
   END_RUNG wire#w3
   RUNG wire#powerrail
      I_Contact( "DB8000_PART_STATUS".UNIT_1.STATION_3.PART_A.STATUS.PRESENT )
      Contact( "DB4000_FIX_TABLE_POSITIONS".UNIT_1.FIXTURE[3].IN_CLADDING_STATION_3 )
   END_RUNG wire#w3
   RUNG wire#powerrail
      I_Contact( "DB8000_PART_STATUS".UNIT_1.STATION_4.PART_A.STATUS.PRESENT )
      Contact( "DB4000_FIX_TABLE_POSITIONS".UNIT_1.FIXTURE[3].IN_CLEAN_STATION_4 )
   END_RUNG wire#w3
   RUNG wire#w2
      Coil( "DB2440_GLOBAL_DATA".GLOBAL_DATA.RESET_FULL_DEPTH_UNIT_01_FIXT_3 )
   END_RUNG
   // the same network as SCL:
   #_w1 := NOT "DB2700_UNIT_01_FIXTURE_3".CLAMPED_WITH_PART_ANALOG AND "DB2440_GLOBAL_DATA".GLOBAL_DATA.AUX14;   // falling edge
   "DB2440_GLOBAL_DATA".GLOBAL_DATA.AUX14 := "DB2700_UNIT_01_FIXTURE_3".CLAMPED_WITH_PART_ANALOG;
   #_w2 := (NOT "DB8000_PART_STATUS".UNIT_1.STATION_1.PART_A.STATUS.PRESENT AND "DB4000_FIX_TABLE_POSITIONS".UNIT_1.FIXTURE[3].IN_LOAD_UNLOAD_STATION_1) OR (NOT "DB8000_PART_STATUS".UNIT_1.STATION_2.PART_A.STATUS.PRESENT AND "DB4000_FIX_TABLE_POSITIONS".UNIT_1.FIXTURE[3].IN_SPARE_STATION_2) OR (NOT "DB8000_PART_STATUS".UNIT_1.STATION_3.PART_A.STATUS.PRESENT AND "DB4000_FIX_TABLE_POSITIONS".UNIT_1.FIXTURE[3].IN_CLADDING_STATION_3) OR (NOT "DB8000_PART_STATUS".UNIT_1.STATION_4.PART_A.STATUS.PRESENT AND "DB4000_FIX_TABLE_POSITIONS".UNIT_1.FIXTURE[3].IN_CLEAN_STATION_4);
   #_w3 := #_w2 AND NOT "DB2440_GLOBAL_DATA".GLOBAL_DATA.AUX6;   // rising edge
   "DB2440_GLOBAL_DATA".GLOBAL_DATA.AUX6 := #_w2;
   #_w4 := (#_w1 AND "DB4000_FIX_TABLE_POSITIONS".UNIT_1.FIXTURE[3].IN_LOAD_UNLOAD_STATION_1 AND NOT "DB7330_ETXETAR_ROBOT_CELL_INTERLOCK".INTERLOCKS_UNIT_01.MACHINE_TO_ROBOT.MCH_UNLD_ANTICIPATION_FACE_R AND (("DB8000_PART_STATUS".UNIT_1.FIXTURE_3.PART_A.STATUS.CELL_STATUS.NEW_IN_TRANSIT AND "DB2440_GLOBAL_DATA".GLOBAL_DATA.U01_RN_CYCLE_PART_TYPE) OR ("DB8000_PART_STATUS".UNIT_1.FIXTURE_3.PART_A.STATUS.CELL_STATUS.U1_ONE_FACE_DONE_ROTATED AND "DB2440_GLOBAL_DATA".GLOBAL_DATA.U01_NR_CYCLE_PART_TYPE))) OR #_w3;
   "DB2440_GLOBAL_DATA".GLOBAL_DATA.RESET_FULL_DEPTH_PULSE_UNIT_01_FIXT_3 := #_w4 AND NOT "DB2440_GLOBAL_DATA".GLOBAL_DATA.RESET_FULL_DEPTH_UNIT_01_FIXT_3;
   "DB2440_GLOBAL_DATA".GLOBAL_DATA.RESET_FULL_DEPTH_UNIT_01_FIXT_3 := #_w4;
END_REGION

REGION Network 124: RESET FULL DEPTH PULSE UNIT 01 FIXTURE 4
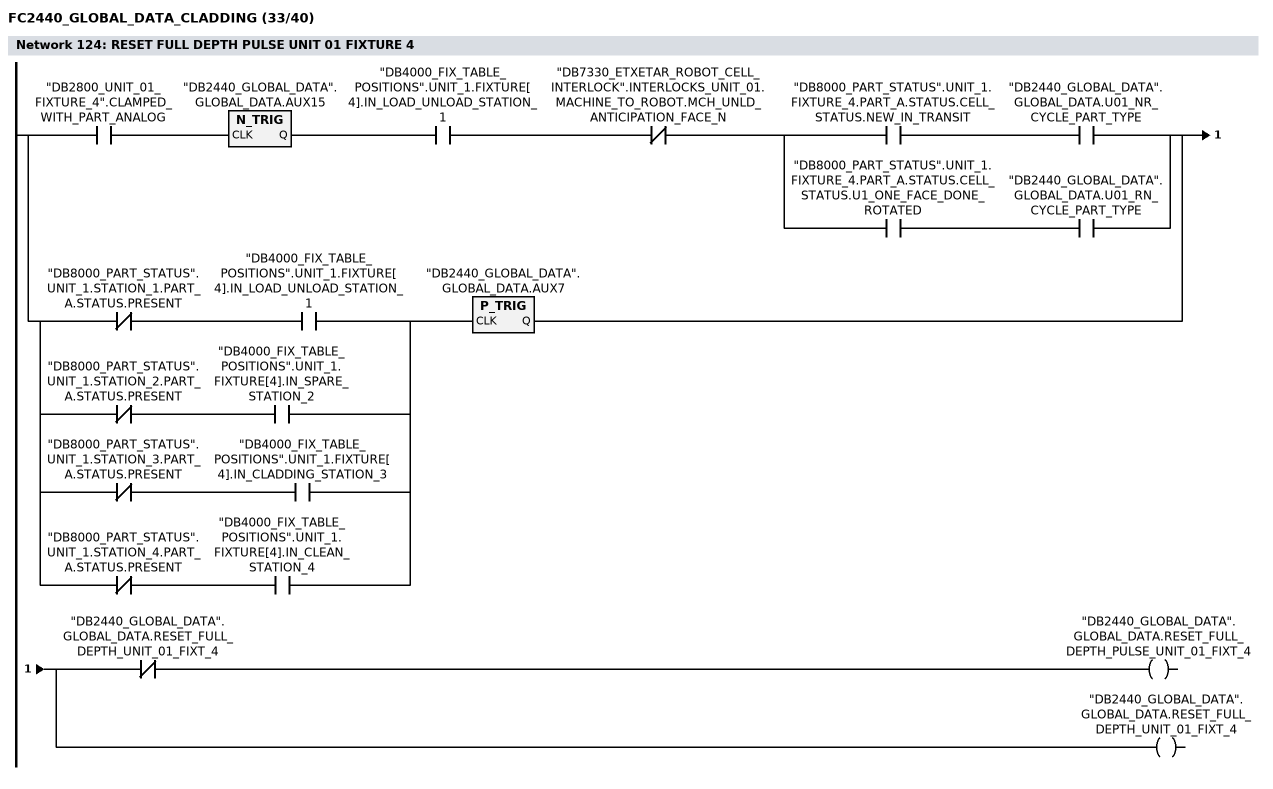
   RUNG wire#powerrail
      Contact( "DB2800_UNIT_01_FIXTURE_4".CLAMPED_WITH_PART_ANALOG )
      N_Trig( "DB2440_GLOBAL_DATA".GLOBAL_DATA.AUX15 )
      Contact( "DB4000_FIX_TABLE_POSITIONS".UNIT_1.FIXTURE[4].IN_LOAD_UNLOAD_STATION_1 )
      I_Contact( "DB7330_ETXETAR_ROBOT_CELL_INTERLOCK".INTERLOCKS_UNIT_01.MACHINE_TO_ROBOT.MCH_UNLD_ANTICIPATION_FACE_N )
      wire#w1
      Contact( "DB8000_PART_STATUS".UNIT_1.FIXTURE_4.PART_A.STATUS.CELL_STATUS.NEW_IN_TRANSIT )
      Contact( "DB2440_GLOBAL_DATA".GLOBAL_DATA.U01_NR_CYCLE_PART_TYPE )
      wire#w2
      I_Contact( "DB2440_GLOBAL_DATA".GLOBAL_DATA.RESET_FULL_DEPTH_UNIT_01_FIXT_4 )
      Coil( "DB2440_GLOBAL_DATA".GLOBAL_DATA.RESET_FULL_DEPTH_PULSE_UNIT_01_FIXT_4 )
   END_RUNG
   RUNG wire#w1
      Contact( "DB8000_PART_STATUS".UNIT_1.FIXTURE_4.PART_A.STATUS.CELL_STATUS.U1_ONE_FACE_DONE_ROTATED )
      Contact( "DB2440_GLOBAL_DATA".GLOBAL_DATA.U01_RN_CYCLE_PART_TYPE )
   END_RUNG wire#w2
   RUNG wire#powerrail
      I_Contact( "DB8000_PART_STATUS".UNIT_1.STATION_1.PART_A.STATUS.PRESENT )
      Contact( "DB4000_FIX_TABLE_POSITIONS".UNIT_1.FIXTURE[4].IN_LOAD_UNLOAD_STATION_1 )
      wire#w3
      P_Trig( "DB2440_GLOBAL_DATA".GLOBAL_DATA.AUX7 )
   END_RUNG wire#w2
   RUNG wire#powerrail
      I_Contact( "DB8000_PART_STATUS".UNIT_1.STATION_2.PART_A.STATUS.PRESENT )
      Contact( "DB4000_FIX_TABLE_POSITIONS".UNIT_1.FIXTURE[4].IN_SPARE_STATION_2 )
   END_RUNG wire#w3
   RUNG wire#powerrail
      I_Contact( "DB8000_PART_STATUS".UNIT_1.STATION_3.PART_A.STATUS.PRESENT )
      Contact( "DB4000_FIX_TABLE_POSITIONS".UNIT_1.FIXTURE[4].IN_CLADDING_STATION_3 )
   END_RUNG wire#w3
   RUNG wire#powerrail
      I_Contact( "DB8000_PART_STATUS".UNIT_1.STATION_4.PART_A.STATUS.PRESENT )
      Contact( "DB4000_FIX_TABLE_POSITIONS".UNIT_1.FIXTURE[4].IN_CLEAN_STATION_4 )
   END_RUNG wire#w3
   RUNG wire#w2
      Coil( "DB2440_GLOBAL_DATA".GLOBAL_DATA.RESET_FULL_DEPTH_UNIT_01_FIXT_4 )
   END_RUNG
   // the same network as SCL:
   #_w1 := NOT "DB2800_UNIT_01_FIXTURE_4".CLAMPED_WITH_PART_ANALOG AND "DB2440_GLOBAL_DATA".GLOBAL_DATA.AUX15;   // falling edge
   "DB2440_GLOBAL_DATA".GLOBAL_DATA.AUX15 := "DB2800_UNIT_01_FIXTURE_4".CLAMPED_WITH_PART_ANALOG;
   #_w2 := (NOT "DB8000_PART_STATUS".UNIT_1.STATION_1.PART_A.STATUS.PRESENT AND "DB4000_FIX_TABLE_POSITIONS".UNIT_1.FIXTURE[4].IN_LOAD_UNLOAD_STATION_1) OR (NOT "DB8000_PART_STATUS".UNIT_1.STATION_2.PART_A.STATUS.PRESENT AND "DB4000_FIX_TABLE_POSITIONS".UNIT_1.FIXTURE[4].IN_SPARE_STATION_2) OR (NOT "DB8000_PART_STATUS".UNIT_1.STATION_3.PART_A.STATUS.PRESENT AND "DB4000_FIX_TABLE_POSITIONS".UNIT_1.FIXTURE[4].IN_CLADDING_STATION_3) OR (NOT "DB8000_PART_STATUS".UNIT_1.STATION_4.PART_A.STATUS.PRESENT AND "DB4000_FIX_TABLE_POSITIONS".UNIT_1.FIXTURE[4].IN_CLEAN_STATION_4);
   #_w3 := #_w2 AND NOT "DB2440_GLOBAL_DATA".GLOBAL_DATA.AUX7;   // rising edge
   "DB2440_GLOBAL_DATA".GLOBAL_DATA.AUX7 := #_w2;
   #_w4 := (#_w1 AND "DB4000_FIX_TABLE_POSITIONS".UNIT_1.FIXTURE[4].IN_LOAD_UNLOAD_STATION_1 AND NOT "DB7330_ETXETAR_ROBOT_CELL_INTERLOCK".INTERLOCKS_UNIT_01.MACHINE_TO_ROBOT.MCH_UNLD_ANTICIPATION_FACE_N AND (("DB8000_PART_STATUS".UNIT_1.FIXTURE_4.PART_A.STATUS.CELL_STATUS.NEW_IN_TRANSIT AND "DB2440_GLOBAL_DATA".GLOBAL_DATA.U01_NR_CYCLE_PART_TYPE) OR ("DB8000_PART_STATUS".UNIT_1.FIXTURE_4.PART_A.STATUS.CELL_STATUS.U1_ONE_FACE_DONE_ROTATED AND "DB2440_GLOBAL_DATA".GLOBAL_DATA.U01_RN_CYCLE_PART_TYPE))) OR #_w3;
   "DB2440_GLOBAL_DATA".GLOBAL_DATA.RESET_FULL_DEPTH_PULSE_UNIT_01_FIXT_4 := #_w4 AND NOT "DB2440_GLOBAL_DATA".GLOBAL_DATA.RESET_FULL_DEPTH_UNIT_01_FIXT_4;
   "DB2440_GLOBAL_DATA".GLOBAL_DATA.RESET_FULL_DEPTH_UNIT_01_FIXT_4 := #_w4;
END_REGION

REGION Network 125: RESET FULL DEPTH PULSE UNIT 02 FIXTURE 1
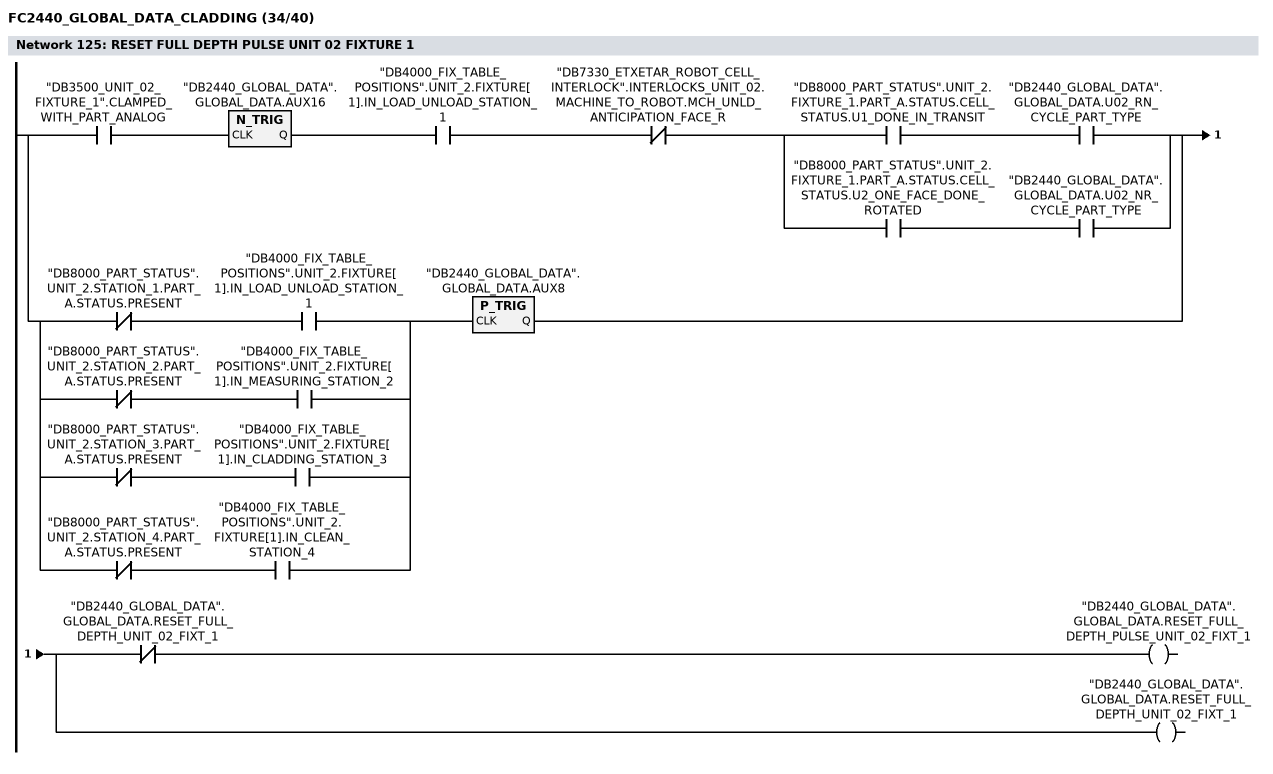
   RUNG wire#powerrail
      Contact( "DB3500_UNIT_02_FIXTURE_1".CLAMPED_WITH_PART_ANALOG )
      N_Trig( "DB2440_GLOBAL_DATA".GLOBAL_DATA.AUX16 )
      Contact( "DB4000_FIX_TABLE_POSITIONS".UNIT_2.FIXTURE[1].IN_LOAD_UNLOAD_STATION_1 )
      I_Contact( "DB7330_ETXETAR_ROBOT_CELL_INTERLOCK".INTERLOCKS_UNIT_02.MACHINE_TO_ROBOT.MCH_UNLD_ANTICIPATION_FACE_R )
      wire#w1
      Contact( "DB8000_PART_STATUS".UNIT_2.FIXTURE_1.PART_A.STATUS.CELL_STATUS.U1_DONE_IN_TRANSIT )
      Contact( "DB2440_GLOBAL_DATA".GLOBAL_DATA.U02_RN_CYCLE_PART_TYPE )
      wire#w2
      I_Contact( "DB2440_GLOBAL_DATA".GLOBAL_DATA.RESET_FULL_DEPTH_UNIT_02_FIXT_1 )
      Coil( "DB2440_GLOBAL_DATA".GLOBAL_DATA.RESET_FULL_DEPTH_PULSE_UNIT_02_FIXT_1 )
   END_RUNG
   RUNG wire#w1
      Contact( "DB8000_PART_STATUS".UNIT_2.FIXTURE_1.PART_A.STATUS.CELL_STATUS.U2_ONE_FACE_DONE_ROTATED )
      Contact( "DB2440_GLOBAL_DATA".GLOBAL_DATA.U02_NR_CYCLE_PART_TYPE )
   END_RUNG wire#w2
   RUNG wire#powerrail
      I_Contact( "DB8000_PART_STATUS".UNIT_2.STATION_1.PART_A.STATUS.PRESENT )
      Contact( "DB4000_FIX_TABLE_POSITIONS".UNIT_2.FIXTURE[1].IN_LOAD_UNLOAD_STATION_1 )
      wire#w3
      P_Trig( "DB2440_GLOBAL_DATA".GLOBAL_DATA.AUX8 )
   END_RUNG wire#w2
   RUNG wire#powerrail
      I_Contact( "DB8000_PART_STATUS".UNIT_2.STATION_2.PART_A.STATUS.PRESENT )
      Contact( "DB4000_FIX_TABLE_POSITIONS".UNIT_2.FIXTURE[1].IN_MEASURING_STATION_2 )
   END_RUNG wire#w3
   RUNG wire#powerrail
      I_Contact( "DB8000_PART_STATUS".UNIT_2.STATION_3.PART_A.STATUS.PRESENT )
      Contact( "DB4000_FIX_TABLE_POSITIONS".UNIT_2.FIXTURE[1].IN_CLADDING_STATION_3 )
   END_RUNG wire#w3
   RUNG wire#powerrail
      I_Contact( "DB8000_PART_STATUS".UNIT_2.STATION_4.PART_A.STATUS.PRESENT )
      Contact( "DB4000_FIX_TABLE_POSITIONS".UNIT_2.FIXTURE[1].IN_CLEAN_STATION_4 )
   END_RUNG wire#w3
   RUNG wire#w2
      Coil( "DB2440_GLOBAL_DATA".GLOBAL_DATA.RESET_FULL_DEPTH_UNIT_02_FIXT_1 )
   END_RUNG
   // the same network as SCL:
   #_w1 := NOT "DB3500_UNIT_02_FIXTURE_1".CLAMPED_WITH_PART_ANALOG AND "DB2440_GLOBAL_DATA".GLOBAL_DATA.AUX16;   // falling edge
   "DB2440_GLOBAL_DATA".GLOBAL_DATA.AUX16 := "DB3500_UNIT_02_FIXTURE_1".CLAMPED_WITH_PART_ANALOG;
   #_w2 := (NOT "DB8000_PART_STATUS".UNIT_2.STATION_1.PART_A.STATUS.PRESENT AND "DB4000_FIX_TABLE_POSITIONS".UNIT_2.FIXTURE[1].IN_LOAD_UNLOAD_STATION_1) OR (NOT "DB8000_PART_STATUS".UNIT_2.STATION_2.PART_A.STATUS.PRESENT AND "DB4000_FIX_TABLE_POSITIONS".UNIT_2.FIXTURE[1].IN_MEASURING_STATION_2) OR (NOT "DB8000_PART_STATUS".UNIT_2.STATION_3.PART_A.STATUS.PRESENT AND "DB4000_FIX_TABLE_POSITIONS".UNIT_2.FIXTURE[1].IN_CLADDING_STATION_3) OR (NOT "DB8000_PART_STATUS".UNIT_2.STATION_4.PART_A.STATUS.PRESENT AND "DB4000_FIX_TABLE_POSITIONS".UNIT_2.FIXTURE[1].IN_CLEAN_STATION_4);
   #_w3 := #_w2 AND NOT "DB2440_GLOBAL_DATA".GLOBAL_DATA.AUX8;   // rising edge
   "DB2440_GLOBAL_DATA".GLOBAL_DATA.AUX8 := #_w2;
   #_w4 := (#_w1 AND "DB4000_FIX_TABLE_POSITIONS".UNIT_2.FIXTURE[1].IN_LOAD_UNLOAD_STATION_1 AND NOT "DB7330_ETXETAR_ROBOT_CELL_INTERLOCK".INTERLOCKS_UNIT_02.MACHINE_TO_ROBOT.MCH_UNLD_ANTICIPATION_FACE_R AND (("DB8000_PART_STATUS".UNIT_2.FIXTURE_1.PART_A.STATUS.CELL_STATUS.U1_DONE_IN_TRANSIT AND "DB2440_GLOBAL_DATA".GLOBAL_DATA.U02_RN_CYCLE_PART_TYPE) OR ("DB8000_PART_STATUS".UNIT_2.FIXTURE_1.PART_A.STATUS.CELL_STATUS.U2_ONE_FACE_DONE_ROTATED AND "DB2440_GLOBAL_DATA".GLOBAL_DATA.U02_NR_CYCLE_PART_TYPE))) OR #_w3;
   "DB2440_GLOBAL_DATA".GLOBAL_DATA.RESET_FULL_DEPTH_PULSE_UNIT_02_FIXT_1 := #_w4 AND NOT "DB2440_GLOBAL_DATA".GLOBAL_DATA.RESET_FULL_DEPTH_UNIT_02_FIXT_1;
   "DB2440_GLOBAL_DATA".GLOBAL_DATA.RESET_FULL_DEPTH_UNIT_02_FIXT_1 := #_w4;
END_REGION

REGION Network 126: RESET FULL DEPTH PULSE UNIT 02 FIXTURE 2
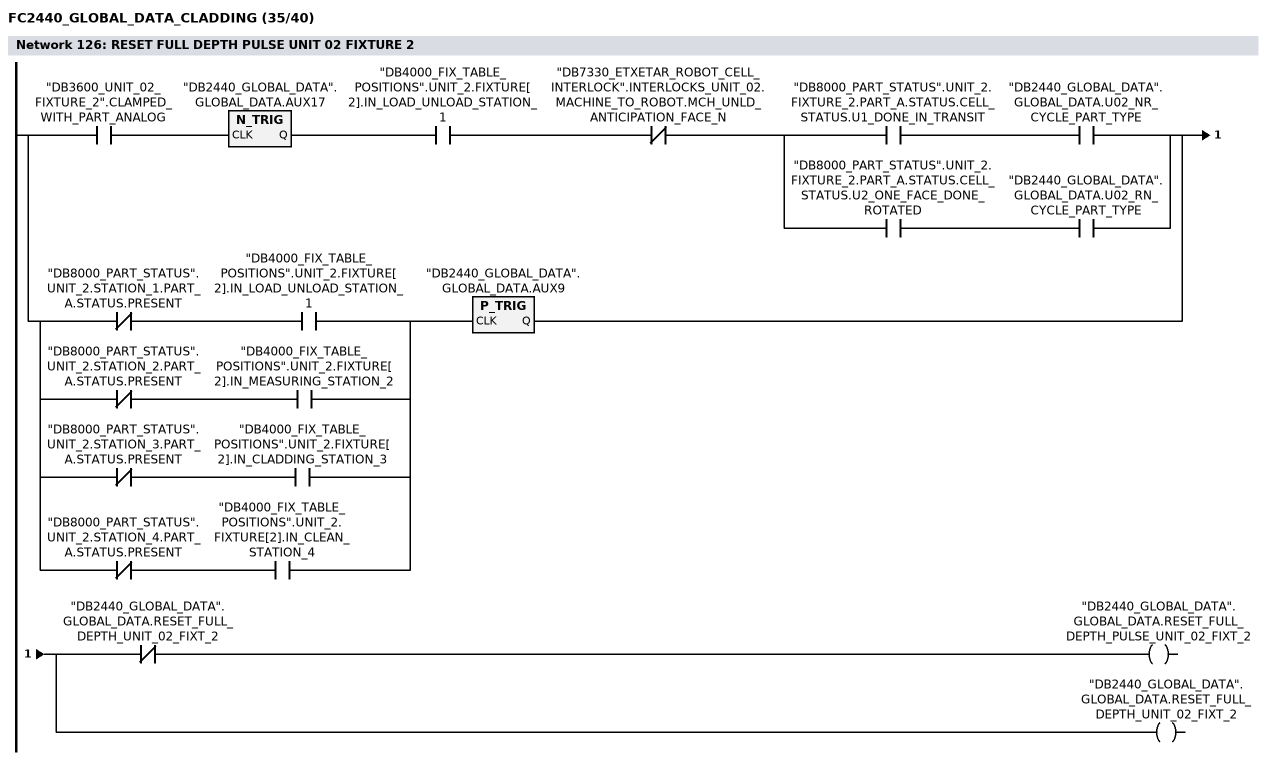
   RUNG wire#powerrail
      Contact( "DB3600_UNIT_02_FIXTURE_2".CLAMPED_WITH_PART_ANALOG )
      N_Trig( "DB2440_GLOBAL_DATA".GLOBAL_DATA.AUX17 )
      Contact( "DB4000_FIX_TABLE_POSITIONS".UNIT_2.FIXTURE[2].IN_LOAD_UNLOAD_STATION_1 )
      I_Contact( "DB7330_ETXETAR_ROBOT_CELL_INTERLOCK".INTERLOCKS_UNIT_02.MACHINE_TO_ROBOT.MCH_UNLD_ANTICIPATION_FACE_N )
      wire#w1
      Contact( "DB8000_PART_STATUS".UNIT_2.FIXTURE_2.PART_A.STATUS.CELL_STATUS.U1_DONE_IN_TRANSIT )
      Contact( "DB2440_GLOBAL_DATA".GLOBAL_DATA.U02_NR_CYCLE_PART_TYPE )
      wire#w2
      I_Contact( "DB2440_GLOBAL_DATA".GLOBAL_DATA.RESET_FULL_DEPTH_UNIT_02_FIXT_2 )
      Coil( "DB2440_GLOBAL_DATA".GLOBAL_DATA.RESET_FULL_DEPTH_PULSE_UNIT_02_FIXT_2 )
   END_RUNG
   RUNG wire#w1
      Contact( "DB8000_PART_STATUS".UNIT_2.FIXTURE_2.PART_A.STATUS.CELL_STATUS.U2_ONE_FACE_DONE_ROTATED )
      Contact( "DB2440_GLOBAL_DATA".GLOBAL_DATA.U02_RN_CYCLE_PART_TYPE )
   END_RUNG wire#w2
   RUNG wire#powerrail
      I_Contact( "DB8000_PART_STATUS".UNIT_2.STATION_1.PART_A.STATUS.PRESENT )
      Contact( "DB4000_FIX_TABLE_POSITIONS".UNIT_2.FIXTURE[2].IN_LOAD_UNLOAD_STATION_1 )
      wire#w3
      P_Trig( "DB2440_GLOBAL_DATA".GLOBAL_DATA.AUX9 )
   END_RUNG wire#w2
   RUNG wire#powerrail
      I_Contact( "DB8000_PART_STATUS".UNIT_2.STATION_2.PART_A.STATUS.PRESENT )
      Contact( "DB4000_FIX_TABLE_POSITIONS".UNIT_2.FIXTURE[2].IN_MEASURING_STATION_2 )
   END_RUNG wire#w3
   RUNG wire#powerrail
      I_Contact( "DB8000_PART_STATUS".UNIT_2.STATION_3.PART_A.STATUS.PRESENT )
      Contact( "DB4000_FIX_TABLE_POSITIONS".UNIT_2.FIXTURE[2].IN_CLADDING_STATION_3 )
   END_RUNG wire#w3
   RUNG wire#powerrail
      I_Contact( "DB8000_PART_STATUS".UNIT_2.STATION_4.PART_A.STATUS.PRESENT )
      Contact( "DB4000_FIX_TABLE_POSITIONS".UNIT_2.FIXTURE[2].IN_CLEAN_STATION_4 )
   END_RUNG wire#w3
   RUNG wire#w2
      Coil( "DB2440_GLOBAL_DATA".GLOBAL_DATA.RESET_FULL_DEPTH_UNIT_02_FIXT_2 )
   END_RUNG
   // the same network as SCL:
   #_w1 := NOT "DB3600_UNIT_02_FIXTURE_2".CLAMPED_WITH_PART_ANALOG AND "DB2440_GLOBAL_DATA".GLOBAL_DATA.AUX17;   // falling edge
   "DB2440_GLOBAL_DATA".GLOBAL_DATA.AUX17 := "DB3600_UNIT_02_FIXTURE_2".CLAMPED_WITH_PART_ANALOG;
   #_w2 := (NOT "DB8000_PART_STATUS".UNIT_2.STATION_1.PART_A.STATUS.PRESENT AND "DB4000_FIX_TABLE_POSITIONS".UNIT_2.FIXTURE[2].IN_LOAD_UNLOAD_STATION_1) OR (NOT "DB8000_PART_STATUS".UNIT_2.STATION_2.PART_A.STATUS.PRESENT AND "DB4000_FIX_TABLE_POSITIONS".UNIT_2.FIXTURE[2].IN_MEASURING_STATION_2) OR (NOT "DB8000_PART_STATUS".UNIT_2.STATION_3.PART_A.STATUS.PRESENT AND "DB4000_FIX_TABLE_POSITIONS".UNIT_2.FIXTURE[2].IN_CLADDING_STATION_3) OR (NOT "DB8000_PART_STATUS".UNIT_2.STATION_4.PART_A.STATUS.PRESENT AND "DB4000_FIX_TABLE_POSITIONS".UNIT_2.FIXTURE[2].IN_CLEAN_STATION_4);
   #_w3 := #_w2 AND NOT "DB2440_GLOBAL_DATA".GLOBAL_DATA.AUX9;   // rising edge
   "DB2440_GLOBAL_DATA".GLOBAL_DATA.AUX9 := #_w2;
   #_w4 := (#_w1 AND "DB4000_FIX_TABLE_POSITIONS".UNIT_2.FIXTURE[2].IN_LOAD_UNLOAD_STATION_1 AND NOT "DB7330_ETXETAR_ROBOT_CELL_INTERLOCK".INTERLOCKS_UNIT_02.MACHINE_TO_ROBOT.MCH_UNLD_ANTICIPATION_FACE_N AND (("DB8000_PART_STATUS".UNIT_2.FIXTURE_2.PART_A.STATUS.CELL_STATUS.U1_DONE_IN_TRANSIT AND "DB2440_GLOBAL_DATA".GLOBAL_DATA.U02_NR_CYCLE_PART_TYPE) OR ("DB8000_PART_STATUS".UNIT_2.FIXTURE_2.PART_A.STATUS.CELL_STATUS.U2_ONE_FACE_DONE_ROTATED AND "DB2440_GLOBAL_DATA".GLOBAL_DATA.U02_RN_CYCLE_PART_TYPE))) OR #_w3;
   "DB2440_GLOBAL_DATA".GLOBAL_DATA.RESET_FULL_DEPTH_PULSE_UNIT_02_FIXT_2 := #_w4 AND NOT "DB2440_GLOBAL_DATA".GLOBAL_DATA.RESET_FULL_DEPTH_UNIT_02_FIXT_2;
   "DB2440_GLOBAL_DATA".GLOBAL_DATA.RESET_FULL_DEPTH_UNIT_02_FIXT_2 := #_w4;
END_REGION

REGION Network 127: RESET FULL DEPTH PULSE UNIT 02 FIXTURE 3
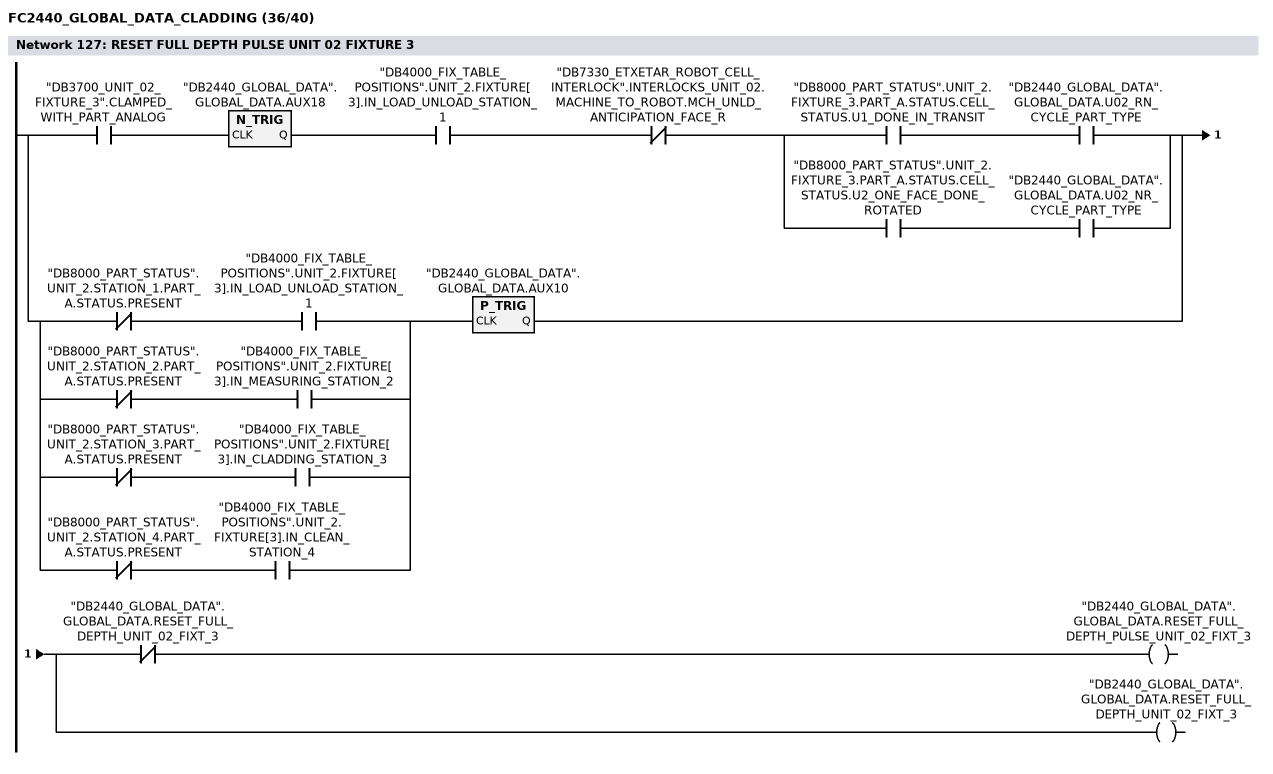
   RUNG wire#powerrail
      Contact( "DB3700_UNIT_02_FIXTURE_3".CLAMPED_WITH_PART_ANALOG )
      N_Trig( "DB2440_GLOBAL_DATA".GLOBAL_DATA.AUX18 )
      Contact( "DB4000_FIX_TABLE_POSITIONS".UNIT_2.FIXTURE[3].IN_LOAD_UNLOAD_STATION_1 )
      I_Contact( "DB7330_ETXETAR_ROBOT_CELL_INTERLOCK".INTERLOCKS_UNIT_02.MACHINE_TO_ROBOT.MCH_UNLD_ANTICIPATION_FACE_R )
      wire#w1
      Contact( "DB8000_PART_STATUS".UNIT_2.FIXTURE_3.PART_A.STATUS.CELL_STATUS.U1_DONE_IN_TRANSIT )
      Contact( "DB2440_GLOBAL_DATA".GLOBAL_DATA.U02_RN_CYCLE_PART_TYPE )
      wire#w2
      I_Contact( "DB2440_GLOBAL_DATA".GLOBAL_DATA.RESET_FULL_DEPTH_UNIT_02_FIXT_3 )
      Coil( "DB2440_GLOBAL_DATA".GLOBAL_DATA.RESET_FULL_DEPTH_PULSE_UNIT_02_FIXT_3 )
   END_RUNG
   RUNG wire#w1
      Contact( "DB8000_PART_STATUS".UNIT_2.FIXTURE_3.PART_A.STATUS.CELL_STATUS.U2_ONE_FACE_DONE_ROTATED )
      Contact( "DB2440_GLOBAL_DATA".GLOBAL_DATA.U02_NR_CYCLE_PART_TYPE )
   END_RUNG wire#w2
   RUNG wire#powerrail
      I_Contact( "DB8000_PART_STATUS".UNIT_2.STATION_1.PART_A.STATUS.PRESENT )
      Contact( "DB4000_FIX_TABLE_POSITIONS".UNIT_2.FIXTURE[3].IN_LOAD_UNLOAD_STATION_1 )
      wire#w3
      P_Trig( "DB2440_GLOBAL_DATA".GLOBAL_DATA.AUX10 )
   END_RUNG wire#w2
   RUNG wire#powerrail
      I_Contact( "DB8000_PART_STATUS".UNIT_2.STATION_2.PART_A.STATUS.PRESENT )
      Contact( "DB4000_FIX_TABLE_POSITIONS".UNIT_2.FIXTURE[3].IN_MEASURING_STATION_2 )
   END_RUNG wire#w3
   RUNG wire#powerrail
      I_Contact( "DB8000_PART_STATUS".UNIT_2.STATION_3.PART_A.STATUS.PRESENT )
      Contact( "DB4000_FIX_TABLE_POSITIONS".UNIT_2.FIXTURE[3].IN_CLADDING_STATION_3 )
   END_RUNG wire#w3
   RUNG wire#powerrail
      I_Contact( "DB8000_PART_STATUS".UNIT_2.STATION_4.PART_A.STATUS.PRESENT )
      Contact( "DB4000_FIX_TABLE_POSITIONS".UNIT_2.FIXTURE[3].IN_CLEAN_STATION_4 )
   END_RUNG wire#w3
   RUNG wire#w2
      Coil( "DB2440_GLOBAL_DATA".GLOBAL_DATA.RESET_FULL_DEPTH_UNIT_02_FIXT_3 )
   END_RUNG
   // the same network as SCL:
   #_w1 := NOT "DB3700_UNIT_02_FIXTURE_3".CLAMPED_WITH_PART_ANALOG AND "DB2440_GLOBAL_DATA".GLOBAL_DATA.AUX18;   // falling edge
   "DB2440_GLOBAL_DATA".GLOBAL_DATA.AUX18 := "DB3700_UNIT_02_FIXTURE_3".CLAMPED_WITH_PART_ANALOG;
   #_w2 := (NOT "DB8000_PART_STATUS".UNIT_2.STATION_1.PART_A.STATUS.PRESENT AND "DB4000_FIX_TABLE_POSITIONS".UNIT_2.FIXTURE[3].IN_LOAD_UNLOAD_STATION_1) OR (NOT "DB8000_PART_STATUS".UNIT_2.STATION_2.PART_A.STATUS.PRESENT AND "DB4000_FIX_TABLE_POSITIONS".UNIT_2.FIXTURE[3].IN_MEASURING_STATION_2) OR (NOT "DB8000_PART_STATUS".UNIT_2.STATION_3.PART_A.STATUS.PRESENT AND "DB4000_FIX_TABLE_POSITIONS".UNIT_2.FIXTURE[3].IN_CLADDING_STATION_3) OR (NOT "DB8000_PART_STATUS".UNIT_2.STATION_4.PART_A.STATUS.PRESENT AND "DB4000_FIX_TABLE_POSITIONS".UNIT_2.FIXTURE[3].IN_CLEAN_STATION_4);
   #_w3 := #_w2 AND NOT "DB2440_GLOBAL_DATA".GLOBAL_DATA.AUX10;   // rising edge
   "DB2440_GLOBAL_DATA".GLOBAL_DATA.AUX10 := #_w2;
   #_w4 := (#_w1 AND "DB4000_FIX_TABLE_POSITIONS".UNIT_2.FIXTURE[3].IN_LOAD_UNLOAD_STATION_1 AND NOT "DB7330_ETXETAR_ROBOT_CELL_INTERLOCK".INTERLOCKS_UNIT_02.MACHINE_TO_ROBOT.MCH_UNLD_ANTICIPATION_FACE_R AND (("DB8000_PART_STATUS".UNIT_2.FIXTURE_3.PART_A.STATUS.CELL_STATUS.U1_DONE_IN_TRANSIT AND "DB2440_GLOBAL_DATA".GLOBAL_DATA.U02_RN_CYCLE_PART_TYPE) OR ("DB8000_PART_STATUS".UNIT_2.FIXTURE_3.PART_A.STATUS.CELL_STATUS.U2_ONE_FACE_DONE_ROTATED AND "DB2440_GLOBAL_DATA".GLOBAL_DATA.U02_NR_CYCLE_PART_TYPE))) OR #_w3;
   "DB2440_GLOBAL_DATA".GLOBAL_DATA.RESET_FULL_DEPTH_PULSE_UNIT_02_FIXT_3 := #_w4 AND NOT "DB2440_GLOBAL_DATA".GLOBAL_DATA.RESET_FULL_DEPTH_UNIT_02_FIXT_3;
   "DB2440_GLOBAL_DATA".GLOBAL_DATA.RESET_FULL_DEPTH_UNIT_02_FIXT_3 := #_w4;
END_REGION

REGION Network 128: RESET FULL DEPTH PULSE UNIT 02 FIXTURE 4
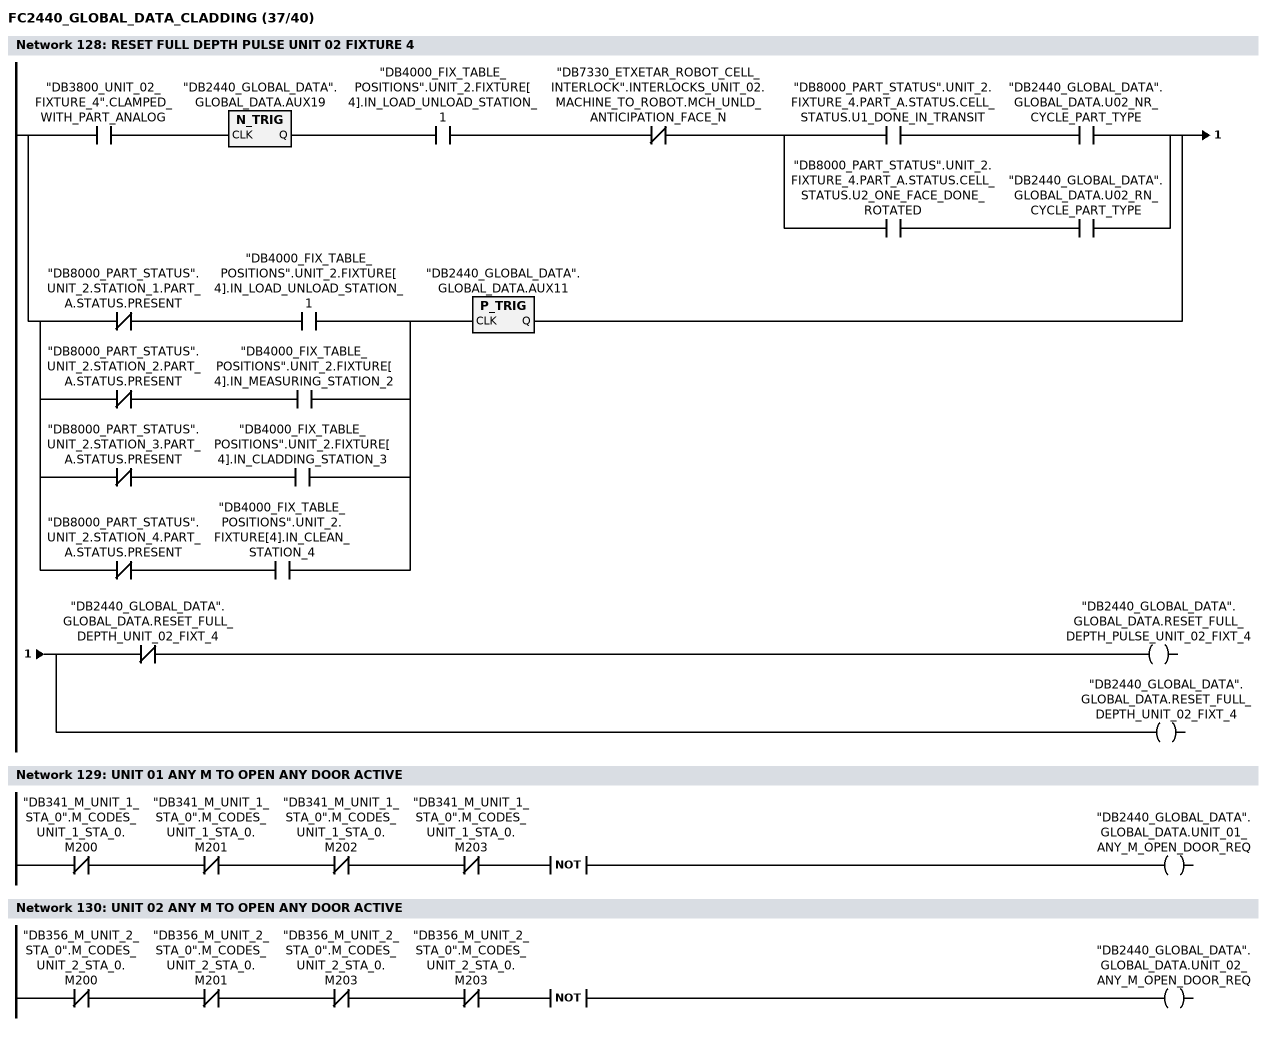
   RUNG wire#powerrail
      Contact( "DB3800_UNIT_02_FIXTURE_4".CLAMPED_WITH_PART_ANALOG )
      N_Trig( "DB2440_GLOBAL_DATA".GLOBAL_DATA.AUX19 )
      Contact( "DB4000_FIX_TABLE_POSITIONS".UNIT_2.FIXTURE[4].IN_LOAD_UNLOAD_STATION_1 )
      I_Contact( "DB7330_ETXETAR_ROBOT_CELL_INTERLOCK".INTERLOCKS_UNIT_02.MACHINE_TO_ROBOT.MCH_UNLD_ANTICIPATION_FACE_N )
      wire#w1
      Contact( "DB8000_PART_STATUS".UNIT_2.FIXTURE_4.PART_A.STATUS.CELL_STATUS.U1_DONE_IN_TRANSIT )
      Contact( "DB2440_GLOBAL_DATA".GLOBAL_DATA.U02_NR_CYCLE_PART_TYPE )
      wire#w2
      I_Contact( "DB2440_GLOBAL_DATA".GLOBAL_DATA.RESET_FULL_DEPTH_UNIT_02_FIXT_4 )
      Coil( "DB2440_GLOBAL_DATA".GLOBAL_DATA.RESET_FULL_DEPTH_PULSE_UNIT_02_FIXT_4 )
   END_RUNG
   RUNG wire#w1
      Contact( "DB8000_PART_STATUS".UNIT_2.FIXTURE_4.PART_A.STATUS.CELL_STATUS.U2_ONE_FACE_DONE_ROTATED )
      Contact( "DB2440_GLOBAL_DATA".GLOBAL_DATA.U02_RN_CYCLE_PART_TYPE )
   END_RUNG wire#w2
   RUNG wire#powerrail
      I_Contact( "DB8000_PART_STATUS".UNIT_2.STATION_1.PART_A.STATUS.PRESENT )
      Contact( "DB4000_FIX_TABLE_POSITIONS".UNIT_2.FIXTURE[4].IN_LOAD_UNLOAD_STATION_1 )
      wire#w3
      P_Trig( "DB2440_GLOBAL_DATA".GLOBAL_DATA.AUX11 )
   END_RUNG wire#w2
   RUNG wire#powerrail
      I_Contact( "DB8000_PART_STATUS".UNIT_2.STATION_2.PART_A.STATUS.PRESENT )
      Contact( "DB4000_FIX_TABLE_POSITIONS".UNIT_2.FIXTURE[4].IN_MEASURING_STATION_2 )
   END_RUNG wire#w3
   RUNG wire#powerrail
      I_Contact( "DB8000_PART_STATUS".UNIT_2.STATION_3.PART_A.STATUS.PRESENT )
      Contact( "DB4000_FIX_TABLE_POSITIONS".UNIT_2.FIXTURE[4].IN_CLADDING_STATION_3 )
   END_RUNG wire#w3
   RUNG wire#powerrail
      I_Contact( "DB8000_PART_STATUS".UNIT_2.STATION_4.PART_A.STATUS.PRESENT )
      Contact( "DB4000_FIX_TABLE_POSITIONS".UNIT_2.FIXTURE[4].IN_CLEAN_STATION_4 )
   END_RUNG wire#w3
   RUNG wire#w2
      Coil( "DB2440_GLOBAL_DATA".GLOBAL_DATA.RESET_FULL_DEPTH_UNIT_02_FIXT_4 )
   END_RUNG
   // the same network as SCL:
   #_w1 := NOT "DB3800_UNIT_02_FIXTURE_4".CLAMPED_WITH_PART_ANALOG AND "DB2440_GLOBAL_DATA".GLOBAL_DATA.AUX19;   // falling edge
   "DB2440_GLOBAL_DATA".GLOBAL_DATA.AUX19 := "DB3800_UNIT_02_FIXTURE_4".CLAMPED_WITH_PART_ANALOG;
   #_w2 := (NOT "DB8000_PART_STATUS".UNIT_2.STATION_1.PART_A.STATUS.PRESENT AND "DB4000_FIX_TABLE_POSITIONS".UNIT_2.FIXTURE[4].IN_LOAD_UNLOAD_STATION_1) OR (NOT "DB8000_PART_STATUS".UNIT_2.STATION_2.PART_A.STATUS.PRESENT AND "DB4000_FIX_TABLE_POSITIONS".UNIT_2.FIXTURE[4].IN_MEASURING_STATION_2) OR (NOT "DB8000_PART_STATUS".UNIT_2.STATION_3.PART_A.STATUS.PRESENT AND "DB4000_FIX_TABLE_POSITIONS".UNIT_2.FIXTURE[4].IN_CLADDING_STATION_3) OR (NOT "DB8000_PART_STATUS".UNIT_2.STATION_4.PART_A.STATUS.PRESENT AND "DB4000_FIX_TABLE_POSITIONS".UNIT_2.FIXTURE[4].IN_CLEAN_STATION_4);
   #_w3 := #_w2 AND NOT "DB2440_GLOBAL_DATA".GLOBAL_DATA.AUX11;   // rising edge
   "DB2440_GLOBAL_DATA".GLOBAL_DATA.AUX11 := #_w2;
   #_w4 := (#_w1 AND "DB4000_FIX_TABLE_POSITIONS".UNIT_2.FIXTURE[4].IN_LOAD_UNLOAD_STATION_1 AND NOT "DB7330_ETXETAR_ROBOT_CELL_INTERLOCK".INTERLOCKS_UNIT_02.MACHINE_TO_ROBOT.MCH_UNLD_ANTICIPATION_FACE_N AND (("DB8000_PART_STATUS".UNIT_2.FIXTURE_4.PART_A.STATUS.CELL_STATUS.U1_DONE_IN_TRANSIT AND "DB2440_GLOBAL_DATA".GLOBAL_DATA.U02_NR_CYCLE_PART_TYPE) OR ("DB8000_PART_STATUS".UNIT_2.FIXTURE_4.PART_A.STATUS.CELL_STATUS.U2_ONE_FACE_DONE_ROTATED AND "DB2440_GLOBAL_DATA".GLOBAL_DATA.U02_RN_CYCLE_PART_TYPE))) OR #_w3;
   "DB2440_GLOBAL_DATA".GLOBAL_DATA.RESET_FULL_DEPTH_PULSE_UNIT_02_FIXT_4 := #_w4 AND NOT "DB2440_GLOBAL_DATA".GLOBAL_DATA.RESET_FULL_DEPTH_UNIT_02_FIXT_4;
   "DB2440_GLOBAL_DATA".GLOBAL_DATA.RESET_FULL_DEPTH_UNIT_02_FIXT_4 := #_w4;
END_REGION

REGION Network 129: UNIT 01 ANY M TO OPEN ANY DOOR ACTIVE
   RUNG wire#powerrail
      I_Contact( "DB341_M_UNIT_1_STA_0".M_CODES_UNIT_1_STA_0.M200 )
      I_Contact( "DB341_M_UNIT_1_STA_0".M_CODES_UNIT_1_STA_0.M201 )
      I_Contact( "DB341_M_UNIT_1_STA_0".M_CODES_UNIT_1_STA_0.M202 )
      I_Contact( "DB341_M_UNIT_1_STA_0".M_CODES_UNIT_1_STA_0.M203 )
      Not()
      Coil( "DB2440_GLOBAL_DATA".GLOBAL_DATA.UNIT_01_ANY_M_OPEN_DOOR_REQ )
   END_RUNG
   // the same network as SCL:
   "DB2440_GLOBAL_DATA".GLOBAL_DATA.UNIT_01_ANY_M_OPEN_DOOR_REQ := NOT (NOT "DB341_M_UNIT_1_STA_0".M_CODES_UNIT_1_STA_0.M200 AND NOT "DB341_M_UNIT_1_STA_0".M_CODES_UNIT_1_STA_0.M201 AND NOT "DB341_M_UNIT_1_STA_0".M_CODES_UNIT_1_STA_0.M202 AND NOT "DB341_M_UNIT_1_STA_0".M_CODES_UNIT_1_STA_0.M203);
END_REGION

REGION Network 130: UNIT 02 ANY M TO OPEN ANY DOOR ACTIVE
   RUNG wire#powerrail
      I_Contact( "DB356_M_UNIT_2_STA_0".M_CODES_UNIT_2_STA_0.M200 )
      I_Contact( "DB356_M_UNIT_2_STA_0".M_CODES_UNIT_2_STA_0.M201 )
      I_Contact( "DB356_M_UNIT_2_STA_0".M_CODES_UNIT_2_STA_0.M203 )
      I_Contact( "DB356_M_UNIT_2_STA_0".M_CODES_UNIT_2_STA_0.M203 )
      Not()
      Coil( "DB2440_GLOBAL_DATA".GLOBAL_DATA.UNIT_02_ANY_M_OPEN_DOOR_REQ )
   END_RUNG
   // the same network as SCL:
   "DB2440_GLOBAL_DATA".GLOBAL_DATA.UNIT_02_ANY_M_OPEN_DOOR_REQ := NOT (NOT "DB356_M_UNIT_2_STA_0".M_CODES_UNIT_2_STA_0.M200 AND NOT "DB356_M_UNIT_2_STA_0".M_CODES_UNIT_2_STA_0.M201 AND NOT "DB356_M_UNIT_2_STA_0".M_CODES_UNIT_2_STA_0.M203 AND NOT "DB356_M_UNIT_2_STA_0".M_CODES_UNIT_2_STA_0.M203);
END_REGION

REGION Network 131: FIXTURE IN UNIT 01 STATION 0 ANY CALIBRATION MISSING
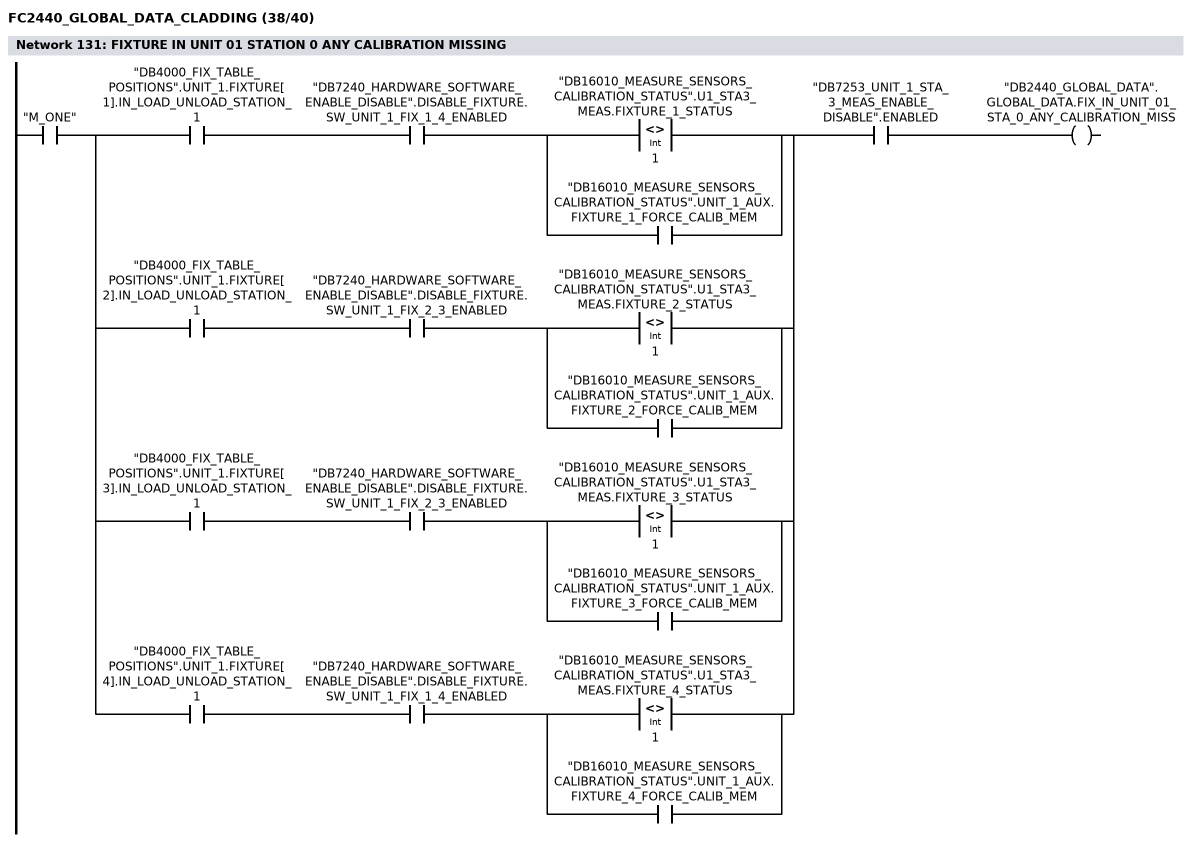
   RUNG wire#powerrail
      Contact( "M_ONE" )
      wire#w1
      Contact( "DB4000_FIX_TABLE_POSITIONS".UNIT_1.FIXTURE[1].IN_LOAD_UNLOAD_STATION_1 )
      Contact( "DB7240_HARDWARE_SOFTWARE_ENABLE_DISABLE".DISABLE_FIXTURE.SW_UNIT_1_FIX_1_4_ENABLED )
      wire#w2
      { S7_Templates := "SrcType := Int" } NE_Contact(in1 := "DB16010_MEASURE_SENSORS_CALIBRATION_STATUS".U1_STA3_MEAS.FIXTURE_1_STATUS, in2 := 1)
      wire#w3
      Contact( "DB7253_UNIT_1_STA_3_MEAS_ENABLE_DISABLE".ENABLED )
      Coil( "DB2440_GLOBAL_DATA".GLOBAL_DATA.FIX_IN_UNIT_01_STA_0_ANY_CALIBRATION_MISS )
   END_RUNG
   RUNG wire#w2
      Contact( "DB16010_MEASURE_SENSORS_CALIBRATION_STATUS".UNIT_1_AUX.FIXTURE_1_FORCE_CALIB_MEM )
   END_RUNG wire#w3
   RUNG wire#w1
      Contact( "DB4000_FIX_TABLE_POSITIONS".UNIT_1.FIXTURE[2].IN_LOAD_UNLOAD_STATION_1 )
      Contact( "DB7240_HARDWARE_SOFTWARE_ENABLE_DISABLE".DISABLE_FIXTURE.SW_UNIT_1_FIX_2_3_ENABLED )
      wire#w4
      { S7_Templates := "SrcType := Int" } NE_Contact(in1 := "DB16010_MEASURE_SENSORS_CALIBRATION_STATUS".U1_STA3_MEAS.FIXTURE_2_STATUS, in2 := 1)
   END_RUNG wire#w3
   RUNG wire#w4
      Contact( "DB16010_MEASURE_SENSORS_CALIBRATION_STATUS".UNIT_1_AUX.FIXTURE_2_FORCE_CALIB_MEM )
   END_RUNG wire#w3
   RUNG wire#w1
      Contact( "DB4000_FIX_TABLE_POSITIONS".UNIT_1.FIXTURE[3].IN_LOAD_UNLOAD_STATION_1 )
      Contact( "DB7240_HARDWARE_SOFTWARE_ENABLE_DISABLE".DISABLE_FIXTURE.SW_UNIT_1_FIX_2_3_ENABLED )
      wire#w5
      { S7_Templates := "SrcType := Int" } NE_Contact(in1 := "DB16010_MEASURE_SENSORS_CALIBRATION_STATUS".U1_STA3_MEAS.FIXTURE_3_STATUS, in2 := 1)
   END_RUNG wire#w3
   RUNG wire#w5
      Contact( "DB16010_MEASURE_SENSORS_CALIBRATION_STATUS".UNIT_1_AUX.FIXTURE_3_FORCE_CALIB_MEM )
   END_RUNG wire#w3
   RUNG wire#w1
      Contact( "DB4000_FIX_TABLE_POSITIONS".UNIT_1.FIXTURE[4].IN_LOAD_UNLOAD_STATION_1 )
      Contact( "DB7240_HARDWARE_SOFTWARE_ENABLE_DISABLE".DISABLE_FIXTURE.SW_UNIT_1_FIX_1_4_ENABLED )
      wire#w6
      { S7_Templates := "SrcType := Int" } NE_Contact(in1 := "DB16010_MEASURE_SENSORS_CALIBRATION_STATUS".U1_STA3_MEAS.FIXTURE_4_STATUS, in2 := 1)
   END_RUNG wire#w3
   RUNG wire#w6
      Contact( "DB16010_MEASURE_SENSORS_CALIBRATION_STATUS".UNIT_1_AUX.FIXTURE_4_FORCE_CALIB_MEM )
   END_RUNG wire#w3
   // the same network as SCL:
   "DB2440_GLOBAL_DATA".GLOBAL_DATA.FIX_IN_UNIT_01_STA_0_ANY_CALIBRATION_MISS := "M_ONE" AND (("DB4000_FIX_TABLE_POSITIONS".UNIT_1.FIXTURE[1].IN_LOAD_UNLOAD_STATION_1 AND "DB7240_HARDWARE_SOFTWARE_ENABLE_DISABLE".DISABLE_FIXTURE.SW_UNIT_1_FIX_1_4_ENABLED AND (("DB16010_MEASURE_SENSORS_CALIBRATION_STATUS".U1_STA3_MEAS.FIXTURE_1_STATUS <> 1) OR "DB16010_MEASURE_SENSORS_CALIBRATION_STATUS".UNIT_1_AUX.FIXTURE_1_FORCE_CALIB_MEM)) OR ("DB4000_FIX_TABLE_POSITIONS".UNIT_1.FIXTURE[2].IN_LOAD_UNLOAD_STATION_1 AND "DB7240_HARDWARE_SOFTWARE_ENABLE_DISABLE".DISABLE_FIXTURE.SW_UNIT_1_FIX_2_3_ENABLED AND (("DB16010_MEASURE_SENSORS_CALIBRATION_STATUS".U1_STA3_MEAS.FIXTURE_2_STATUS <> 1) OR "DB16010_MEASURE_SENSORS_CALIBRATION_STATUS".UNIT_1_AUX.FIXTURE_2_FORCE_CALIB_MEM)) OR ("DB4000_FIX_TABLE_POSITIONS".UNIT_1.FIXTURE[3].IN_LOAD_UNLOAD_STATION_1 AND "DB7240_HARDWARE_SOFTWARE_ENABLE_DISABLE".DISABLE_FIXTURE.SW_UNIT_1_FIX_2_3_ENABLED AND (("DB16010_MEASURE_SENSORS_CALIBRATION_STATUS".U1_STA3_MEAS.FIXTURE_3_STATUS <> 1) OR "DB16010_MEASURE_SENSORS_CALIBRATION_STATUS".UNIT_1_AUX.FIXTURE_3_FORCE_CALIB_MEM)) OR ("DB4000_FIX_TABLE_POSITIONS".UNIT_1.FIXTURE[4].IN_LOAD_UNLOAD_STATION_1 AND "DB7240_HARDWARE_SOFTWARE_ENABLE_DISABLE".DISABLE_FIXTURE.SW_UNIT_1_FIX_1_4_ENABLED AND (("DB16010_MEASURE_SENSORS_CALIBRATION_STATUS".U1_STA3_MEAS.FIXTURE_4_STATUS <> 1) OR "DB16010_MEASURE_SENSORS_CALIBRATION_STATUS".UNIT_1_AUX.FIXTURE_4_FORCE_CALIB_MEM))) AND "DB7253_UNIT_1_STA_3_MEAS_ENABLE_DISABLE".ENABLED;
END_REGION

